REGION Network 79: TMP - ERROR - Tout Bajar Tope
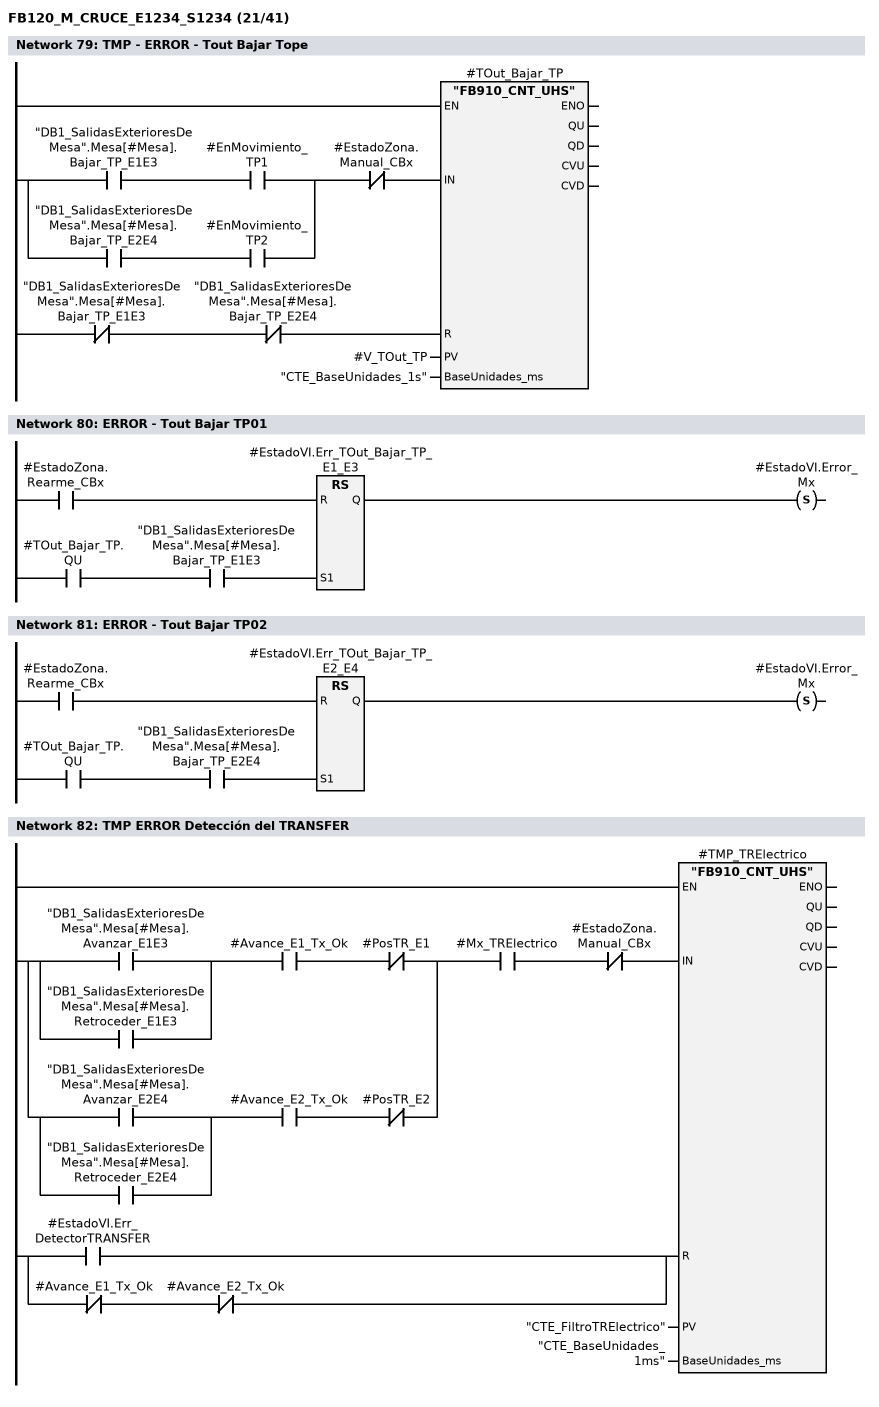
   RUNG wire#powerrail
      #TOut_Bajar_TP(IN := wire#w2, R := wire#w3, PV := #V_TOut_TP, BaseUnidades_ms := "CTE_BaseUnidades_1s", QU =>, QD =>, CVU =>, CVD =>)
   END_RUNG
   RUNG wire#powerrail
      Contact( "DB1_SalidasExterioresDeMesa".Mesa[#Mesa].Bajar_TP_E1E3 )
      Contact( #EnMovimiento_TP1 )
      wire#w1
      I_Contact( #EstadoZona.Manual_CBx )
   END_RUNG wire#w2
   RUNG wire#powerrail
      Contact( "DB1_SalidasExterioresDeMesa".Mesa[#Mesa].Bajar_TP_E2E4 )
      Contact( #EnMovimiento_TP2 )
   END_RUNG wire#w1
   RUNG wire#powerrail
      I_Contact( "DB1_SalidasExterioresDeMesa".Mesa[#Mesa].Bajar_TP_E1E3 )
      I_Contact( "DB1_SalidasExterioresDeMesa".Mesa[#Mesa].Bajar_TP_E2E4 )
   END_RUNG wire#w3
   // the same network as SCL:
   #TOut_Bajar_TP(IN := (("DB1_SalidasExterioresDeMesa".Mesa[#Mesa].Bajar_TP_E1E3 AND #EnMovimiento_TP1) OR ("DB1_SalidasExterioresDeMesa".Mesa[#Mesa].Bajar_TP_E2E4 AND #EnMovimiento_TP2)) AND NOT #EstadoZona.Manual_CBx,   // "FB910_CNT_UHS"
                  R := NOT "DB1_SalidasExterioresDeMesa".Mesa[#Mesa].Bajar_TP_E1E3 AND NOT "DB1_SalidasExterioresDeMesa".Mesa[#Mesa].Bajar_TP_E2E4,
                  PV := #V_TOut_TP,
                  BaseUnidades_ms := "CTE_BaseUnidades_1s");
END_REGION

REGION Network 80: ERROR - Tout Bajar TP01
   RUNG wire#powerrail
      Contact( #EstadoZona.Rearme_CBx )
      S_RS(operand := #EstadoVI.Err_TOut_Bajar_TP_E1_E3, s1 := wire#w1)
      S_Coil( #EstadoVI.Error_Mx )
   END_RUNG
   RUNG wire#powerrail
      Contact( #TOut_Bajar_TP.QU )
      Contact( "DB1_SalidasExterioresDeMesa".Mesa[#Mesa].Bajar_TP_E1E3 )
   END_RUNG wire#w1
   // the same network as SCL:
   IF #EstadoZona.Rearme_CBx THEN
       #EstadoVI.Err_TOut_Bajar_TP_E1_E3 := FALSE;   // RS flip-flop
   END_IF;
   IF #TOut_Bajar_TP.QU AND "DB1_SalidasExterioresDeMesa".Mesa[#Mesa].Bajar_TP_E1E3 THEN
       #EstadoVI.Err_TOut_Bajar_TP_E1_E3 := TRUE;
   END_IF;
   IF #EstadoVI.Err_TOut_Bajar_TP_E1_E3 THEN #EstadoVI.Error_Mx := TRUE; END_IF;
END_REGION

REGION Network 81: ERROR - Tout Bajar TP02
   RUNG wire#powerrail
      Contact( #EstadoZona.Rearme_CBx )
      S_RS(operand := #EstadoVI.Err_TOut_Bajar_TP_E2_E4, s1 := wire#w1)
      S_Coil( #EstadoVI.Error_Mx )
   END_RUNG
   RUNG wire#powerrail
      Contact( #TOut_Bajar_TP.QU )
      Contact( "DB1_SalidasExterioresDeMesa".Mesa[#Mesa].Bajar_TP_E2E4 )
   END_RUNG wire#w1
   // the same network as SCL:
   IF #EstadoZona.Rearme_CBx THEN
       #EstadoVI.Err_TOut_Bajar_TP_E2_E4 := FALSE;   // RS flip-flop
   END_IF;
   IF #TOut_Bajar_TP.QU AND "DB1_SalidasExterioresDeMesa".Mesa[#Mesa].Bajar_TP_E2E4 THEN
       #EstadoVI.Err_TOut_Bajar_TP_E2_E4 := TRUE;
   END_IF;
   IF #EstadoVI.Err_TOut_Bajar_TP_E2_E4 THEN #EstadoVI.Error_Mx := TRUE; END_IF;
END_REGION

REGION Network 82: TMP ERROR Detección del TRANSFER
   RUNG wire#powerrail
      #TMP_TRElectrico(IN := wire#w4, R := wire#w5, PV := "CTE_FiltroTRElectrico", BaseUnidades_ms := "CTE_BaseUnidades_1ms", QU =>, QD =>, CVU =>, CVD =>)
   END_RUNG
   RUNG wire#powerrail
      Contact( "DB1_SalidasExterioresDeMesa".Mesa[#Mesa].Avanzar_E1E3 )
      wire#w1
      Contact( #Avance_E1_Tx_Ok )
      I_Contact( #PosTR_E1 )
      wire#w2
      Contact( #Mx_TRElectrico )
      I_Contact( #EstadoZona.Manual_CBx )
   END_RUNG wire#w4
   RUNG wire#powerrail
      Contact( "DB1_SalidasExterioresDeMesa".Mesa[#Mesa].Retroceder_E1E3 )
   END_RUNG wire#w1
   RUNG wire#powerrail
      Contact( "DB1_SalidasExterioresDeMesa".Mesa[#Mesa].Avanzar_E2E4 )
      wire#w3
      Contact( #Avance_E2_Tx_Ok )
      I_Contact( #PosTR_E2 )
   END_RUNG wire#w2
   RUNG wire#powerrail
      Contact( "DB1_SalidasExterioresDeMesa".Mesa[#Mesa].Retroceder_E2E4 )
   END_RUNG wire#w3
   RUNG wire#powerrail
      Contact( #EstadoVI.Err_DetectorTRANSFER )
   END_RUNG wire#w5
   RUNG wire#powerrail
      I_Contact( #Avance_E1_Tx_Ok )
      I_Contact( #Avance_E2_Tx_Ok )
   END_RUNG wire#w5
   // the same network as SCL:
   #TMP_TRElectrico(IN := ((("DB1_SalidasExterioresDeMesa".Mesa[#Mesa].Avanzar_E1E3 OR "DB1_SalidasExterioresDeMesa".Mesa[#Mesa].Retroceder_E1E3) AND #Avance_E1_Tx_Ok AND NOT #PosTR_E1) OR (("DB1_SalidasExterioresDeMesa".Mesa[#Mesa].Avanzar_E2E4 OR "DB1_SalidasExterioresDeMesa".Mesa[#Mesa].Retroceder_E2E4) AND #Avance_E2_Tx_Ok AND NOT #PosTR_E2)) AND #Mx_TRElectrico AND NOT #EstadoZona.Manual_CBx,   // "FB910_CNT_UHS"
                    R := #EstadoVI.Err_DetectorTRANSFER OR (NOT #Avance_E1_Tx_Ok AND NOT #Avance_E2_Tx_Ok),
                    PV := "CTE_FiltroTRElectrico",
                    BaseUnidades_ms := "CTE_BaseUnidades_1ms");
END_REGION

REGION Network 83: ERROR - Detección del TRANSFER
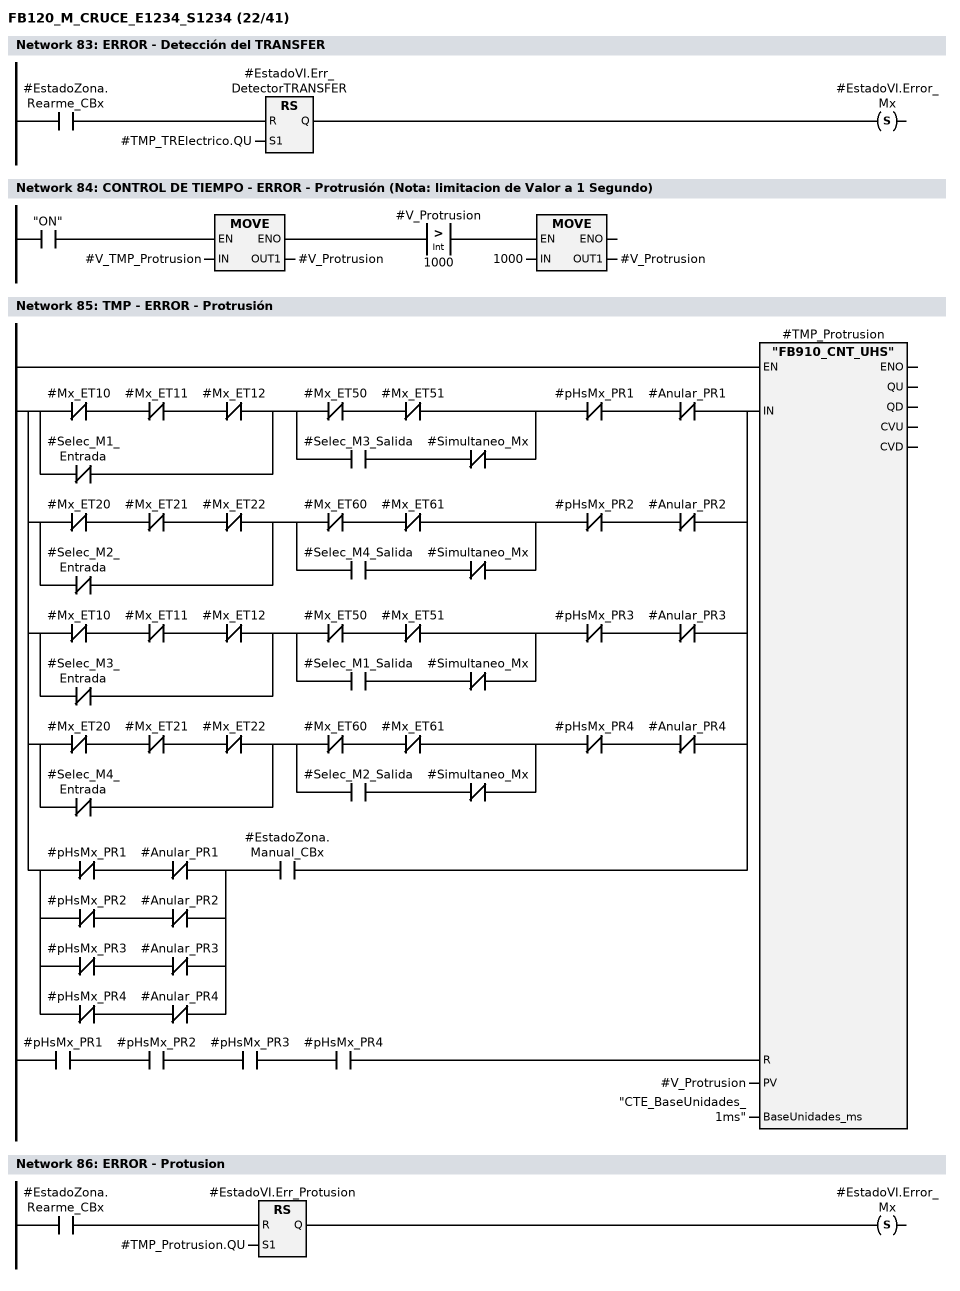
   RUNG wire#powerrail
      Contact( #EstadoZona.Rearme_CBx )
      S_RS(operand := #EstadoVI.Err_DetectorTRANSFER, s1 := #TMP_TRElectrico.QU)
      S_Coil( #EstadoVI.Error_Mx )
   END_RUNG
   // the same network as SCL:
   IF #EstadoZona.Rearme_CBx THEN
       #EstadoVI.Err_DetectorTRANSFER := FALSE;   // RS flip-flop
   END_IF;
   IF #TMP_TRElectrico.QU THEN #EstadoVI.Err_DetectorTRANSFER := TRUE; END_IF;
   IF #EstadoVI.Err_DetectorTRANSFER THEN #EstadoVI.Error_Mx := TRUE; END_IF;
END_REGION

REGION Network 84: CONTROL DE TIEMPO - ERROR - Protrusión (Nota: limitacion de Valor a 1 Segundo)
   RUNG wire#powerrail
      Contact( "ON" )
      Move(in := #V_TMP_Protrusion, out1 => #V_Protrusion)
      { S7_Templates := "SrcType := Int" } GT_Contact(in1 := #V_Protrusion, in2 := 1000)
      Move(in := 1000, out1 => #V_Protrusion)
   END_RUNG
   // the same network as SCL:
   IF "ON" THEN #V_Protrusion := #V_TMP_Protrusion; END_IF;
   IF "ON" AND (#V_Protrusion > 1000) THEN #V_Protrusion := 1000; END_IF;
END_REGION

REGION Network 85: TMP - ERROR - Protrusión
   RUNG wire#powerrail
      #TMP_Protrusion(IN := wire#w10, R := wire#w11, PV := #V_Protrusion, BaseUnidades_ms := "CTE_BaseUnidades_1ms", QU =>, QD =>, CVU =>, CVD =>)
   END_RUNG
   RUNG wire#powerrail
      I_Contact( #Mx_ET10 )
      I_Contact( #Mx_ET11 )
      I_Contact( #Mx_ET12 )
      wire#w1
      I_Contact( #Mx_ET50 )
      I_Contact( #Mx_ET51 )
      wire#w2
      I_Contact( #pHsMx_PR1 )
      I_Contact( #Anular_PR1 )
   END_RUNG wire#w10
   RUNG wire#powerrail
      I_Contact( #Selec_M1_Entrada )
   END_RUNG wire#w1
   RUNG wire#w1
      Contact( #Selec_M3_Salida )
      I_Contact( #Simultaneo_Mx )
   END_RUNG wire#w2
   RUNG wire#powerrail
      I_Contact( #Mx_ET20 )
      I_Contact( #Mx_ET21 )
      I_Contact( #Mx_ET22 )
      wire#w3
      I_Contact( #Mx_ET60 )
      I_Contact( #Mx_ET61 )
      wire#w4
      I_Contact( #pHsMx_PR2 )
      I_Contact( #Anular_PR2 )
   END_RUNG wire#w10
   RUNG wire#powerrail
      I_Contact( #Selec_M2_Entrada )
   END_RUNG wire#w3
   RUNG wire#w3
      Contact( #Selec_M4_Salida )
      I_Contact( #Simultaneo_Mx )
   END_RUNG wire#w4
   RUNG wire#powerrail
      I_Contact( #Mx_ET10 )
      I_Contact( #Mx_ET11 )
      I_Contact( #Mx_ET12 )
      wire#w5
      I_Contact( #Mx_ET50 )
      I_Contact( #Mx_ET51 )
      wire#w6
      I_Contact( #pHsMx_PR3 )
      I_Contact( #Anular_PR3 )
   END_RUNG wire#w10
   RUNG wire#powerrail
      I_Contact( #Selec_M3_Entrada )
   END_RUNG wire#w5
   RUNG wire#w5
      Contact( #Selec_M1_Salida )
      I_Contact( #Simultaneo_Mx )
   END_RUNG wire#w6
   RUNG wire#powerrail
      I_Contact( #Mx_ET20 )
      I_Contact( #Mx_ET21 )
      I_Contact( #Mx_ET22 )
      wire#w7
      I_Contact( #Mx_ET60 )
      I_Contact( #Mx_ET61 )
      wire#w8
      I_Contact( #pHsMx_PR4 )
      I_Contact( #Anular_PR4 )
   END_RUNG wire#w10
   RUNG wire#powerrail
      I_Contact( #Selec_M4_Entrada )
   END_RUNG wire#w7
   RUNG wire#w7
      Contact( #Selec_M2_Salida )
      I_Contact( #Simultaneo_Mx )
   END_RUNG wire#w8
   RUNG wire#powerrail
      I_Contact( #pHsMx_PR1 )
      I_Contact( #Anular_PR1 )
      wire#w9
      Contact( #EstadoZona.Manual_CBx )
   END_RUNG wire#w10
   RUNG wire#powerrail
      I_Contact( #pHsMx_PR2 )
      I_Contact( #Anular_PR2 )
   END_RUNG wire#w9
   RUNG wire#powerrail
      I_Contact( #pHsMx_PR3 )
      I_Contact( #Anular_PR3 )
   END_RUNG wire#w9
   RUNG wire#powerrail
      I_Contact( #pHsMx_PR4 )
      I_Contact( #Anular_PR4 )
   END_RUNG wire#w9
   RUNG wire#powerrail
      Contact( #pHsMx_PR1 )
      Contact( #pHsMx_PR2 )
      Contact( #pHsMx_PR3 )
      Contact( #pHsMx_PR4 )
   END_RUNG wire#w11
   // the same network as SCL:
   #TMP_Protrusion(IN := (((NOT #Mx_ET10 AND NOT #Mx_ET11 AND NOT #Mx_ET12) OR NOT #Selec_M1_Entrada) AND ((NOT #Mx_ET50 AND NOT #Mx_ET51) OR (#Selec_M3_Salida AND NOT #Simultaneo_Mx)) AND NOT #pHsMx_PR1 AND NOT #Anular_PR1) OR (((NOT #Mx_ET20 AND NOT #Mx_ET21 AND NOT #Mx_ET22) OR NOT #Selec_M2_Entrada) AND ((NOT #Mx_ET60 AND NOT #Mx_ET61) OR (#Selec_M4_Salida AND NOT #Simultaneo_Mx)) AND NOT #pHsMx_PR2 AND NOT #Anular_PR2) OR (((NOT #Mx_ET10 AND NOT #Mx_ET11 AND NOT #Mx_ET12) OR NOT #Selec_M3_Entrada) AND ((NOT #Mx_ET50 AND NOT #Mx_ET51) OR (#Selec_M1_Salida AND NOT #Simultaneo_Mx)) AND NOT #pHsMx_PR3 AND NOT #Anular_PR3) OR (((NOT #Mx_ET20 AND NOT #Mx_ET21 AND NOT #Mx_ET22) OR NOT #Selec_M4_Entrada) AND ((NOT #Mx_ET60 AND NOT #Mx_ET61) OR (#Selec_M2_Salida AND NOT #Simultaneo_Mx)) AND NOT #pHsMx_PR4 AND NOT #Anular_PR4) OR (((NOT #pHsMx_PR1 AND NOT #Anular_PR1) OR (NOT #pHsMx_PR2 AND NOT #Anular_PR2) OR (NOT #pHsMx_PR3 AND NOT #Anular_PR3) OR (NOT #pHsMx_PR4 AND NOT #Anular_PR4)) AND #EstadoZona.Manual_CBx),   // "FB910_CNT_UHS"
                   R := #pHsMx_PR1 AND #pHsMx_PR2 AND #pHsMx_PR3 AND #pHsMx_PR4,
                   PV := #V_Protrusion,
                   BaseUnidades_ms := "CTE_BaseUnidades_1ms");
END_REGION

REGION Network 86: ERROR - Protusion
   RUNG wire#powerrail
      Contact( #EstadoZona.Rearme_CBx )
      S_RS(operand := #EstadoVI.Err_Protusion, s1 := #TMP_Protrusion.QU)
      S_Coil( #EstadoVI.Error_Mx )
   END_RUNG
   // the same network as SCL:
   IF #EstadoZona.Rearme_CBx THEN
       #EstadoVI.Err_Protusion := FALSE;   // RS flip-flop
   END_IF;
   IF #TMP_Protrusion.QU THEN #EstadoVI.Err_Protusion := TRUE; END_IF;
   IF #EstadoVI.Err_Protusion THEN #EstadoVI.Error_Mx := TRUE; END_IF;
END_REGION

REGION Network 87: CONTADOR DE AUSENCIA DE LA "pHsSeg" DE CNTSeg - CNTApHs_CNTSeg_E1E3
   // Este contador asegura que la fotocélula con la que se empieza a contar el contador de seguridad ha dado ausencia. 
   // Por lo que con esto aseguramos que el contador de seguridad puede volver a comenzar a contar con la nueva paleta que se esta cargando.
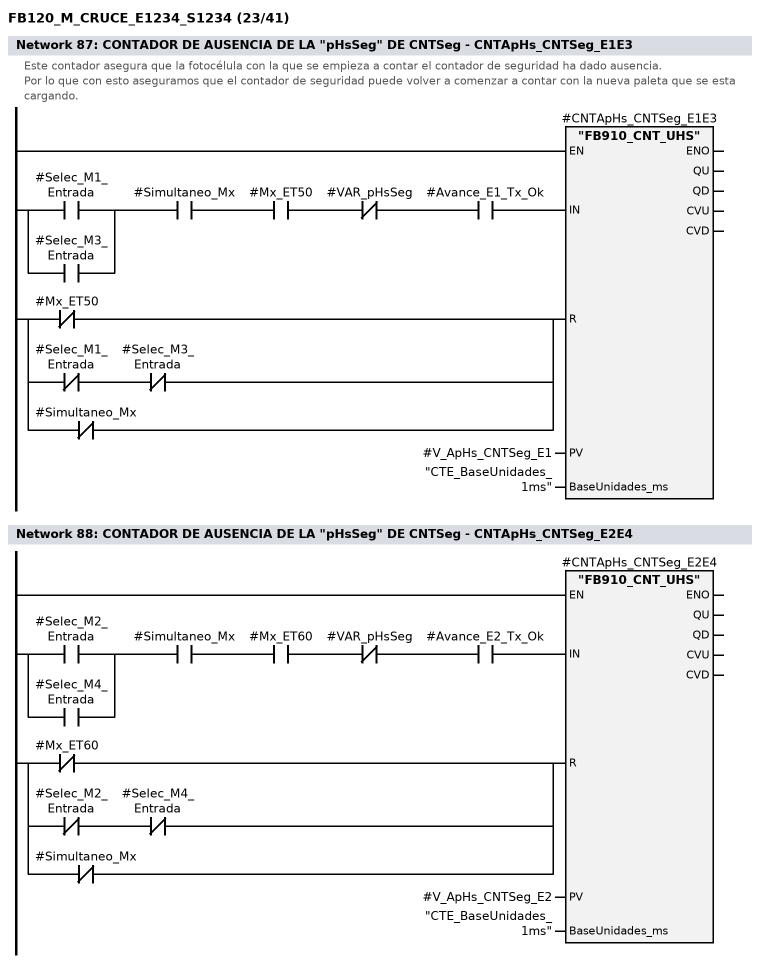
   RUNG wire#powerrail
      #CNTApHs_CNTSeg_E1E3(IN := wire#w2, R := wire#w3, PV := #V_ApHs_CNTSeg_E1, BaseUnidades_ms := "CTE_BaseUnidades_1ms", QU =>, QD =>, CVU =>, CVD =>)
   END_RUNG
   RUNG wire#powerrail
      Contact( #Selec_M1_Entrada )
      wire#w1
      Contact( #Simultaneo_Mx )
      Contact( #Mx_ET50 )
      I_Contact( #VAR_pHsSeg )
      Contact( #Avance_E1_Tx_Ok )
   END_RUNG wire#w2
   RUNG wire#powerrail
      Contact( #Selec_M3_Entrada )
   END_RUNG wire#w1
   RUNG wire#powerrail
      I_Contact( #Mx_ET50 )
   END_RUNG wire#w3
   RUNG wire#powerrail
      I_Contact( #Selec_M1_Entrada )
      I_Contact( #Selec_M3_Entrada )
   END_RUNG wire#w3
   RUNG wire#powerrail
      I_Contact( #Simultaneo_Mx )
   END_RUNG wire#w3
   // the same network as SCL:
   #CNTApHs_CNTSeg_E1E3(IN := (#Selec_M1_Entrada OR #Selec_M3_Entrada) AND #Simultaneo_Mx AND #Mx_ET50 AND NOT #VAR_pHsSeg AND #Avance_E1_Tx_Ok,   // "FB910_CNT_UHS"
                        R := NOT #Mx_ET50 OR (NOT #Selec_M1_Entrada AND NOT #Selec_M3_Entrada) OR NOT #Simultaneo_Mx,
                        PV := #V_ApHs_CNTSeg_E1,
                        BaseUnidades_ms := "CTE_BaseUnidades_1ms");
END_REGION

REGION Network 88: CONTADOR DE AUSENCIA DE LA "pHsSeg" DE CNTSeg - CNTApHs_CNTSeg_E2E4
   RUNG wire#powerrail
      #CNTApHs_CNTSeg_E2E4(IN := wire#w2, R := wire#w3, PV := #V_ApHs_CNTSeg_E2, BaseUnidades_ms := "CTE_BaseUnidades_1ms", QU =>, QD =>, CVU =>, CVD =>)
   END_RUNG
   RUNG wire#powerrail
      Contact( #Selec_M2_Entrada )
      wire#w1
      Contact( #Simultaneo_Mx )
      Contact( #Mx_ET60 )
      I_Contact( #VAR_pHsSeg )
      Contact( #Avance_E2_Tx_Ok )
   END_RUNG wire#w2
   RUNG wire#powerrail
      Contact( #Selec_M4_Entrada )
   END_RUNG wire#w1
   RUNG wire#powerrail
      I_Contact( #Mx_ET60 )
   END_RUNG wire#w3
   RUNG wire#powerrail
      I_Contact( #Selec_M2_Entrada )
      I_Contact( #Selec_M4_Entrada )
   END_RUNG wire#w3
   RUNG wire#powerrail
      I_Contact( #Simultaneo_Mx )
   END_RUNG wire#w3
   // the same network as SCL:
   #CNTApHs_CNTSeg_E2E4(IN := (#Selec_M2_Entrada OR #Selec_M4_Entrada) AND #Simultaneo_Mx AND #Mx_ET60 AND NOT #VAR_pHsSeg AND #Avance_E2_Tx_Ok,   // "FB910_CNT_UHS"
                        R := NOT #Mx_ET60 OR (NOT #Selec_M2_Entrada AND NOT #Selec_M4_Entrada) OR NOT #Simultaneo_Mx,
                        PV := #V_ApHs_CNTSeg_E2,
                        BaseUnidades_ms := "CTE_BaseUnidades_1ms");
END_REGION

REGION Network 89: CONTADOR DE SEGURIDAD DE PRESENCIA - CNTSeg_pHsMx_E1E3
   // VAR_pHsSeg ---> Inicio del CNT de Seguridad (Ha funcionar) ---- NOTA : Diferente con FB264
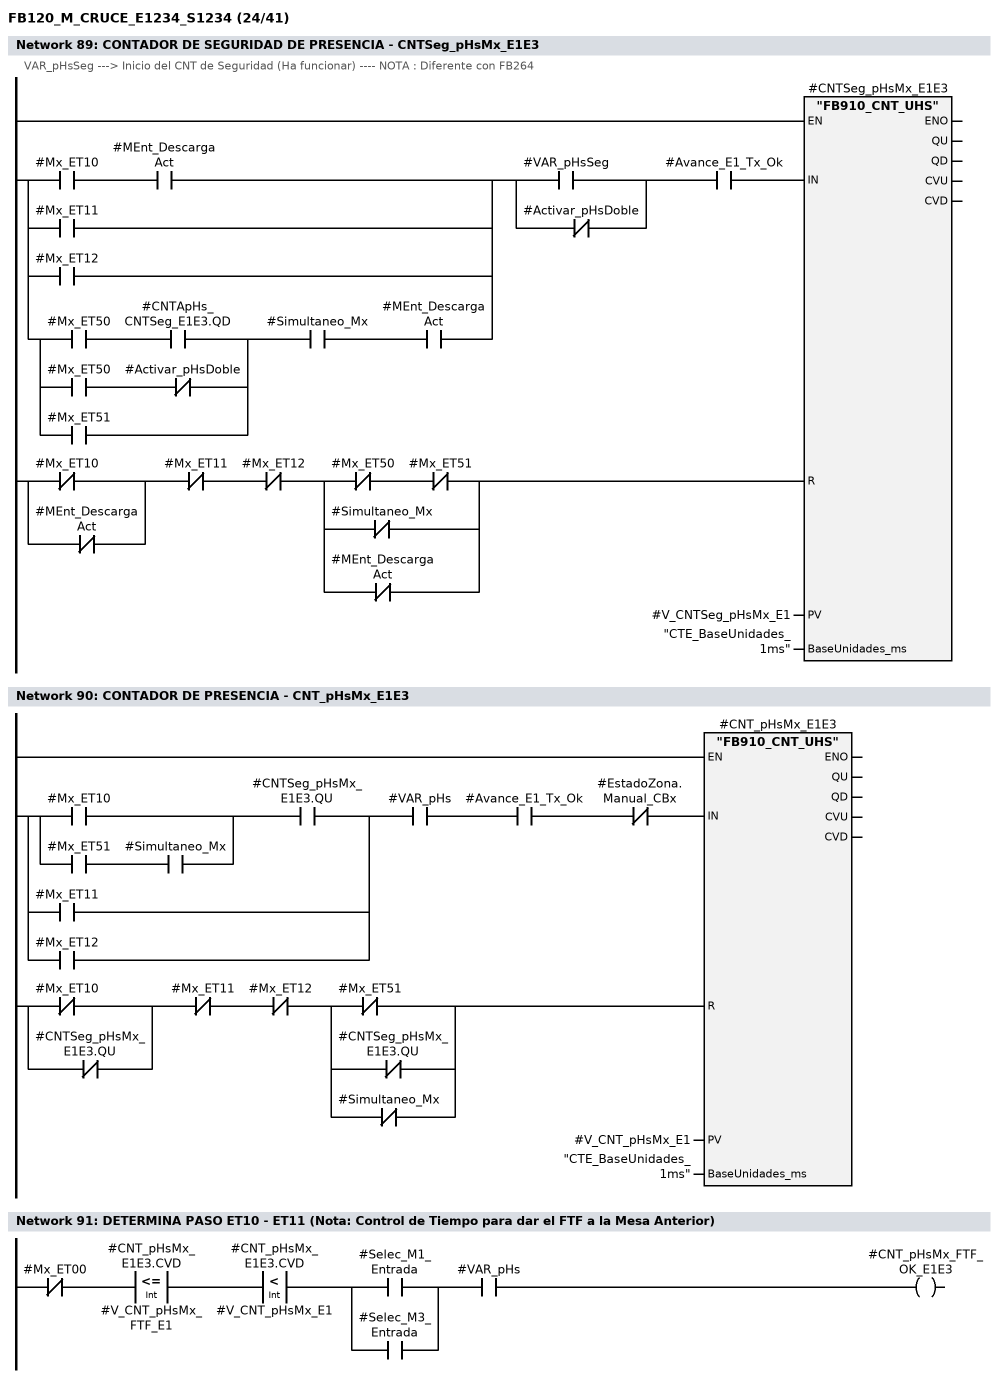
   RUNG wire#powerrail
      #CNTSeg_pHsMx_E1E3(IN := wire#w4, R := wire#w7, PV := #V_CNTSeg_pHsMx_E1, BaseUnidades_ms := "CTE_BaseUnidades_1ms", QU =>, QD =>, CVU =>, CVD =>)
   END_RUNG
   RUNG wire#powerrail
      Contact( #Mx_ET10 )
      Contact( #MEnt_DescargaAct )
      wire#w1
      Contact( #VAR_pHsSeg )
      wire#w3
      Contact( #Avance_E1_Tx_Ok )
   END_RUNG wire#w4
   RUNG wire#powerrail
      Contact( #Mx_ET11 )
   END_RUNG wire#w1
   RUNG wire#powerrail
      Contact( #Mx_ET12 )
   END_RUNG wire#w1
   RUNG wire#powerrail
      Contact( #Mx_ET50 )
      Contact( #CNTApHs_CNTSeg_E1E3.QD )
      wire#w2
      Contact( #Simultaneo_Mx )
      Contact( #MEnt_DescargaAct )
   END_RUNG wire#w1
   RUNG wire#powerrail
      Contact( #Mx_ET50 )
      I_Contact( #Activar_pHsDoble )
   END_RUNG wire#w2
   RUNG wire#powerrail
      Contact( #Mx_ET51 )
   END_RUNG wire#w2
   RUNG wire#w1
      I_Contact( #Activar_pHsDoble )
   END_RUNG wire#w3
   RUNG wire#powerrail
      I_Contact( #Mx_ET10 )
      wire#w5
      I_Contact( #Mx_ET11 )
      I_Contact( #Mx_ET12 )
      wire#w6
      I_Contact( #Mx_ET50 )
      I_Contact( #Mx_ET51 )
   END_RUNG wire#w7
   RUNG wire#powerrail
      I_Contact( #MEnt_DescargaAct )
   END_RUNG wire#w5
   RUNG wire#w6
      I_Contact( #Simultaneo_Mx )
   END_RUNG wire#w7
   RUNG wire#w6
      I_Contact( #MEnt_DescargaAct )
   END_RUNG wire#w7
   // the same network as SCL:
   #CNTSeg_pHsMx_E1E3(IN := ((#Mx_ET10 AND #MEnt_DescargaAct) OR #Mx_ET11 OR #Mx_ET12 OR (((#Mx_ET50 AND #CNTApHs_CNTSeg_E1E3.QD) OR (#Mx_ET50 AND NOT #Activar_pHsDoble) OR #Mx_ET51) AND #Simultaneo_Mx AND #MEnt_DescargaAct)) AND (#VAR_pHsSeg OR NOT #Activar_pHsDoble) AND #Avance_E1_Tx_Ok,   // "FB910_CNT_UHS"
                      R := (NOT #Mx_ET10 OR NOT #MEnt_DescargaAct) AND NOT #Mx_ET11 AND NOT #Mx_ET12 AND ((NOT #Mx_ET50 AND NOT #Mx_ET51) OR NOT #Simultaneo_Mx OR NOT #MEnt_DescargaAct),
                      PV := #V_CNTSeg_pHsMx_E1,
                      BaseUnidades_ms := "CTE_BaseUnidades_1ms");
END_REGION

REGION Network 90: CONTADOR DE PRESENCIA - CNT_pHsMx_E1E3
   RUNG wire#powerrail
      #CNT_pHsMx_E1E3(IN := wire#w3, R := wire#w6, PV := #V_CNT_pHsMx_E1, BaseUnidades_ms := "CTE_BaseUnidades_1ms", QU =>, QD =>, CVU =>, CVD =>)
   END_RUNG
   RUNG wire#powerrail
      Contact( #Mx_ET10 )
      wire#w1
      Contact( #CNTSeg_pHsMx_E1E3.QU )
      wire#w2
      Contact( #VAR_pHs )
      Contact( #Avance_E1_Tx_Ok )
      I_Contact( #EstadoZona.Manual_CBx )
   END_RUNG wire#w3
   RUNG wire#powerrail
      Contact( #Mx_ET51 )
      Contact( #Simultaneo_Mx )
   END_RUNG wire#w1
   RUNG wire#powerrail
      Contact( #Mx_ET11 )
   END_RUNG wire#w2
   RUNG wire#powerrail
      Contact( #Mx_ET12 )
   END_RUNG wire#w2
   RUNG wire#powerrail
      I_Contact( #Mx_ET10 )
      wire#w4
      I_Contact( #Mx_ET11 )
      I_Contact( #Mx_ET12 )
      wire#w5
      I_Contact( #Mx_ET51 )
   END_RUNG wire#w6
   RUNG wire#powerrail
      I_Contact( #CNTSeg_pHsMx_E1E3.QU )
   END_RUNG wire#w4
   RUNG wire#w5
      I_Contact( #CNTSeg_pHsMx_E1E3.QU )
   END_RUNG wire#w6
   RUNG wire#w5
      I_Contact( #Simultaneo_Mx )
   END_RUNG wire#w6
   // the same network as SCL:
   #CNT_pHsMx_E1E3(IN := (((#Mx_ET10 OR (#Mx_ET51 AND #Simultaneo_Mx)) AND #CNTSeg_pHsMx_E1E3.QU) OR #Mx_ET11 OR #Mx_ET12) AND #VAR_pHs AND #Avance_E1_Tx_Ok AND NOT #EstadoZona.Manual_CBx,   // "FB910_CNT_UHS"
                   R := (NOT #Mx_ET10 OR NOT #CNTSeg_pHsMx_E1E3.QU) AND NOT #Mx_ET11 AND NOT #Mx_ET12 AND (NOT #Mx_ET51 OR NOT #CNTSeg_pHsMx_E1E3.QU OR NOT #Simultaneo_Mx),
                   PV := #V_CNT_pHsMx_E1,
                   BaseUnidades_ms := "CTE_BaseUnidades_1ms");
END_REGION

REGION Network 91: DETERMINA PASO ET10 - ET11 (Nota: Control de Tiempo para dar el FTF a la Mesa Anterior)
   RUNG wire#powerrail
      I_Contact( #Mx_ET00 )
      { S7_Templates := "SrcType := Int" } LE_Contact(in1 := #CNT_pHsMx_E1E3.CVD, in2 := #V_CNT_pHsMx_FTF_E1)
      { S7_Templates := "SrcType := Int" } LT_Contact(in1 := #CNT_pHsMx_E1E3.CVD, in2 := #V_CNT_pHsMx_E1)
      wire#w1
      Contact( #Selec_M1_Entrada )
      wire#w2
      Contact( #VAR_pHs )
      Coil( #CNT_pHsMx_FTF_OK_E1E3 )
   END_RUNG
   RUNG wire#w1
      Contact( #Selec_M3_Entrada )
   END_RUNG wire#w2
   // the same network as SCL:
   #CNT_pHsMx_FTF_OK_E1E3 := NOT #Mx_ET00 AND (#CNT_pHsMx_E1E3.CVD <= #V_CNT_pHsMx_FTF_E1) AND (#CNT_pHsMx_E1E3.CVD < #V_CNT_pHsMx_E1) AND (#Selec_M1_Entrada OR #Selec_M3_Entrada) AND #VAR_pHs;
END_REGION

REGION Network 92: CONTADOR DE SEGURIDAD DE PRESENCIA - CNTSeg_pHsMx_E2E4
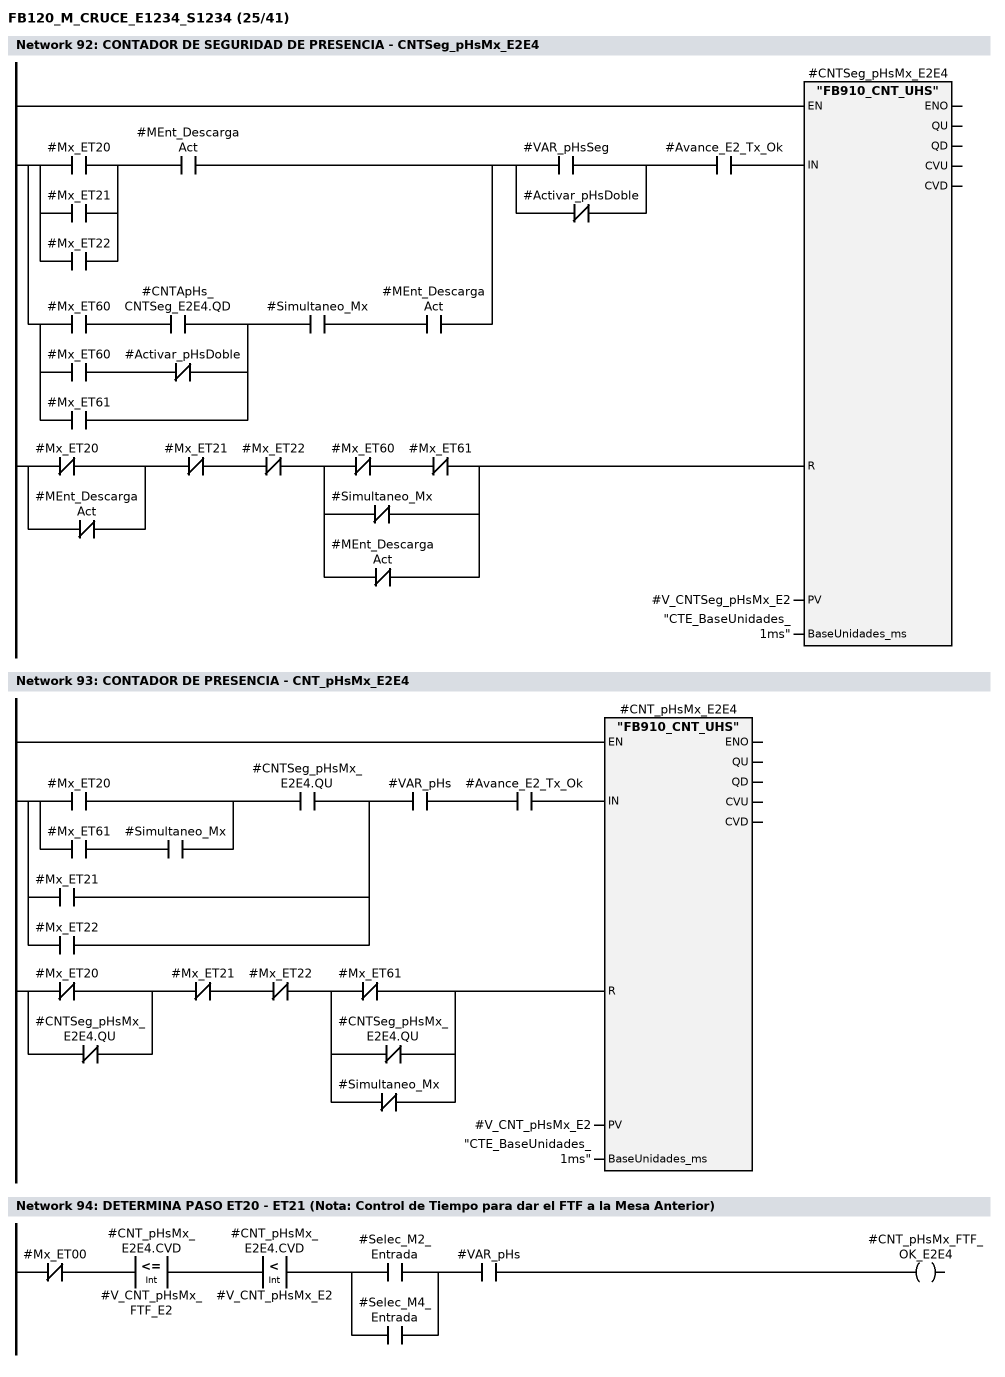
   RUNG wire#powerrail
      #CNTSeg_pHsMx_E2E4(IN := wire#w5, R := wire#w8, PV := #V_CNTSeg_pHsMx_E2, BaseUnidades_ms := "CTE_BaseUnidades_1ms", QU =>, QD =>, CVU =>, CVD =>)
   END_RUNG
   RUNG wire#powerrail
      Contact( #Mx_ET20 )
      wire#w1
      Contact( #MEnt_DescargaAct )
      wire#w2
      Contact( #VAR_pHsSeg )
      wire#w4
      Contact( #Avance_E2_Tx_Ok )
   END_RUNG wire#w5
   RUNG wire#powerrail
      Contact( #Mx_ET21 )
   END_RUNG wire#w1
   RUNG wire#powerrail
      Contact( #Mx_ET22 )
   END_RUNG wire#w1
   RUNG wire#powerrail
      Contact( #Mx_ET60 )
      Contact( #CNTApHs_CNTSeg_E2E4.QD )
      wire#w3
      Contact( #Simultaneo_Mx )
      Contact( #MEnt_DescargaAct )
   END_RUNG wire#w2
   RUNG wire#powerrail
      Contact( #Mx_ET60 )
      I_Contact( #Activar_pHsDoble )
   END_RUNG wire#w3
   RUNG wire#powerrail
      Contact( #Mx_ET61 )
   END_RUNG wire#w3
   RUNG wire#w2
      I_Contact( #Activar_pHsDoble )
   END_RUNG wire#w4
   RUNG wire#powerrail
      I_Contact( #Mx_ET20 )
      wire#w6
      I_Contact( #Mx_ET21 )
      I_Contact( #Mx_ET22 )
      wire#w7
      I_Contact( #Mx_ET60 )
      I_Contact( #Mx_ET61 )
   END_RUNG wire#w8
   RUNG wire#powerrail
      I_Contact( #MEnt_DescargaAct )
   END_RUNG wire#w6
   RUNG wire#w7
      I_Contact( #Simultaneo_Mx )
   END_RUNG wire#w8
   RUNG wire#w7
      I_Contact( #MEnt_DescargaAct )
   END_RUNG wire#w8
   // the same network as SCL:
   #CNTSeg_pHsMx_E2E4(IN := (((#Mx_ET20 OR #Mx_ET21 OR #Mx_ET22) AND #MEnt_DescargaAct) OR (((#Mx_ET60 AND #CNTApHs_CNTSeg_E2E4.QD) OR (#Mx_ET60 AND NOT #Activar_pHsDoble) OR #Mx_ET61) AND #Simultaneo_Mx AND #MEnt_DescargaAct)) AND (#VAR_pHsSeg OR NOT #Activar_pHsDoble) AND #Avance_E2_Tx_Ok,   // "FB910_CNT_UHS"
                      R := (NOT #Mx_ET20 OR NOT #MEnt_DescargaAct) AND NOT #Mx_ET21 AND NOT #Mx_ET22 AND ((NOT #Mx_ET60 AND NOT #Mx_ET61) OR NOT #Simultaneo_Mx OR NOT #MEnt_DescargaAct),
                      PV := #V_CNTSeg_pHsMx_E2,
                      BaseUnidades_ms := "CTE_BaseUnidades_1ms");
END_REGION

REGION Network 93: CONTADOR DE PRESENCIA - CNT_pHsMx_E2E4
   RUNG wire#powerrail
      #CNT_pHsMx_E2E4(IN := wire#w3, R := wire#w6, PV := #V_CNT_pHsMx_E2, BaseUnidades_ms := "CTE_BaseUnidades_1ms", QU =>, QD =>, CVU =>, CVD =>)
   END_RUNG
   RUNG wire#powerrail
      Contact( #Mx_ET20 )
      wire#w1
      Contact( #CNTSeg_pHsMx_E2E4.QU )
      wire#w2
      Contact( #VAR_pHs )
      Contact( #Avance_E2_Tx_Ok )
   END_RUNG wire#w3
   RUNG wire#powerrail
      Contact( #Mx_ET61 )
      Contact( #Simultaneo_Mx )
   END_RUNG wire#w1
   RUNG wire#powerrail
      Contact( #Mx_ET21 )
   END_RUNG wire#w2
   RUNG wire#powerrail
      Contact( #Mx_ET22 )
   END_RUNG wire#w2
   RUNG wire#powerrail
      I_Contact( #Mx_ET20 )
      wire#w4
      I_Contact( #Mx_ET21 )
      I_Contact( #Mx_ET22 )
      wire#w5
      I_Contact( #Mx_ET61 )
   END_RUNG wire#w6
   RUNG wire#powerrail
      I_Contact( #CNTSeg_pHsMx_E2E4.QU )
   END_RUNG wire#w4
   RUNG wire#w5
      I_Contact( #CNTSeg_pHsMx_E2E4.QU )
   END_RUNG wire#w6
   RUNG wire#w5
      I_Contact( #Simultaneo_Mx )
   END_RUNG wire#w6
   // the same network as SCL:
   #CNT_pHsMx_E2E4(IN := (((#Mx_ET20 OR (#Mx_ET61 AND #Simultaneo_Mx)) AND #CNTSeg_pHsMx_E2E4.QU) OR #Mx_ET21 OR #Mx_ET22) AND #VAR_pHs AND #Avance_E2_Tx_Ok,   // "FB910_CNT_UHS"
                   R := (NOT #Mx_ET20 OR NOT #CNTSeg_pHsMx_E2E4.QU) AND NOT #Mx_ET21 AND NOT #Mx_ET22 AND (NOT #Mx_ET61 OR NOT #CNTSeg_pHsMx_E2E4.QU OR NOT #Simultaneo_Mx),
                   PV := #V_CNT_pHsMx_E2,
                   BaseUnidades_ms := "CTE_BaseUnidades_1ms");
END_REGION

REGION Network 94: DETERMINA PASO ET20 - ET21 (Nota: Control de Tiempo para dar el FTF a la Mesa Anterior)
   RUNG wire#powerrail
      I_Contact( #Mx_ET00 )
      { S7_Templates := "SrcType := Int" } LE_Contact(in1 := #CNT_pHsMx_E2E4.CVD, in2 := #V_CNT_pHsMx_FTF_E2)
      { S7_Templates := "SrcType := Int" } LT_Contact(in1 := #CNT_pHsMx_E2E4.CVD, in2 := #V_CNT_pHsMx_E2)
      wire#w1
      Contact( #Selec_M2_Entrada )
      wire#w2
      Contact( #VAR_pHs )
      Coil( #CNT_pHsMx_FTF_OK_E2E4 )
   END_RUNG
   RUNG wire#w1
      Contact( #Selec_M4_Entrada )
   END_RUNG wire#w2
   // the same network as SCL:
   #CNT_pHsMx_FTF_OK_E2E4 := NOT #Mx_ET00 AND (#CNT_pHsMx_E2E4.CVD <= #V_CNT_pHsMx_FTF_E2) AND (#CNT_pHsMx_E2E4.CVD < #V_CNT_pHsMx_E2) AND (#Selec_M2_Entrada OR #Selec_M4_Entrada) AND #VAR_pHs;
END_REGION

REGION Network 95: CONTADOR SEGURIDAD DE AUSENCIA - CNTSeg_ApHsMx ??????? RESTAR VALOR DE POSICIONAMIENTO
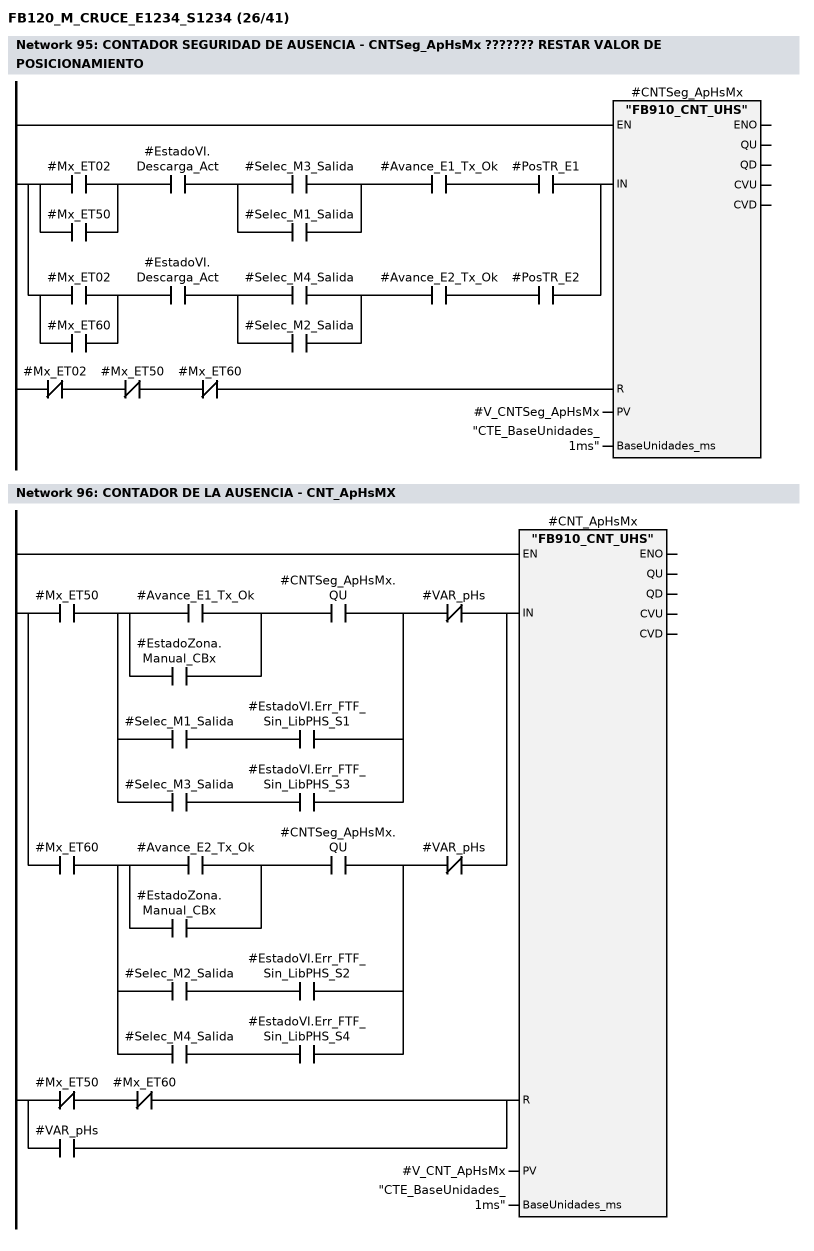
   RUNG wire#powerrail
      #CNTSeg_ApHsMx(IN := wire#w7, R := wire#w8, PV := #V_CNTSeg_ApHsMx, BaseUnidades_ms := "CTE_BaseUnidades_1ms", QU =>, QD =>, CVU =>, CVD =>)
   END_RUNG
   RUNG wire#powerrail
      Contact( #Mx_ET02 )
      wire#w1
      Contact( #EstadoVI.Descarga_Act )
      wire#w2
      Contact( #Selec_M3_Salida )
      wire#w3
      Contact( #Avance_E1_Tx_Ok )
      Contact( #PosTR_E1 )
   END_RUNG wire#w7
   RUNG wire#powerrail
      Contact( #Mx_ET50 )
   END_RUNG wire#w1
   RUNG wire#w2
      Contact( #Selec_M1_Salida )
   END_RUNG wire#w3
   RUNG wire#powerrail
      Contact( #Mx_ET02 )
      wire#w4
      Contact( #EstadoVI.Descarga_Act )
      wire#w5
      Contact( #Selec_M4_Salida )
      wire#w6
      Contact( #Avance_E2_Tx_Ok )
      Contact( #PosTR_E2 )
   END_RUNG wire#w7
   RUNG wire#powerrail
      Contact( #Mx_ET60 )
   END_RUNG wire#w4
   RUNG wire#w5
      Contact( #Selec_M2_Salida )
   END_RUNG wire#w6
   RUNG wire#powerrail
      I_Contact( #Mx_ET02 )
      I_Contact( #Mx_ET50 )
      I_Contact( #Mx_ET60 )
   END_RUNG wire#w8
   // the same network as SCL:
   #CNTSeg_ApHsMx(IN := ((#Mx_ET02 OR #Mx_ET50) AND #EstadoVI.Descarga_Act AND (#Selec_M3_Salida OR #Selec_M1_Salida) AND #Avance_E1_Tx_Ok AND #PosTR_E1) OR ((#Mx_ET02 OR #Mx_ET60) AND #EstadoVI.Descarga_Act AND (#Selec_M4_Salida OR #Selec_M2_Salida) AND #Avance_E2_Tx_Ok AND #PosTR_E2),   // "FB910_CNT_UHS"
                  R := NOT #Mx_ET02 AND NOT #Mx_ET50 AND NOT #Mx_ET60,
                  PV := #V_CNTSeg_ApHsMx,
                  BaseUnidades_ms := "CTE_BaseUnidades_1ms");
END_REGION

REGION Network 96: CONTADOR DE LA AUSENCIA - CNT_ApHsMX
   RUNG wire#powerrail
      #CNT_ApHsMx(IN := wire#w7, R := wire#w8, PV := #V_CNT_ApHsMx, BaseUnidades_ms := "CTE_BaseUnidades_1ms", QU =>, QD =>, CVU =>, CVD =>)
   END_RUNG
   RUNG wire#powerrail
      Contact( #Mx_ET50 )
      wire#w1
      Contact( #Avance_E1_Tx_Ok )
      wire#w2
      Contact( #CNTSeg_ApHsMx.QU )
      wire#w3
      I_Contact( #VAR_pHs )
   END_RUNG wire#w7
   RUNG wire#w1
      Contact( #EstadoZona.Manual_CBx )
   END_RUNG wire#w2
   RUNG wire#w1
      Contact( #Selec_M1_Salida )
      Contact( #EstadoVI.Err_FTF_Sin_LibPHS_S1 )
   END_RUNG wire#w3
   RUNG wire#w1
      Contact( #Selec_M3_Salida )
      Contact( #EstadoVI.Err_FTF_Sin_LibPHS_S3 )
   END_RUNG wire#w3
   RUNG wire#powerrail
      Contact( #Mx_ET60 )
      wire#w4
      Contact( #Avance_E2_Tx_Ok )
      wire#w5
      Contact( #CNTSeg_ApHsMx.QU )
      wire#w6
      I_Contact( #VAR_pHs )
   END_RUNG wire#w7
   RUNG wire#w4
      Contact( #EstadoZona.Manual_CBx )
   END_RUNG wire#w5
   RUNG wire#w4
      Contact( #Selec_M2_Salida )
      Contact( #EstadoVI.Err_FTF_Sin_LibPHS_S2 )
   END_RUNG wire#w6
   RUNG wire#w4
      Contact( #Selec_M4_Salida )
      Contact( #EstadoVI.Err_FTF_Sin_LibPHS_S4 )
   END_RUNG wire#w6
   RUNG wire#powerrail
      I_Contact( #Mx_ET50 )
      I_Contact( #Mx_ET60 )
   END_RUNG wire#w8
   RUNG wire#powerrail
      Contact( #VAR_pHs )
   END_RUNG wire#w8
   // the same network as SCL:
   #CNT_ApHsMx(IN := (#Mx_ET50 AND (((#Avance_E1_Tx_Ok OR #EstadoZona.Manual_CBx) AND #CNTSeg_ApHsMx.QU) OR (#Selec_M1_Salida AND #EstadoVI.Err_FTF_Sin_LibPHS_S1) OR (#Selec_M3_Salida AND #EstadoVI.Err_FTF_Sin_LibPHS_S3)) AND NOT #VAR_pHs) OR (#Mx_ET60 AND (((#Avance_E2_Tx_Ok OR #EstadoZona.Manual_CBx) AND #CNTSeg_ApHsMx.QU) OR (#Selec_M2_Salida AND #EstadoVI.Err_FTF_Sin_LibPHS_S2) OR (#Selec_M4_Salida AND #EstadoVI.Err_FTF_Sin_LibPHS_S4)) AND NOT #VAR_pHs),   // "FB910_CNT_UHS"
               R := (NOT #Mx_ET50 AND NOT #Mx_ET60) OR #VAR_pHs,
               PV := #V_CNT_ApHsMx,
               BaseUnidades_ms := "CTE_BaseUnidades_1ms");
END_REGION

REGION Network 97: TEMPORIZADOR DE BLOQUEO DE MESA
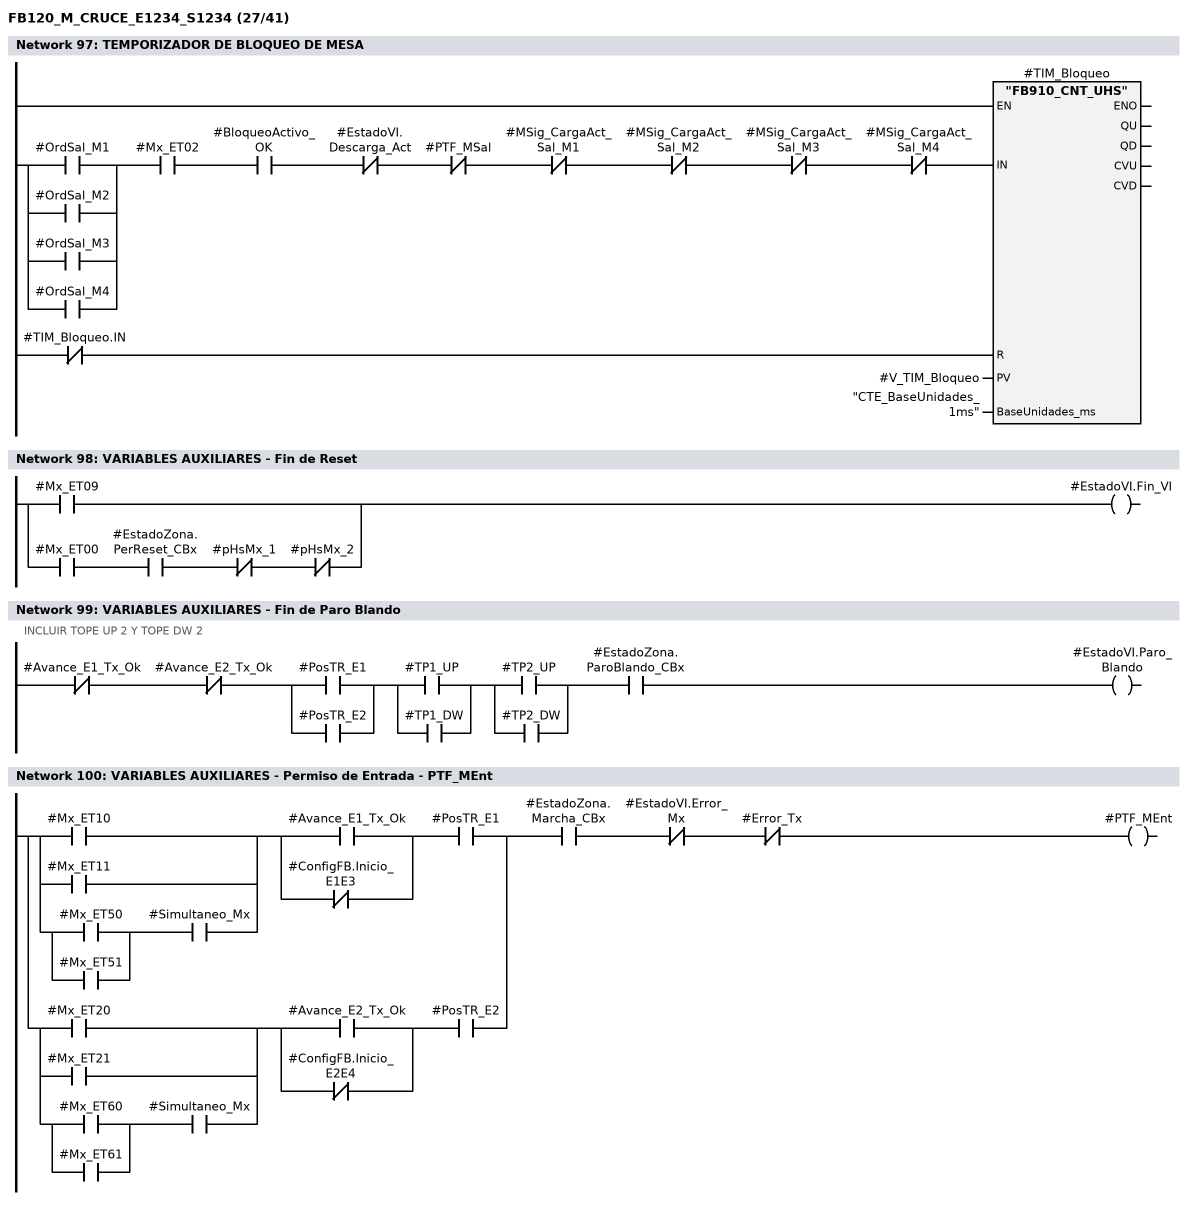
   RUNG wire#powerrail
      #TIM_Bloqueo(IN := wire#w2, R := wire#w3, PV := #V_TIM_Bloqueo, BaseUnidades_ms := "CTE_BaseUnidades_1ms", QU =>, QD =>, CVU =>, CVD =>)
   END_RUNG
   RUNG wire#powerrail
      Contact( #OrdSal_M1 )
      wire#w1
      Contact( #Mx_ET02 )
      Contact( #BloqueoActivo_OK )
      I_Contact( #EstadoVI.Descarga_Act )
      I_Contact( #PTF_MSal )
      I_Contact( #MSig_CargaAct_Sal_M1 )
      I_Contact( #MSig_CargaAct_Sal_M2 )
      I_Contact( #MSig_CargaAct_Sal_M3 )
      I_Contact( #MSig_CargaAct_Sal_M4 )
   END_RUNG wire#w2
   RUNG wire#powerrail
      Contact( #OrdSal_M2 )
   END_RUNG wire#w1
   RUNG wire#powerrail
      Contact( #OrdSal_M3 )
   END_RUNG wire#w1
   RUNG wire#powerrail
      Contact( #OrdSal_M4 )
   END_RUNG wire#w1
   RUNG wire#powerrail
      I_Contact( #TIM_Bloqueo.IN )
   END_RUNG wire#w3
   // the same network as SCL:
   #TIM_Bloqueo(IN := (#OrdSal_M1 OR #OrdSal_M2 OR #OrdSal_M3 OR #OrdSal_M4) AND #Mx_ET02 AND #BloqueoActivo_OK AND NOT #EstadoVI.Descarga_Act AND NOT #PTF_MSal AND NOT #MSig_CargaAct_Sal_M1 AND NOT #MSig_CargaAct_Sal_M2 AND NOT #MSig_CargaAct_Sal_M3 AND NOT #MSig_CargaAct_Sal_M4,   // "FB910_CNT_UHS"
                R := NOT #TIM_Bloqueo.IN,
                PV := #V_TIM_Bloqueo,
                BaseUnidades_ms := "CTE_BaseUnidades_1ms");
END_REGION

REGION Network 98: VARIABLES AUXILIARES - Fin de Reset
   RUNG wire#powerrail
      Contact( #Mx_ET09 )
      wire#w1
      Coil( #EstadoVI.Fin_VI )
   END_RUNG
   RUNG wire#powerrail
      Contact( #Mx_ET00 )
      Contact( #EstadoZona.PerReset_CBx )
      I_Contact( #pHsMx_1 )
      I_Contact( #pHsMx_2 )
   END_RUNG wire#w1
   // the same network as SCL:
   #EstadoVI.Fin_VI := #Mx_ET09 OR (#Mx_ET00 AND #EstadoZona.PerReset_CBx AND NOT #pHsMx_1 AND NOT #pHsMx_2);
END_REGION

REGION Network 99: VARIABLES AUXILIARES - Fin de Paro Blando
   // INCLUIR TOPE UP 2 Y TOPE DW 2
   RUNG wire#powerrail
      I_Contact( #Avance_E1_Tx_Ok )
      I_Contact( #Avance_E2_Tx_Ok )
      wire#w1
      Contact( #PosTR_E1 )
      wire#w2
      Contact( #TP1_UP )
      wire#w3
      Contact( #TP2_UP )
      wire#w4
      Contact( #EstadoZona.ParoBlando_CBx )
      Coil( #EstadoVI.Paro_Blando )
   END_RUNG
   RUNG wire#w1
      Contact( #PosTR_E2 )
   END_RUNG wire#w2
   RUNG wire#w2
      Contact( #TP1_DW )
   END_RUNG wire#w3
   RUNG wire#w3
      Contact( #TP2_DW )
   END_RUNG wire#w4
   // the same network as SCL:
   #EstadoVI.Paro_Blando := NOT #Avance_E1_Tx_Ok AND NOT #Avance_E2_Tx_Ok AND (#PosTR_E1 OR #PosTR_E2) AND (#TP1_UP OR #TP1_DW) AND (#TP2_UP OR #TP2_DW) AND #EstadoZona.ParoBlando_CBx;
END_REGION

REGION Network 100: VARIABLES AUXILIARES - Permiso de Entrada - PTF_MEnt
   RUNG wire#powerrail
      Contact( #Mx_ET10 )
      wire#w1
      Contact( #Avance_E1_Tx_Ok )
      wire#w3
      Contact( #PosTR_E1 )
      wire#w4
      Contact( #EstadoZona.Marcha_CBx )
      I_Contact( #EstadoVI.Error_Mx )
      I_Contact( #Error_Tx )
      Coil( #PTF_MEnt )
   END_RUNG
   RUNG wire#powerrail
      Contact( #Mx_ET11 )
   END_RUNG wire#w1
   RUNG wire#powerrail
      Contact( #Mx_ET50 )
      wire#w2
      Contact( #Simultaneo_Mx )
   END_RUNG wire#w1
   RUNG wire#powerrail
      Contact( #Mx_ET51 )
   END_RUNG wire#w2
   RUNG wire#w1
      I_Contact( #ConfigFB.Inicio_E1E3 )
   END_RUNG wire#w3
   RUNG wire#powerrail
      Contact( #Mx_ET20 )
      wire#w5
      Contact( #Avance_E2_Tx_Ok )
      wire#w7
      Contact( #PosTR_E2 )
   END_RUNG wire#w4
   RUNG wire#powerrail
      Contact( #Mx_ET21 )
   END_RUNG wire#w5
   RUNG wire#powerrail
      Contact( #Mx_ET60 )
      wire#w6
      Contact( #Simultaneo_Mx )
   END_RUNG wire#w5
   RUNG wire#powerrail
      Contact( #Mx_ET61 )
   END_RUNG wire#w6
   RUNG wire#w5
      I_Contact( #ConfigFB.Inicio_E2E4 )
   END_RUNG wire#w7
   // the same network as SCL:
   #PTF_MEnt := (((#Mx_ET10 OR #Mx_ET11 OR ((#Mx_ET50 OR #Mx_ET51) AND #Simultaneo_Mx)) AND (#Avance_E1_Tx_Ok OR NOT #ConfigFB.Inicio_E1E3) AND #PosTR_E1) OR ((#Mx_ET20 OR #Mx_ET21 OR ((#Mx_ET60 OR #Mx_ET61) AND #Simultaneo_Mx)) AND (#Avance_E2_Tx_Ok OR NOT #ConfigFB.Inicio_E2E4) AND #PosTR_E2)) AND #EstadoZona.Marcha_CBx AND NOT #EstadoVI.Error_Mx AND NOT #Error_Tx;
END_REGION

REGION Network 101: VARIABLES AUXILIARES - Aviso de Salida - AVTF_MSal
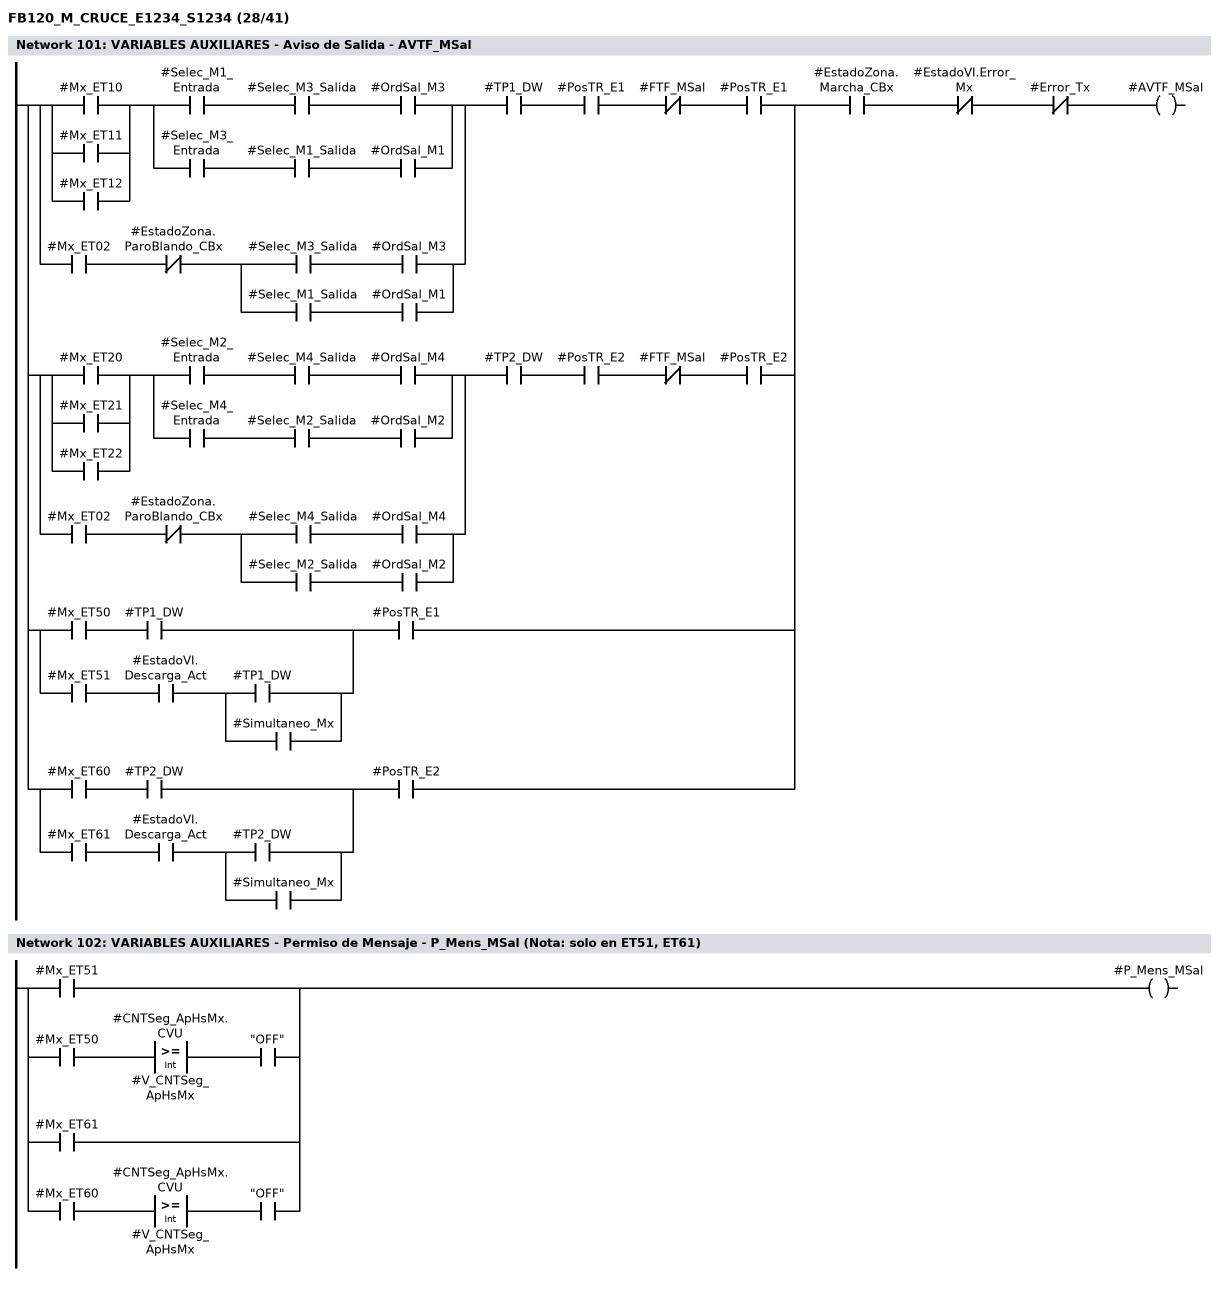
   RUNG wire#powerrail
      Contact( #Mx_ET10 )
      wire#w1
      Contact( #Selec_M1_Entrada )
      Contact( #Selec_M3_Salida )
      Contact( #OrdSal_M3 )
      wire#w2
      Contact( #TP1_DW )
      Contact( #PosTR_E1 )
      I_Contact( #FTF_MSal )
      Contact( #PosTR_E1 )
      wire#w4
      Contact( #EstadoZona.Marcha_CBx )
      I_Contact( #EstadoVI.Error_Mx )
      I_Contact( #Error_Tx )
      Coil( #AVTF_MSal )
   END_RUNG
   RUNG wire#powerrail
      Contact( #Mx_ET11 )
   END_RUNG wire#w1
   RUNG wire#powerrail
      Contact( #Mx_ET12 )
   END_RUNG wire#w1
   RUNG wire#w1
      Contact( #Selec_M3_Entrada )
      Contact( #Selec_M1_Salida )
      Contact( #OrdSal_M1 )
   END_RUNG wire#w2
   RUNG wire#powerrail
      Contact( #Mx_ET02 )
      I_Contact( #EstadoZona.ParoBlando_CBx )
      wire#w3
      Contact( #Selec_M3_Salida )
      Contact( #OrdSal_M3 )
   END_RUNG wire#w2
   RUNG wire#w3
      Contact( #Selec_M1_Salida )
      Contact( #OrdSal_M1 )
   END_RUNG wire#w2
   RUNG wire#powerrail
      Contact( #Mx_ET20 )
      wire#w5
      Contact( #Selec_M2_Entrada )
      Contact( #Selec_M4_Salida )
      Contact( #OrdSal_M4 )
      wire#w6
      Contact( #TP2_DW )
      Contact( #PosTR_E2 )
      I_Contact( #FTF_MSal )
      Contact( #PosTR_E2 )
   END_RUNG wire#w4
   RUNG wire#powerrail
      Contact( #Mx_ET21 )
   END_RUNG wire#w5
   RUNG wire#powerrail
      Contact( #Mx_ET22 )
   END_RUNG wire#w5
   RUNG wire#w5
      Contact( #Selec_M4_Entrada )
      Contact( #Selec_M2_Salida )
      Contact( #OrdSal_M2 )
   END_RUNG wire#w6
   RUNG wire#powerrail
      Contact( #Mx_ET02 )
      I_Contact( #EstadoZona.ParoBlando_CBx )
      wire#w7
      Contact( #Selec_M4_Salida )
      Contact( #OrdSal_M4 )
   END_RUNG wire#w6
   RUNG wire#w7
      Contact( #Selec_M2_Salida )
      Contact( #OrdSal_M2 )
   END_RUNG wire#w6
   RUNG wire#powerrail
      Contact( #Mx_ET50 )
      Contact( #TP1_DW )
      wire#w8
      Contact( #PosTR_E1 )
   END_RUNG wire#w4
   RUNG wire#powerrail
      Contact( #Mx_ET51 )
      Contact( #EstadoVI.Descarga_Act )
      wire#w9
      Contact( #TP1_DW )
   END_RUNG wire#w8
   RUNG wire#w9
      Contact( #Simultaneo_Mx )
   END_RUNG wire#w8
   RUNG wire#powerrail
      Contact( #Mx_ET60 )
      Contact( #TP2_DW )
      wire#w10
      Contact( #PosTR_E2 )
   END_RUNG wire#w4
   RUNG wire#powerrail
      Contact( #Mx_ET61 )
      Contact( #EstadoVI.Descarga_Act )
      wire#w11
      Contact( #TP2_DW )
   END_RUNG wire#w10
   RUNG wire#w11
      Contact( #Simultaneo_Mx )
   END_RUNG wire#w10
   // the same network as SCL:
   #AVTF_MSal := (((((#Mx_ET10 OR #Mx_ET11 OR #Mx_ET12) AND ((#Selec_M1_Entrada AND #Selec_M3_Salida AND #OrdSal_M3) OR (#Selec_M3_Entrada AND #Selec_M1_Salida AND #OrdSal_M1))) OR (#Mx_ET02 AND NOT #EstadoZona.ParoBlando_CBx AND ((#Selec_M3_Salida AND #OrdSal_M3) OR (#Selec_M1_Salida AND #OrdSal_M1)))) AND #TP1_DW AND #PosTR_E1 AND NOT #FTF_MSal AND #PosTR_E1) OR ((((#Mx_ET20 OR #Mx_ET21 OR #Mx_ET22) AND ((#Selec_M2_Entrada AND #Selec_M4_Salida AND #OrdSal_M4) OR (#Selec_M4_Entrada AND #Selec_M2_Salida AND #OrdSal_M2))) OR (#Mx_ET02 AND NOT #EstadoZona.ParoBlando_CBx AND ((#Selec_M4_Salida AND #OrdSal_M4) OR (#Selec_M2_Salida AND #OrdSal_M2)))) AND #TP2_DW AND #PosTR_E2 AND NOT #FTF_MSal AND #PosTR_E2) OR (((#Mx_ET50 AND #TP1_DW) OR (#Mx_ET51 AND #EstadoVI.Descarga_Act AND (#TP1_DW OR #Simultaneo_Mx))) AND #PosTR_E1) OR (((#Mx_ET60 AND #TP2_DW) OR (#Mx_ET61 AND #EstadoVI.Descarga_Act AND (#TP2_DW OR #Simultaneo_Mx))) AND #PosTR_E2)) AND #EstadoZona.Marcha_CBx AND NOT #EstadoVI.Error_Mx AND NOT #Error_Tx;
END_REGION

REGION Network 102: VARIABLES AUXILIARES - Permiso de Mensaje - P_Mens_MSal (Nota: solo en ET51, ET61)
   RUNG wire#powerrail
      Contact( #Mx_ET51 )
      wire#w1
      Coil( #P_Mens_MSal )
   END_RUNG
   RUNG wire#powerrail
      Contact( #Mx_ET50 )
      { S7_Templates := "SrcType := Int" } GE_Contact(in1 := #CNTSeg_ApHsMx.CVU, in2 := #V_CNTSeg_ApHsMx)
      Contact( "OFF" )
   END_RUNG wire#w1
   RUNG wire#powerrail
      Contact( #Mx_ET61 )
   END_RUNG wire#w1
   RUNG wire#powerrail
      Contact( #Mx_ET60 )
      { S7_Templates := "SrcType := Int" } GE_Contact(in1 := #CNTSeg_ApHsMx.CVU, in2 := #V_CNTSeg_ApHsMx)
      Contact( "OFF" )
   END_RUNG wire#w1
   // the same network as SCL:
   #P_Mens_MSal := #Mx_ET51 OR (#Mx_ET50 AND (#CNTSeg_ApHsMx.CVU >= #V_CNTSeg_ApHsMx) AND "OFF") OR #Mx_ET61 OR (#Mx_ET60 AND (#CNTSeg_ApHsMx.CVU >= #V_CNTSeg_ApHsMx) AND "OFF");
END_REGION

REGION Network 103: MULTIPLEXADO FINAL SEÑALES DE ENTRADA DE CARGA - PTF_MEnt
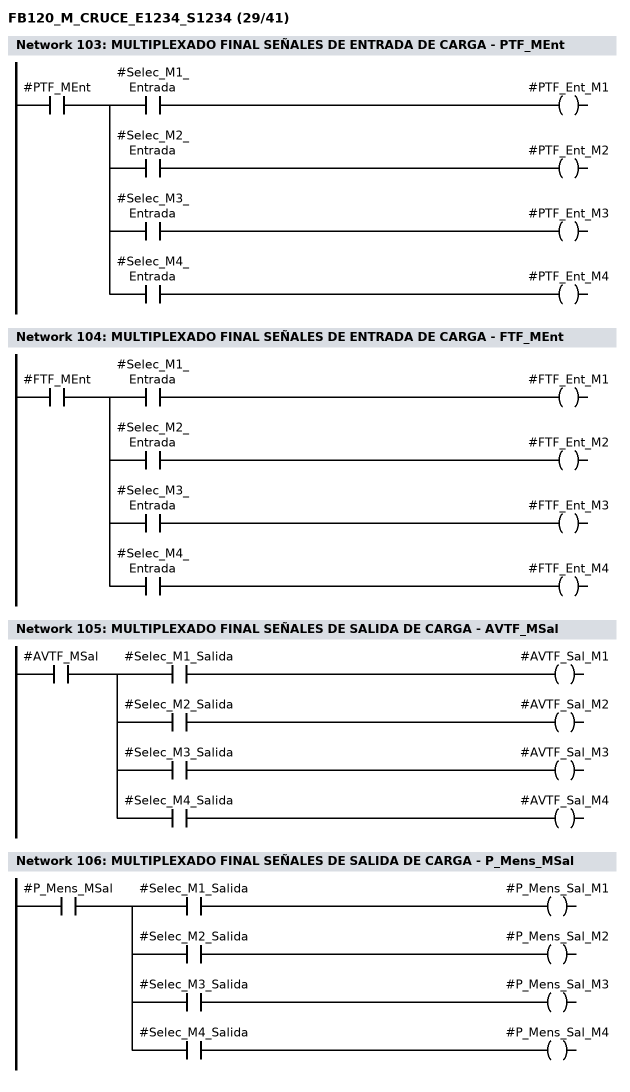
   RUNG wire#powerrail
      Contact( #PTF_MEnt )
      wire#w1
      Contact( #Selec_M1_Entrada )
      Coil( #PTF_Ent_M1 )
   END_RUNG
   RUNG wire#w1
      Contact( #Selec_M2_Entrada )
      Coil( #PTF_Ent_M2 )
   END_RUNG
   RUNG wire#w1
      Contact( #Selec_M3_Entrada )
      Coil( #PTF_Ent_M3 )
   END_RUNG
   RUNG wire#w1
      Contact( #Selec_M4_Entrada )
      Coil( #PTF_Ent_M4 )
   END_RUNG
   // the same network as SCL:
   #PTF_Ent_M1 := #PTF_MEnt AND #Selec_M1_Entrada;
   #PTF_Ent_M2 := #PTF_MEnt AND #Selec_M2_Entrada;
   #PTF_Ent_M3 := #PTF_MEnt AND #Selec_M3_Entrada;
   #PTF_Ent_M4 := #PTF_MEnt AND #Selec_M4_Entrada;
END_REGION

REGION Network 104: MULTIPLEXADO FINAL SEÑALES DE ENTRADA DE CARGA - FTF_MEnt
   RUNG wire#powerrail
      Contact( #FTF_MEnt )
      wire#w1
      Contact( #Selec_M1_Entrada )
      Coil( #FTF_Ent_M1 )
   END_RUNG
   RUNG wire#w1
      Contact( #Selec_M2_Entrada )
      Coil( #FTF_Ent_M2 )
   END_RUNG
   RUNG wire#w1
      Contact( #Selec_M3_Entrada )
      Coil( #FTF_Ent_M3 )
   END_RUNG
   RUNG wire#w1
      Contact( #Selec_M4_Entrada )
      Coil( #FTF_Ent_M4 )
   END_RUNG
   // the same network as SCL:
   #FTF_Ent_M1 := #FTF_MEnt AND #Selec_M1_Entrada;
   #FTF_Ent_M2 := #FTF_MEnt AND #Selec_M2_Entrada;
   #FTF_Ent_M3 := #FTF_MEnt AND #Selec_M3_Entrada;
   #FTF_Ent_M4 := #FTF_MEnt AND #Selec_M4_Entrada;
END_REGION

REGION Network 105: MULTIPLEXADO FINAL SEÑALES DE SALIDA DE CARGA - AVTF_MSal
   RUNG wire#powerrail
      Contact( #AVTF_MSal )
      wire#w1
      Contact( #Selec_M1_Salida )
      Coil( #AVTF_Sal_M1 )
   END_RUNG
   RUNG wire#w1
      Contact( #Selec_M2_Salida )
      Coil( #AVTF_Sal_M2 )
   END_RUNG
   RUNG wire#w1
      Contact( #Selec_M3_Salida )
      Coil( #AVTF_Sal_M3 )
   END_RUNG
   RUNG wire#w1
      Contact( #Selec_M4_Salida )
      Coil( #AVTF_Sal_M4 )
   END_RUNG
   // the same network as SCL:
   #AVTF_Sal_M1 := #AVTF_MSal AND #Selec_M1_Salida;
   #AVTF_Sal_M2 := #AVTF_MSal AND #Selec_M2_Salida;
   #AVTF_Sal_M3 := #AVTF_MSal AND #Selec_M3_Salida;
   #AVTF_Sal_M4 := #AVTF_MSal AND #Selec_M4_Salida;
END_REGION

REGION Network 106: MULTIPLEXADO FINAL SEÑALES DE SALIDA DE CARGA - P_Mens_MSal
   RUNG wire#powerrail
      Contact( #P_Mens_MSal )
      wire#w1
      Contact( #Selec_M1_Salida )
      Coil( #P_Mens_Sal_M1 )
   END_RUNG
   RUNG wire#w1
      Contact( #Selec_M2_Salida )
      Coil( #P_Mens_Sal_M2 )
   END_RUNG
   RUNG wire#w1
      Contact( #Selec_M3_Salida )
      Coil( #P_Mens_Sal_M3 )
   END_RUNG
   RUNG wire#w1
      Contact( #Selec_M4_Salida )
      Coil( #P_Mens_Sal_M4 )
   END_RUNG
   // the same network as SCL:
   #P_Mens_Sal_M1 := #P_Mens_MSal AND #Selec_M1_Salida;
   #P_Mens_Sal_M2 := #P_Mens_MSal AND #Selec_M2_Salida;
   #P_Mens_Sal_M3 := #P_Mens_MSal AND #Selec_M3_Salida;
   #P_Mens_Sal_M4 := #P_Mens_MSal AND #Selec_M4_Salida;
END_REGION

REGION Network 107: CONTADOR DE SIMULTANEO
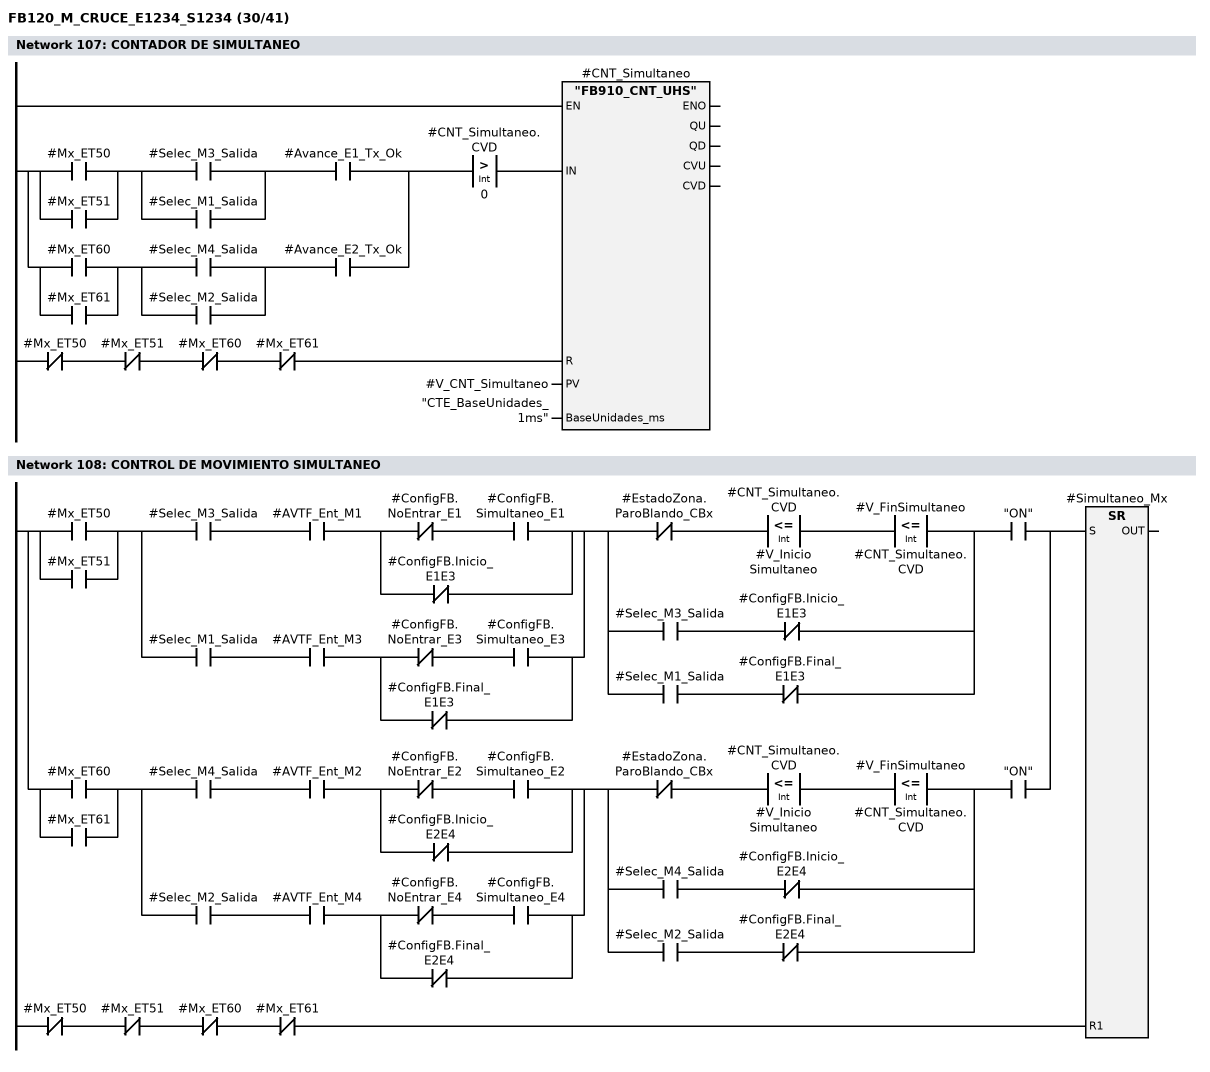
   RUNG wire#powerrail
      #CNT_Simultaneo(IN := wire#w6, R := wire#w7, PV := #V_CNT_Simultaneo, BaseUnidades_ms := "CTE_BaseUnidades_1ms", QU =>, QD =>, CVU =>, CVD =>)
   END_RUNG
   RUNG wire#powerrail
      Contact( #Mx_ET50 )
      wire#w1
      Contact( #Selec_M3_Salida )
      wire#w2
      Contact( #Avance_E1_Tx_Ok )
      wire#w3
      { S7_Templates := "SrcType := Int" } GT_Contact(in1 := #CNT_Simultaneo.CVD, in2 := 0)
   END_RUNG wire#w6
   RUNG wire#powerrail
      Contact( #Mx_ET51 )
   END_RUNG wire#w1
   RUNG wire#w1
      Contact( #Selec_M1_Salida )
   END_RUNG wire#w2
   RUNG wire#powerrail
      Contact( #Mx_ET60 )
      wire#w4
      Contact( #Selec_M4_Salida )
      wire#w5
      Contact( #Avance_E2_Tx_Ok )
   END_RUNG wire#w3
   RUNG wire#powerrail
      Contact( #Mx_ET61 )
   END_RUNG wire#w4
   RUNG wire#w4
      Contact( #Selec_M2_Salida )
   END_RUNG wire#w5
   RUNG wire#powerrail
      I_Contact( #Mx_ET50 )
      I_Contact( #Mx_ET51 )
      I_Contact( #Mx_ET60 )
      I_Contact( #Mx_ET61 )
   END_RUNG wire#w7
   // the same network as SCL:
   #CNT_Simultaneo(IN := (((#Mx_ET50 OR #Mx_ET51) AND (#Selec_M3_Salida OR #Selec_M1_Salida) AND #Avance_E1_Tx_Ok) OR ((#Mx_ET60 OR #Mx_ET61) AND (#Selec_M4_Salida OR #Selec_M2_Salida) AND #Avance_E2_Tx_Ok)) AND (#CNT_Simultaneo.CVD > 0),   // "FB910_CNT_UHS"
                   R := NOT #Mx_ET50 AND NOT #Mx_ET51 AND NOT #Mx_ET60 AND NOT #Mx_ET61,
                   PV := #V_CNT_Simultaneo,
                   BaseUnidades_ms := "CTE_BaseUnidades_1ms");
END_REGION

REGION Network 108: CONTROL DE MOVIMIENTO SIMULTANEO
   RUNG wire#powerrail
      Contact( #Mx_ET50 )
      wire#w1
      Contact( #Selec_M3_Salida )
      Contact( #AVTF_Ent_M1 )
      wire#w2
      I_Contact( #ConfigFB.NoEntrar_E1 )
      Contact( #ConfigFB.Simultaneo_E1 )
      wire#w3
      I_Contact( #EstadoZona.ParoBlando_CBx )
      { S7_Templates := "SrcType := Int" } LE_Contact(in1 := #CNT_Simultaneo.CVD, in2 := #V_InicioSimultaneo)
      { S7_Templates := "SrcType := Int" } LE_Contact(in1 := #V_FinSimultaneo, in2 := #CNT_Simultaneo.CVD)
      wire#w5
      Contact( "ON" )
      wire#w6
      S_SR(operand := #Simultaneo_Mx, r1 := wire#w12)
   END_RUNG
   RUNG wire#powerrail
      Contact( #Mx_ET51 )
   END_RUNG wire#w1
   RUNG wire#w2
      I_Contact( #ConfigFB.Inicio_E1E3 )
   END_RUNG wire#w3
   RUNG wire#w1
      Contact( #Selec_M1_Salida )
      Contact( #AVTF_Ent_M3 )
      wire#w4
      I_Contact( #ConfigFB.NoEntrar_E3 )
      Contact( #ConfigFB.Simultaneo_E3 )
   END_RUNG wire#w3
   RUNG wire#w4
      I_Contact( #ConfigFB.Final_E1E3 )
   END_RUNG wire#w3
   RUNG wire#w3
      Contact( #Selec_M3_Salida )
      I_Contact( #ConfigFB.Inicio_E1E3 )
   END_RUNG wire#w5
   RUNG wire#w3
      Contact( #Selec_M1_Salida )
      I_Contact( #ConfigFB.Final_E1E3 )
   END_RUNG wire#w5
   RUNG wire#powerrail
      Contact( #Mx_ET60 )
      wire#w7
      Contact( #Selec_M4_Salida )
      Contact( #AVTF_Ent_M2 )
      wire#w8
      I_Contact( #ConfigFB.NoEntrar_E2 )
      Contact( #ConfigFB.Simultaneo_E2 )
      wire#w9
      I_Contact( #EstadoZona.ParoBlando_CBx )
      { S7_Templates := "SrcType := Int" } LE_Contact(in1 := #CNT_Simultaneo.CVD, in2 := #V_InicioSimultaneo)
      { S7_Templates := "SrcType := Int" } LE_Contact(in1 := #V_FinSimultaneo, in2 := #CNT_Simultaneo.CVD)
      wire#w11
      Contact( "ON" )
   END_RUNG wire#w6
   RUNG wire#powerrail
      Contact( #Mx_ET61 )
   END_RUNG wire#w7
   RUNG wire#w8
      I_Contact( #ConfigFB.Inicio_E2E4 )
   END_RUNG wire#w9
   RUNG wire#w7
      Contact( #Selec_M2_Salida )
      Contact( #AVTF_Ent_M4 )
      wire#w10
      I_Contact( #ConfigFB.NoEntrar_E4 )
      Contact( #ConfigFB.Simultaneo_E4 )
   END_RUNG wire#w9
   RUNG wire#w10
      I_Contact( #ConfigFB.Final_E2E4 )
   END_RUNG wire#w9
   RUNG wire#w9
      Contact( #Selec_M4_Salida )
      I_Contact( #ConfigFB.Inicio_E2E4 )
   END_RUNG wire#w11
   RUNG wire#w9
      Contact( #Selec_M2_Salida )
      I_Contact( #ConfigFB.Final_E2E4 )
   END_RUNG wire#w11
   RUNG wire#powerrail
      I_Contact( #Mx_ET50 )
      I_Contact( #Mx_ET51 )
      I_Contact( #Mx_ET60 )
      I_Contact( #Mx_ET61 )
   END_RUNG wire#w12
   // the same network as SCL:
   IF ((#Mx_ET50 OR #Mx_ET51) AND ((#Selec_M3_Salida AND #AVTF_Ent_M1 AND ((NOT #ConfigFB.NoEntrar_E1 AND #ConfigFB.Simultaneo_E1) OR NOT #ConfigFB.Inicio_E1E3)) OR (#Selec_M1_Salida AND #AVTF_Ent_M3 AND ((NOT #ConfigFB.NoEntrar_E3 AND #ConfigFB.Simultaneo_E3) OR NOT #ConfigFB.Final_E1E3))) AND ((NOT #EstadoZona.ParoBlando_CBx AND (#CNT_Simultaneo.CVD <= #V_InicioSimultaneo) AND (#V_FinSimultaneo <= #CNT_Simultaneo.CVD)) OR (#Selec_M3_Salida AND NOT #ConfigFB.Inicio_E1E3) OR (#Selec_M1_Salida AND NOT #ConfigFB.Final_E1E3)) AND "ON") OR ((#Mx_ET60 OR #Mx_ET61) AND ((#Selec_M4_Salida AND #AVTF_Ent_M2 AND ((NOT #ConfigFB.NoEntrar_E2 AND #ConfigFB.Simultaneo_E2) OR NOT #ConfigFB.Inicio_E2E4)) OR (#Selec_M2_Salida AND #AVTF_Ent_M4 AND ((NOT #ConfigFB.NoEntrar_E4 AND #ConfigFB.Simultaneo_E4) OR NOT #ConfigFB.Final_E2E4))) AND ((NOT #EstadoZona.ParoBlando_CBx AND (#CNT_Simultaneo.CVD <= #V_InicioSimultaneo) AND (#V_FinSimultaneo <= #CNT_Simultaneo.CVD)) OR (#Selec_M4_Salida AND NOT #ConfigFB.Inicio_E2E4) OR (#Selec_M2_Salida AND NOT #ConfigFB.Final_E2E4)) AND "ON") THEN
       #Simultaneo_Mx := TRUE;   // SR flip-flop
   END_IF;
   IF NOT #Mx_ET50 AND NOT #Mx_ET51 AND NOT #Mx_ET60 AND NOT #Mx_ET61 THEN #Simultaneo_Mx := FALSE; END_IF;
END_REGION

REGION Network 109: MENSAJES - PRESENCIA
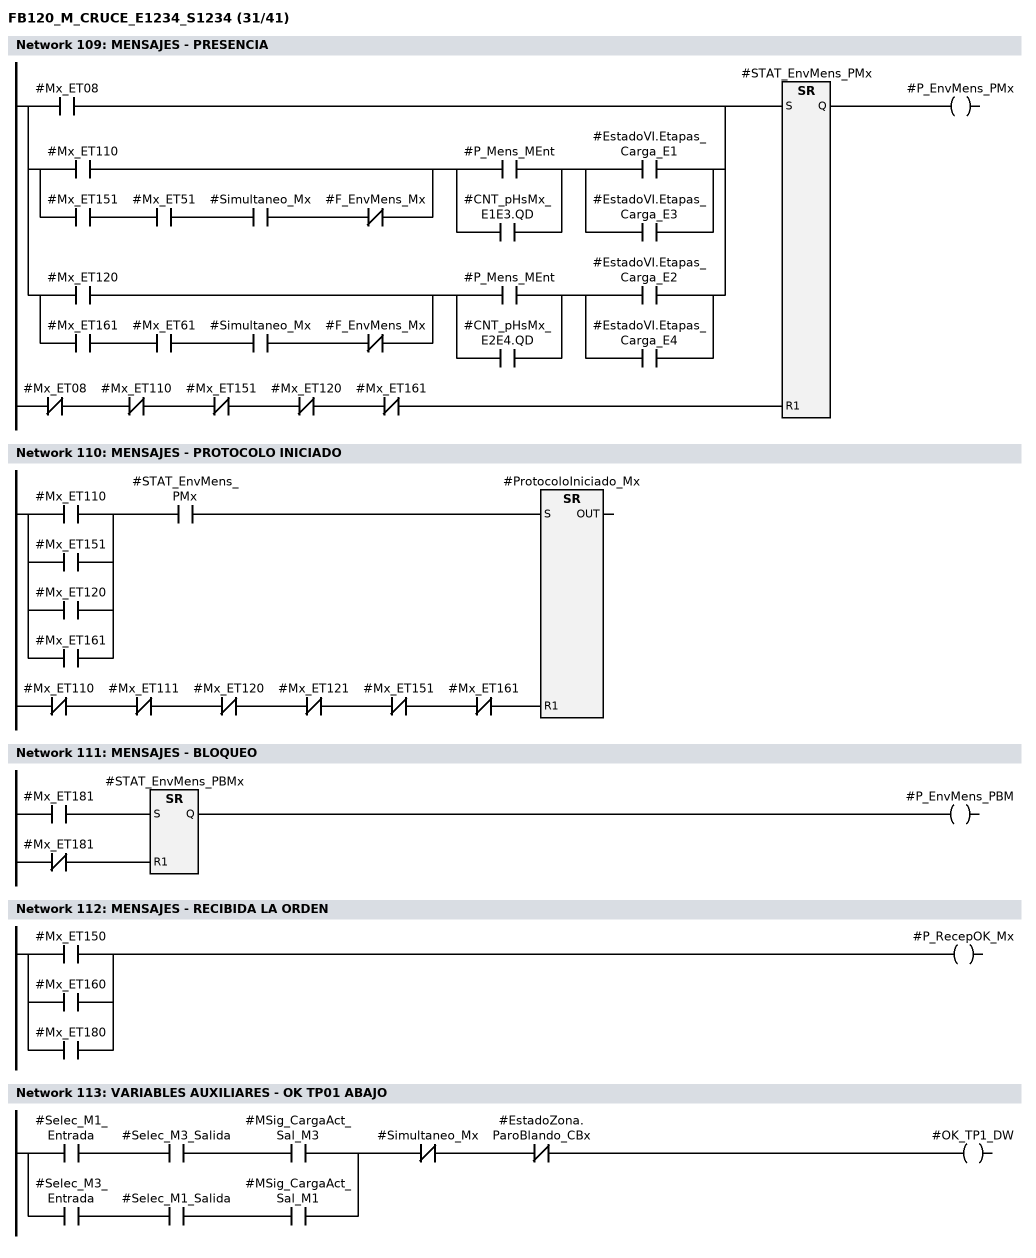
   RUNG wire#powerrail
      Contact( #Mx_ET08 )
      wire#w1
      S_SR(operand := #STAT_EnvMens_PMx, r1 := wire#w6)
      Coil( #P_EnvMens_PMx )
   END_RUNG
   RUNG wire#powerrail
      Contact( #Mx_ET110 )
      wire#w2
      Contact( #P_Mens_MEnt )
      wire#w3
      Contact( #EstadoVI.Etapas_Carga_E1 )
   END_RUNG wire#w1
   RUNG wire#powerrail
      Contact( #Mx_ET151 )
      Contact( #Mx_ET51 )
      Contact( #Simultaneo_Mx )
      I_Contact( #F_EnvMens_Mx )
   END_RUNG wire#w2
   RUNG wire#w2
      Contact( #CNT_pHsMx_E1E3.QD )
   END_RUNG wire#w3
   RUNG wire#w3
      Contact( #EstadoVI.Etapas_Carga_E3 )
   END_RUNG wire#w1
   RUNG wire#powerrail
      Contact( #Mx_ET120 )
      wire#w4
      Contact( #P_Mens_MEnt )
      wire#w5
      Contact( #EstadoVI.Etapas_Carga_E2 )
   END_RUNG wire#w1
   RUNG wire#powerrail
      Contact( #Mx_ET161 )
      Contact( #Mx_ET61 )
      Contact( #Simultaneo_Mx )
      I_Contact( #F_EnvMens_Mx )
   END_RUNG wire#w4
   RUNG wire#w4
      Contact( #CNT_pHsMx_E2E4.QD )
   END_RUNG wire#w5
   RUNG wire#w5
      Contact( #EstadoVI.Etapas_Carga_E4 )
   END_RUNG wire#w1
   RUNG wire#powerrail
      I_Contact( #Mx_ET08 )
      I_Contact( #Mx_ET110 )
      I_Contact( #Mx_ET151 )
      I_Contact( #Mx_ET120 )
      I_Contact( #Mx_ET161 )
   END_RUNG wire#w6
   // the same network as SCL:
   IF #Mx_ET08 OR ((#Mx_ET110 OR (#Mx_ET151 AND #Mx_ET51 AND #Simultaneo_Mx AND NOT #F_EnvMens_Mx)) AND (#P_Mens_MEnt OR #CNT_pHsMx_E1E3.QD) AND (#EstadoVI.Etapas_Carga_E1 OR #EstadoVI.Etapas_Carga_E3)) OR ((#Mx_ET120 OR (#Mx_ET161 AND #Mx_ET61 AND #Simultaneo_Mx AND NOT #F_EnvMens_Mx)) AND (#P_Mens_MEnt OR #CNT_pHsMx_E2E4.QD) AND (#EstadoVI.Etapas_Carga_E2 OR #EstadoVI.Etapas_Carga_E4)) THEN
       #STAT_EnvMens_PMx := TRUE;   // SR flip-flop
   END_IF;
   IF NOT #Mx_ET08 AND NOT #Mx_ET110 AND NOT #Mx_ET151 AND NOT #Mx_ET120 AND NOT #Mx_ET161 THEN
       #STAT_EnvMens_PMx := FALSE;
   END_IF;
   #P_EnvMens_PMx := #STAT_EnvMens_PMx;
END_REGION

REGION Network 110: MENSAJES - PROTOCOLO INICIADO
   RUNG wire#powerrail
      Contact( #Mx_ET110 )
      wire#w1
      Contact( #STAT_EnvMens_PMx )
      S_SR(operand := #ProtocoloIniciado_Mx, r1 := wire#w2)
   END_RUNG
   RUNG wire#powerrail
      Contact( #Mx_ET151 )
   END_RUNG wire#w1
   RUNG wire#powerrail
      Contact( #Mx_ET120 )
   END_RUNG wire#w1
   RUNG wire#powerrail
      Contact( #Mx_ET161 )
   END_RUNG wire#w1
   RUNG wire#powerrail
      I_Contact( #Mx_ET110 )
      I_Contact( #Mx_ET111 )
      I_Contact( #Mx_ET120 )
      I_Contact( #Mx_ET121 )
      I_Contact( #Mx_ET151 )
      I_Contact( #Mx_ET161 )
   END_RUNG wire#w2
   // the same network as SCL:
   IF (#Mx_ET110 OR #Mx_ET151 OR #Mx_ET120 OR #Mx_ET161) AND #STAT_EnvMens_PMx THEN
       #ProtocoloIniciado_Mx := TRUE;   // SR flip-flop
   END_IF;
   IF NOT #Mx_ET110 AND NOT #Mx_ET111 AND NOT #Mx_ET120 AND NOT #Mx_ET121 AND NOT #Mx_ET151 AND NOT #Mx_ET161 THEN
       #ProtocoloIniciado_Mx := FALSE;
   END_IF;
END_REGION

REGION Network 111: MENSAJES - BLOQUEO
   RUNG wire#powerrail
      Contact( #Mx_ET181 )
      S_SR(operand := #STAT_EnvMens_PBMx, r1 := wire#w1)
      Coil( #P_EnvMens_PBM )
   END_RUNG
   RUNG wire#powerrail
      I_Contact( #Mx_ET181 )
   END_RUNG wire#w1
   // the same network as SCL:
   IF #Mx_ET181 THEN
       #STAT_EnvMens_PBMx := TRUE;   // SR flip-flop
   END_IF;
   IF NOT #Mx_ET181 THEN #STAT_EnvMens_PBMx := FALSE; END_IF;
   #P_EnvMens_PBM := #STAT_EnvMens_PBMx;
END_REGION

REGION Network 112: MENSAJES - RECIBIDA LA ORDEN
   RUNG wire#powerrail
      Contact( #Mx_ET150 )
      wire#w1
      Coil( #P_RecepOK_Mx )
   END_RUNG
   RUNG wire#powerrail
      Contact( #Mx_ET160 )
   END_RUNG wire#w1
   RUNG wire#powerrail
      Contact( #Mx_ET180 )
   END_RUNG wire#w1
   // the same network as SCL:
   #P_RecepOK_Mx := #Mx_ET150 OR #Mx_ET160 OR #Mx_ET180;
END_REGION

REGION Network 113: VARIABLES AUXILIARES - OK TP01 ABAJO
   RUNG wire#powerrail
      Contact( #Selec_M1_Entrada )
      Contact( #Selec_M3_Salida )
      Contact( #MSig_CargaAct_Sal_M3 )
      wire#w1
      I_Contact( #Simultaneo_Mx )
      I_Contact( #EstadoZona.ParoBlando_CBx )
      Coil( #OK_TP1_DW )
   END_RUNG
   RUNG wire#powerrail
      Contact( #Selec_M3_Entrada )
      Contact( #Selec_M1_Salida )
      Contact( #MSig_CargaAct_Sal_M1 )
   END_RUNG wire#w1
   // the same network as SCL:
   #OK_TP1_DW := ((#Selec_M1_Entrada AND #Selec_M3_Salida AND #MSig_CargaAct_Sal_M3) OR (#Selec_M3_Entrada AND #Selec_M1_Salida AND #MSig_CargaAct_Sal_M1)) AND NOT #Simultaneo_Mx AND NOT #EstadoZona.ParoBlando_CBx;
END_REGION

REGION Network 114: VARIABLES AUXILIARES - OK TP02 ABAJO
   // MODIFICACION: NUEVO TOPE
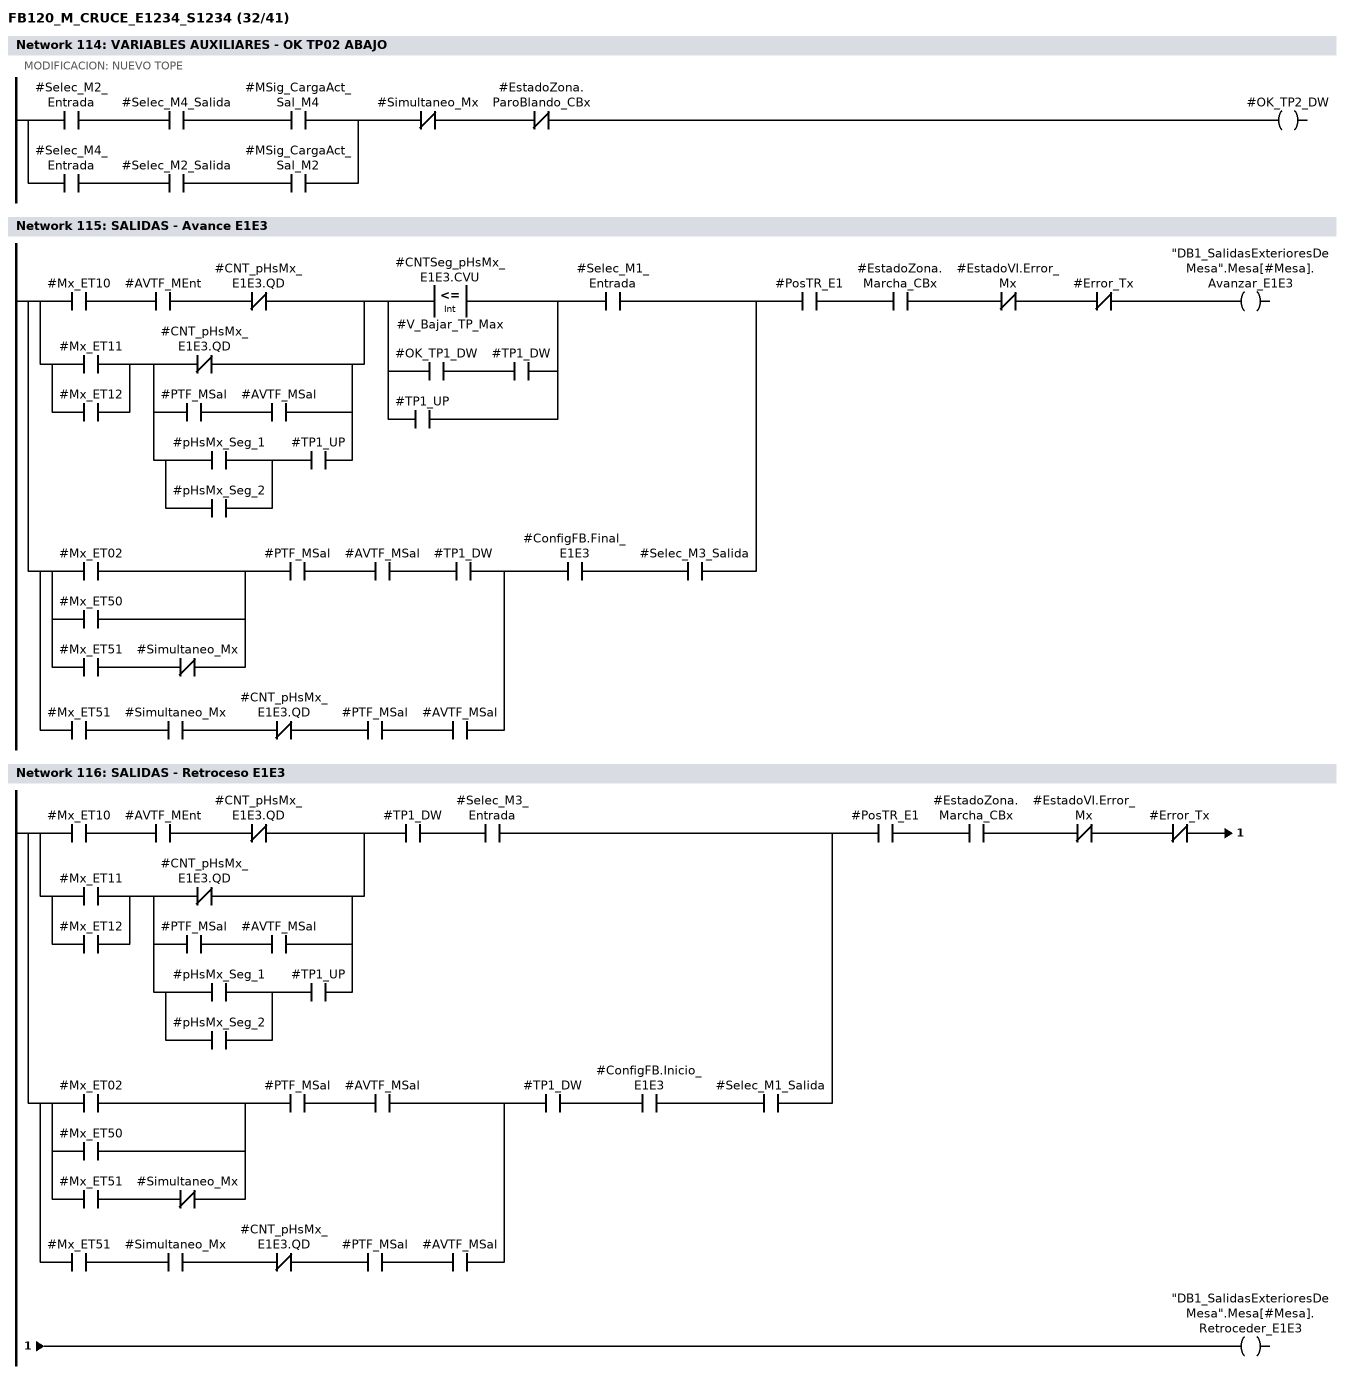
   RUNG wire#powerrail
      Contact( #Selec_M2_Entrada )
      Contact( #Selec_M4_Salida )
      Contact( #MSig_CargaAct_Sal_M4 )
      wire#w1
      I_Contact( #Simultaneo_Mx )
      I_Contact( #EstadoZona.ParoBlando_CBx )
      Coil( #OK_TP2_DW )
   END_RUNG
   RUNG wire#powerrail
      Contact( #Selec_M4_Entrada )
      Contact( #Selec_M2_Salida )
      Contact( #MSig_CargaAct_Sal_M2 )
   END_RUNG wire#w1
   // the same network as SCL:
   #OK_TP2_DW := ((#Selec_M2_Entrada AND #Selec_M4_Salida AND #MSig_CargaAct_Sal_M4) OR (#Selec_M4_Entrada AND #Selec_M2_Salida AND #MSig_CargaAct_Sal_M2)) AND NOT #Simultaneo_Mx AND NOT #EstadoZona.ParoBlando_CBx;
END_REGION

REGION Network 115: SALIDAS - Avance E1E3
   RUNG wire#powerrail
      Contact( #Mx_ET10 )
      Contact( #AVTF_MEnt )
      I_Contact( #CNT_pHsMx_E1E3.QD )
      wire#w1
      { S7_Templates := "SrcType := Int" } LE_Contact(in1 := #CNTSeg_pHsMx_E1E3.CVU, in2 := #V_Bajar_TP_Max)
      wire#w4
      Contact( #Selec_M1_Entrada )
      wire#w5
      Contact( #PosTR_E1 )
      Contact( #EstadoZona.Marcha_CBx )
      I_Contact( #EstadoVI.Error_Mx )
      I_Contact( #Error_Tx )
      Coil( "DB1_SalidasExterioresDeMesa".Mesa[#Mesa].Avanzar_E1E3 )
   END_RUNG
   RUNG wire#powerrail
      Contact( #Mx_ET11 )
      wire#w2
      I_Contact( #CNT_pHsMx_E1E3.QD )
   END_RUNG wire#w1
   RUNG wire#powerrail
      Contact( #Mx_ET12 )
   END_RUNG wire#w2
   RUNG wire#w2
      Contact( #PTF_MSal )
      Contact( #AVTF_MSal )
   END_RUNG wire#w1
   RUNG wire#w2
      Contact( #pHsMx_Seg_1 )
      wire#w3
      Contact( #TP1_UP )
   END_RUNG wire#w1
   RUNG wire#w2
      Contact( #pHsMx_Seg_2 )
   END_RUNG wire#w3
   RUNG wire#w1
      Contact( #OK_TP1_DW )
      Contact( #TP1_DW )
   END_RUNG wire#w4
   RUNG wire#w1
      Contact( #TP1_UP )
   END_RUNG wire#w4
   RUNG wire#powerrail
      Contact( #Mx_ET02 )
      wire#w6
      Contact( #PTF_MSal )
      Contact( #AVTF_MSal )
      Contact( #TP1_DW )
      wire#w7
      Contact( #ConfigFB.Final_E1E3 )
      Contact( #Selec_M3_Salida )
   END_RUNG wire#w5
   RUNG wire#powerrail
      Contact( #Mx_ET50 )
   END_RUNG wire#w6
   RUNG wire#powerrail
      Contact( #Mx_ET51 )
      I_Contact( #Simultaneo_Mx )
   END_RUNG wire#w6
   RUNG wire#powerrail
      Contact( #Mx_ET51 )
      Contact( #Simultaneo_Mx )
      I_Contact( #CNT_pHsMx_E1E3.QD )
      Contact( #PTF_MSal )
      Contact( #AVTF_MSal )
   END_RUNG wire#w7
   // the same network as SCL:
   "DB1_SalidasExterioresDeMesa".Mesa[#Mesa].Avanzar_E1E3 := ((((#Mx_ET10 AND #AVTF_MEnt AND NOT #CNT_pHsMx_E1E3.QD) OR ((#Mx_ET11 OR #Mx_ET12) AND (NOT #CNT_pHsMx_E1E3.QD OR (#PTF_MSal AND #AVTF_MSal) OR ((#pHsMx_Seg_1 OR #pHsMx_Seg_2) AND #TP1_UP)))) AND ((#CNTSeg_pHsMx_E1E3.CVU <= #V_Bajar_TP_Max) OR (#OK_TP1_DW AND #TP1_DW) OR #TP1_UP) AND #Selec_M1_Entrada) OR ((((#Mx_ET02 OR #Mx_ET50 OR (#Mx_ET51 AND NOT #Simultaneo_Mx)) AND #PTF_MSal AND #AVTF_MSal AND #TP1_DW) OR (#Mx_ET51 AND #Simultaneo_Mx AND NOT #CNT_pHsMx_E1E3.QD AND #PTF_MSal AND #AVTF_MSal)) AND #ConfigFB.Final_E1E3 AND #Selec_M3_Salida)) AND #PosTR_E1 AND #EstadoZona.Marcha_CBx AND NOT #EstadoVI.Error_Mx AND NOT #Error_Tx;
END_REGION

REGION Network 116: SALIDAS - Retroceso E1E3
   RUNG wire#powerrail
      Contact( #Mx_ET10 )
      Contact( #AVTF_MEnt )
      I_Contact( #CNT_pHsMx_E1E3.QD )
      wire#w1
      Contact( #TP1_DW )
      Contact( #Selec_M3_Entrada )
      wire#w4
      Contact( #PosTR_E1 )
      Contact( #EstadoZona.Marcha_CBx )
      I_Contact( #EstadoVI.Error_Mx )
      I_Contact( #Error_Tx )
      Coil( "DB1_SalidasExterioresDeMesa".Mesa[#Mesa].Retroceder_E1E3 )
   END_RUNG
   RUNG wire#powerrail
      Contact( #Mx_ET11 )
      wire#w2
      I_Contact( #CNT_pHsMx_E1E3.QD )
   END_RUNG wire#w1
   RUNG wire#powerrail
      Contact( #Mx_ET12 )
   END_RUNG wire#w2
   RUNG wire#w2
      Contact( #PTF_MSal )
      Contact( #AVTF_MSal )
   END_RUNG wire#w1
   RUNG wire#w2
      Contact( #pHsMx_Seg_1 )
      wire#w3
      Contact( #TP1_UP )
   END_RUNG wire#w1
   RUNG wire#w2
      Contact( #pHsMx_Seg_2 )
   END_RUNG wire#w3
   RUNG wire#powerrail
      Contact( #Mx_ET02 )
      wire#w5
      Contact( #PTF_MSal )
      Contact( #AVTF_MSal )
      wire#w6
      Contact( #TP1_DW )
      Contact( #ConfigFB.Inicio_E1E3 )
      Contact( #Selec_M1_Salida )
   END_RUNG wire#w4
   RUNG wire#powerrail
      Contact( #Mx_ET50 )
   END_RUNG wire#w5
   RUNG wire#powerrail
      Contact( #Mx_ET51 )
      I_Contact( #Simultaneo_Mx )
   END_RUNG wire#w5
   RUNG wire#powerrail
      Contact( #Mx_ET51 )
      Contact( #Simultaneo_Mx )
      I_Contact( #CNT_pHsMx_E1E3.QD )
      Contact( #PTF_MSal )
      Contact( #AVTF_MSal )
   END_RUNG wire#w6
   // the same network as SCL:
   "DB1_SalidasExterioresDeMesa".Mesa[#Mesa].Retroceder_E1E3 := ((((#Mx_ET10 AND #AVTF_MEnt AND NOT #CNT_pHsMx_E1E3.QD) OR ((#Mx_ET11 OR #Mx_ET12) AND (NOT #CNT_pHsMx_E1E3.QD OR (#PTF_MSal AND #AVTF_MSal) OR ((#pHsMx_Seg_1 OR #pHsMx_Seg_2) AND #TP1_UP)))) AND #TP1_DW AND #Selec_M3_Entrada) OR ((((#Mx_ET02 OR #Mx_ET50 OR (#Mx_ET51 AND NOT #Simultaneo_Mx)) AND #PTF_MSal AND #AVTF_MSal) OR (#Mx_ET51 AND #Simultaneo_Mx AND NOT #CNT_pHsMx_E1E3.QD AND #PTF_MSal AND #AVTF_MSal)) AND #TP1_DW AND #ConfigFB.Inicio_E1E3 AND #Selec_M1_Salida)) AND #PosTR_E1 AND #EstadoZona.Marcha_CBx AND NOT #EstadoVI.Error_Mx AND NOT #Error_Tx;
END_REGION

REGION Network 117: SALIDAS - Parar E1E3
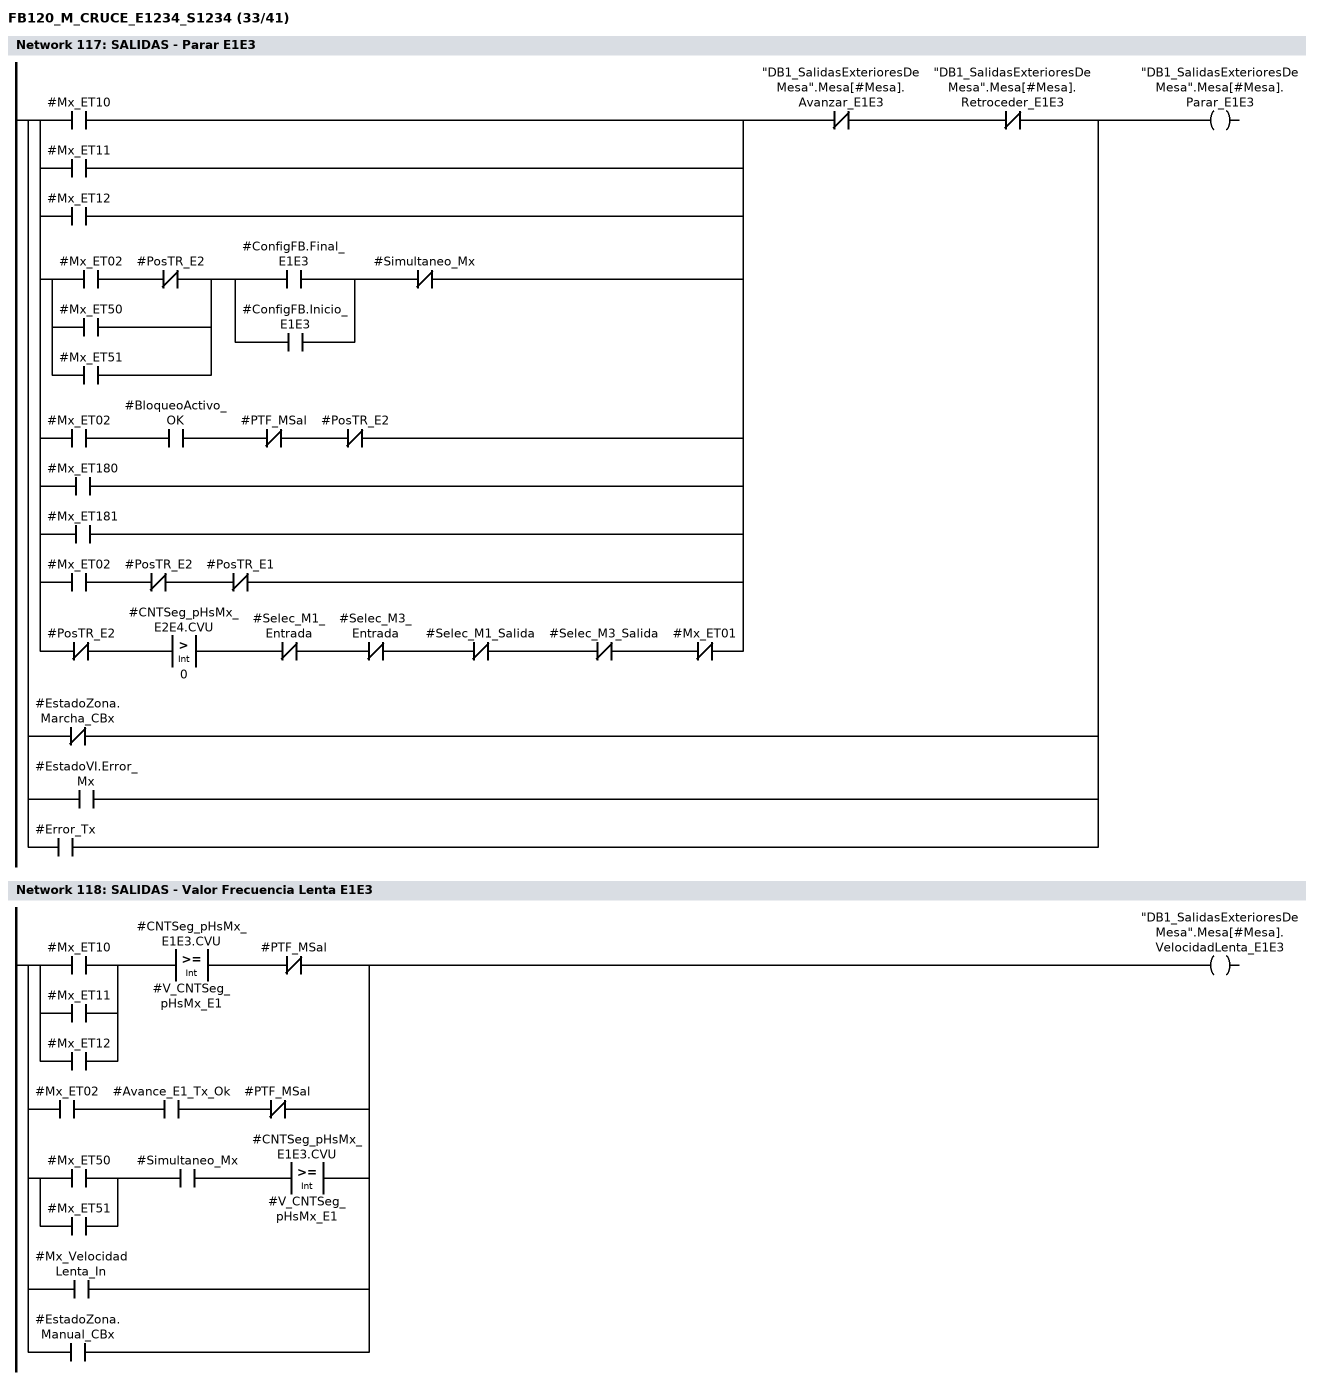
   RUNG wire#powerrail
      Contact( #Mx_ET10 )
      wire#w1
      I_Contact( "DB1_SalidasExterioresDeMesa".Mesa[#Mesa].Avanzar_E1E3 )
      I_Contact( "DB1_SalidasExterioresDeMesa".Mesa[#Mesa].Retroceder_E1E3 )
      wire#w4
      Coil( "DB1_SalidasExterioresDeMesa".Mesa[#Mesa].Parar_E1E3 )
   END_RUNG
   RUNG wire#powerrail
      Contact( #Mx_ET11 )
   END_RUNG wire#w1
   RUNG wire#powerrail
      Contact( #Mx_ET12 )
   END_RUNG wire#w1
   RUNG wire#powerrail
      Contact( #Mx_ET02 )
      I_Contact( #PosTR_E2 )
      wire#w2
      Contact( #ConfigFB.Final_E1E3 )
      wire#w3
      I_Contact( #Simultaneo_Mx )
   END_RUNG wire#w1
   RUNG wire#powerrail
      Contact( #Mx_ET50 )
   END_RUNG wire#w2
   RUNG wire#powerrail
      Contact( #Mx_ET51 )
   END_RUNG wire#w2
   RUNG wire#w2
      Contact( #ConfigFB.Inicio_E1E3 )
   END_RUNG wire#w3
   RUNG wire#powerrail
      Contact( #Mx_ET02 )
      Contact( #BloqueoActivo_OK )
      I_Contact( #PTF_MSal )
      I_Contact( #PosTR_E2 )
   END_RUNG wire#w1
   RUNG wire#powerrail
      Contact( #Mx_ET180 )
   END_RUNG wire#w1
   RUNG wire#powerrail
      Contact( #Mx_ET181 )
   END_RUNG wire#w1
   RUNG wire#powerrail
      Contact( #Mx_ET02 )
      I_Contact( #PosTR_E2 )
      I_Contact( #PosTR_E1 )
   END_RUNG wire#w1
   RUNG wire#powerrail
      I_Contact( #PosTR_E2 )
      { S7_Templates := "SrcType := Int" } GT_Contact(in1 := #CNTSeg_pHsMx_E2E4.CVU, in2 := 0)
      I_Contact( #Selec_M1_Entrada )
      I_Contact( #Selec_M3_Entrada )
      I_Contact( #Selec_M1_Salida )
      I_Contact( #Selec_M3_Salida )
      I_Contact( #Mx_ET01 )
   END_RUNG wire#w1
   RUNG wire#powerrail
      I_Contact( #EstadoZona.Marcha_CBx )
   END_RUNG wire#w4
   RUNG wire#powerrail
      Contact( #EstadoVI.Error_Mx )
   END_RUNG wire#w4
   RUNG wire#powerrail
      Contact( #Error_Tx )
   END_RUNG wire#w4
   // the same network as SCL:
   "DB1_SalidasExterioresDeMesa".Mesa[#Mesa].Parar_E1E3 := ((#Mx_ET10 OR #Mx_ET11 OR #Mx_ET12 OR (((#Mx_ET02 AND NOT #PosTR_E2) OR #Mx_ET50 OR #Mx_ET51) AND (#ConfigFB.Final_E1E3 OR #ConfigFB.Inicio_E1E3) AND NOT #Simultaneo_Mx) OR (#Mx_ET02 AND #BloqueoActivo_OK AND NOT #PTF_MSal AND NOT #PosTR_E2) OR #Mx_ET180 OR #Mx_ET181 OR (#Mx_ET02 AND NOT #PosTR_E2 AND NOT #PosTR_E1) OR (NOT #PosTR_E2 AND (#CNTSeg_pHsMx_E2E4.CVU > 0) AND NOT #Selec_M1_Entrada AND NOT #Selec_M3_Entrada AND NOT #Selec_M1_Salida AND NOT #Selec_M3_Salida AND NOT #Mx_ET01)) AND NOT "DB1_SalidasExterioresDeMesa".Mesa[#Mesa].Avanzar_E1E3 AND NOT "DB1_SalidasExterioresDeMesa".Mesa[#Mesa].Retroceder_E1E3) OR NOT #EstadoZona.Marcha_CBx OR #EstadoVI.Error_Mx OR #Error_Tx;
END_REGION

REGION Network 118: SALIDAS - Valor Frecuencia Lenta E1E3
   RUNG wire#powerrail
      Contact( #Mx_ET10 )
      wire#w1
      { S7_Templates := "SrcType := Int" } GE_Contact(in1 := #CNTSeg_pHsMx_E1E3.CVU, in2 := #V_CNTSeg_pHsMx_E1)
      I_Contact( #PTF_MSal )
      wire#w2
      Coil( "DB1_SalidasExterioresDeMesa".Mesa[#Mesa].VelocidadLenta_E1E3 )
   END_RUNG
   RUNG wire#powerrail
      Contact( #Mx_ET11 )
   END_RUNG wire#w1
   RUNG wire#powerrail
      Contact( #Mx_ET12 )
   END_RUNG wire#w1
   RUNG wire#powerrail
      Contact( #Mx_ET02 )
      Contact( #Avance_E1_Tx_Ok )
      I_Contact( #PTF_MSal )
   END_RUNG wire#w2
   RUNG wire#powerrail
      Contact( #Mx_ET50 )
      wire#w3
      Contact( #Simultaneo_Mx )
      { S7_Templates := "SrcType := Int" } GE_Contact(in1 := #CNTSeg_pHsMx_E1E3.CVU, in2 := #V_CNTSeg_pHsMx_E1)
   END_RUNG wire#w2
   RUNG wire#powerrail
      Contact( #Mx_ET51 )
   END_RUNG wire#w3
   RUNG wire#powerrail
      Contact( #Mx_VelocidadLenta_In )
   END_RUNG wire#w2
   RUNG wire#powerrail
      Contact( #EstadoZona.Manual_CBx )
   END_RUNG wire#w2
   // the same network as SCL:
   "DB1_SalidasExterioresDeMesa".Mesa[#Mesa].VelocidadLenta_E1E3 := ((#Mx_ET10 OR #Mx_ET11 OR #Mx_ET12) AND (#CNTSeg_pHsMx_E1E3.CVU >= #V_CNTSeg_pHsMx_E1) AND NOT #PTF_MSal) OR (#Mx_ET02 AND #Avance_E1_Tx_Ok AND NOT #PTF_MSal) OR ((#Mx_ET50 OR #Mx_ET51) AND #Simultaneo_Mx AND (#CNTSeg_pHsMx_E1E3.CVU >= #V_CNTSeg_pHsMx_E1)) OR #Mx_VelocidadLenta_In OR #EstadoZona.Manual_CBx;
END_REGION

REGION Network 119: SALIDAS - Avance E2E4
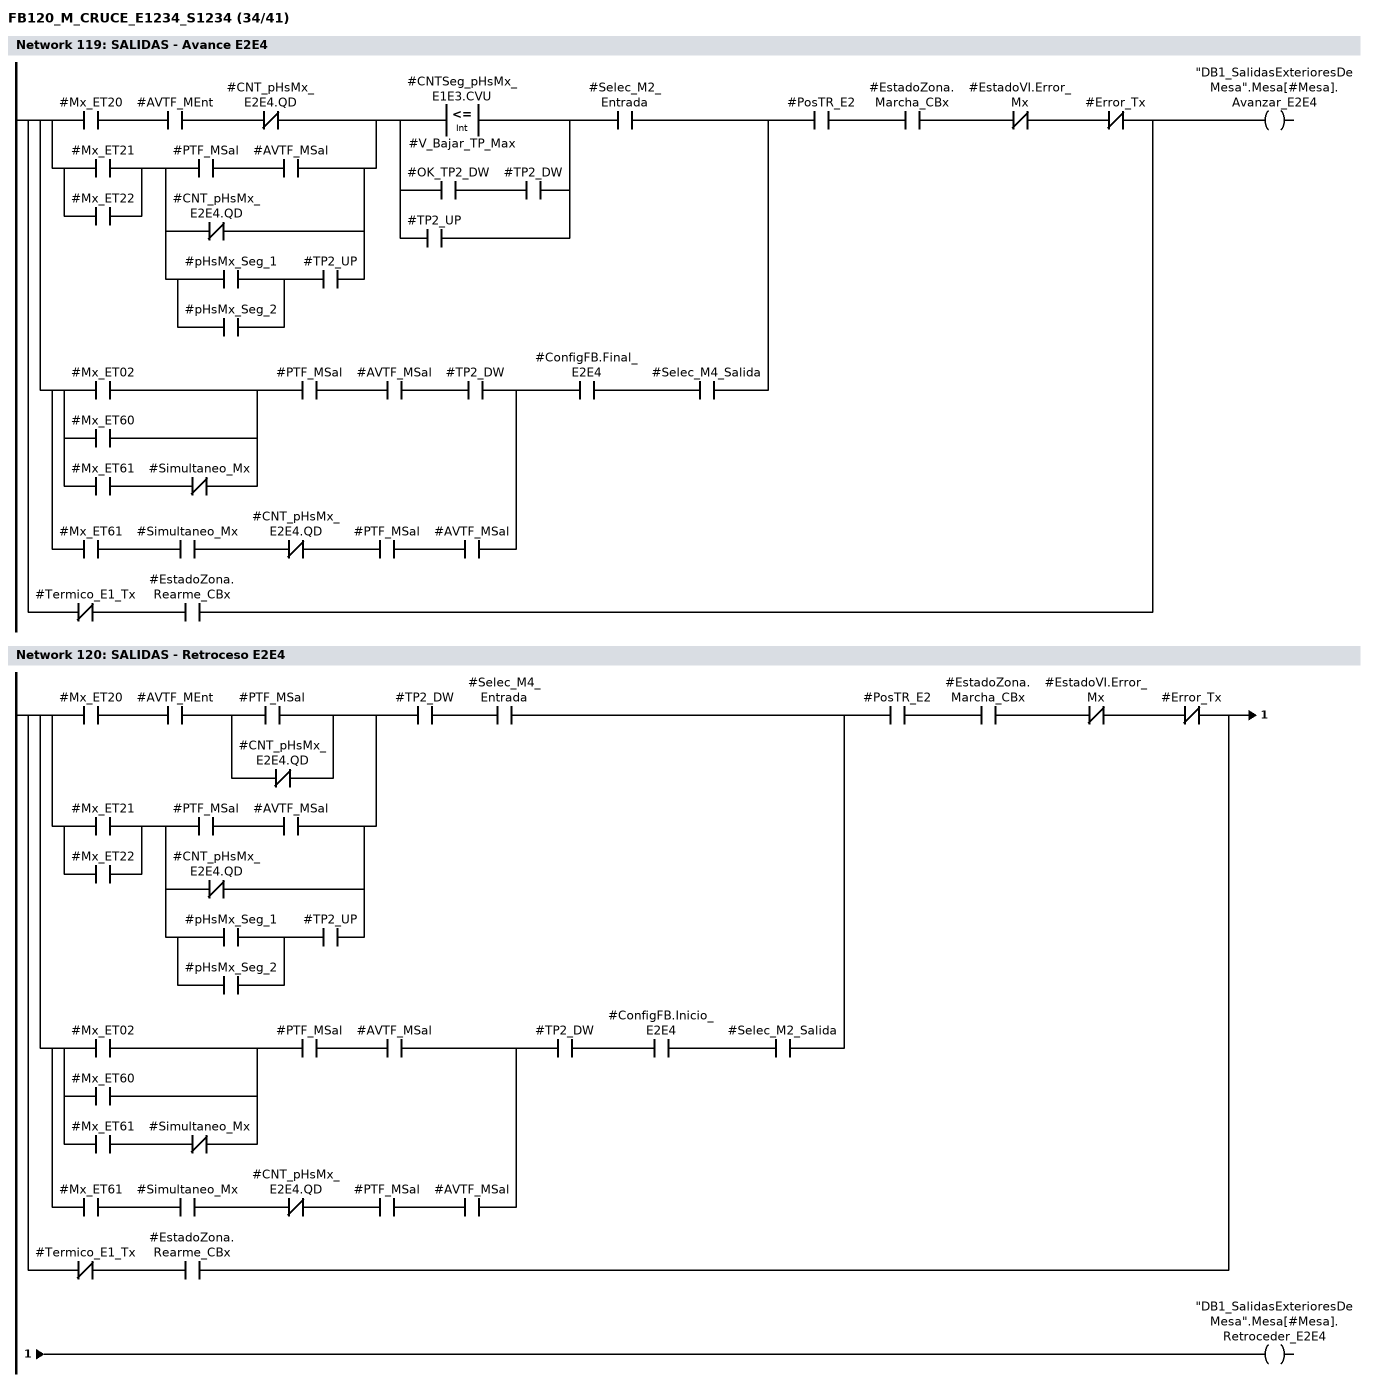
   RUNG wire#powerrail
      Contact( #Mx_ET20 )
      Contact( #AVTF_MEnt )
      I_Contact( #CNT_pHsMx_E2E4.QD )
      wire#w1
      { S7_Templates := "SrcType := Int" } LE_Contact(in1 := #CNTSeg_pHsMx_E1E3.CVU, in2 := #V_Bajar_TP_Max)
      wire#w4
      Contact( #Selec_M2_Entrada )
      wire#w5
      Contact( #PosTR_E2 )
      Contact( #EstadoZona.Marcha_CBx )
      I_Contact( #EstadoVI.Error_Mx )
      I_Contact( #Error_Tx )
      wire#w8
      Coil( "DB1_SalidasExterioresDeMesa".Mesa[#Mesa].Avanzar_E2E4 )
   END_RUNG
   RUNG wire#powerrail
      Contact( #Mx_ET21 )
      wire#w2
      Contact( #PTF_MSal )
      Contact( #AVTF_MSal )
   END_RUNG wire#w1
   RUNG wire#powerrail
      Contact( #Mx_ET22 )
   END_RUNG wire#w2
   RUNG wire#w2
      I_Contact( #CNT_pHsMx_E2E4.QD )
   END_RUNG wire#w1
   RUNG wire#w2
      Contact( #pHsMx_Seg_1 )
      wire#w3
      Contact( #TP2_UP )
   END_RUNG wire#w1
   RUNG wire#w2
      Contact( #pHsMx_Seg_2 )
   END_RUNG wire#w3
   RUNG wire#w1
      Contact( #OK_TP2_DW )
      Contact( #TP2_DW )
   END_RUNG wire#w4
   RUNG wire#w1
      Contact( #TP2_UP )
   END_RUNG wire#w4
   RUNG wire#powerrail
      Contact( #Mx_ET02 )
      wire#w6
      Contact( #PTF_MSal )
      Contact( #AVTF_MSal )
      Contact( #TP2_DW )
      wire#w7
      Contact( #ConfigFB.Final_E2E4 )
      Contact( #Selec_M4_Salida )
   END_RUNG wire#w5
   RUNG wire#powerrail
      Contact( #Mx_ET60 )
   END_RUNG wire#w6
   RUNG wire#powerrail
      Contact( #Mx_ET61 )
      I_Contact( #Simultaneo_Mx )
   END_RUNG wire#w6
   RUNG wire#powerrail
      Contact( #Mx_ET61 )
      Contact( #Simultaneo_Mx )
      I_Contact( #CNT_pHsMx_E2E4.QD )
      Contact( #PTF_MSal )
      Contact( #AVTF_MSal )
   END_RUNG wire#w7
   RUNG wire#powerrail
      I_Contact( #Termico_E1_Tx )
      Contact( #EstadoZona.Rearme_CBx )
   END_RUNG wire#w8
   // the same network as SCL:
   "DB1_SalidasExterioresDeMesa".Mesa[#Mesa].Avanzar_E2E4 := (((((#Mx_ET20 AND #AVTF_MEnt AND NOT #CNT_pHsMx_E2E4.QD) OR ((#Mx_ET21 OR #Mx_ET22) AND ((#PTF_MSal AND #AVTF_MSal) OR NOT #CNT_pHsMx_E2E4.QD OR ((#pHsMx_Seg_1 OR #pHsMx_Seg_2) AND #TP2_UP)))) AND ((#CNTSeg_pHsMx_E1E3.CVU <= #V_Bajar_TP_Max) OR (#OK_TP2_DW AND #TP2_DW) OR #TP2_UP) AND #Selec_M2_Entrada) OR ((((#Mx_ET02 OR #Mx_ET60 OR (#Mx_ET61 AND NOT #Simultaneo_Mx)) AND #PTF_MSal AND #AVTF_MSal AND #TP2_DW) OR (#Mx_ET61 AND #Simultaneo_Mx AND NOT #CNT_pHsMx_E2E4.QD AND #PTF_MSal AND #AVTF_MSal)) AND #ConfigFB.Final_E2E4 AND #Selec_M4_Salida)) AND #PosTR_E2 AND #EstadoZona.Marcha_CBx AND NOT #EstadoVI.Error_Mx AND NOT #Error_Tx) OR (NOT #Termico_E1_Tx AND #EstadoZona.Rearme_CBx);
END_REGION

REGION Network 120: SALIDAS - Retroceso E2E4
   RUNG wire#powerrail
      Contact( #Mx_ET20 )
      Contact( #AVTF_MEnt )
      wire#w1
      Contact( #PTF_MSal )
      wire#w2
      Contact( #TP2_DW )
      Contact( #Selec_M4_Entrada )
      wire#w5
      Contact( #PosTR_E2 )
      Contact( #EstadoZona.Marcha_CBx )
      I_Contact( #EstadoVI.Error_Mx )
      I_Contact( #Error_Tx )
      wire#w8
      Coil( "DB1_SalidasExterioresDeMesa".Mesa[#Mesa].Retroceder_E2E4 )
   END_RUNG
   RUNG wire#w1
      I_Contact( #CNT_pHsMx_E2E4.QD )
   END_RUNG wire#w2
   RUNG wire#powerrail
      Contact( #Mx_ET21 )
      wire#w3
      Contact( #PTF_MSal )
      Contact( #AVTF_MSal )
   END_RUNG wire#w2
   RUNG wire#powerrail
      Contact( #Mx_ET22 )
   END_RUNG wire#w3
   RUNG wire#w3
      I_Contact( #CNT_pHsMx_E2E4.QD )
   END_RUNG wire#w2
   RUNG wire#w3
      Contact( #pHsMx_Seg_1 )
      wire#w4
      Contact( #TP2_UP )
   END_RUNG wire#w2
   RUNG wire#w3
      Contact( #pHsMx_Seg_2 )
   END_RUNG wire#w4
   RUNG wire#powerrail
      Contact( #Mx_ET02 )
      wire#w6
      Contact( #PTF_MSal )
      Contact( #AVTF_MSal )
      wire#w7
      Contact( #TP2_DW )
      Contact( #ConfigFB.Inicio_E2E4 )
      Contact( #Selec_M2_Salida )
   END_RUNG wire#w5
   RUNG wire#powerrail
      Contact( #Mx_ET60 )
   END_RUNG wire#w6
   RUNG wire#powerrail
      Contact( #Mx_ET61 )
      I_Contact( #Simultaneo_Mx )
   END_RUNG wire#w6
   RUNG wire#powerrail
      Contact( #Mx_ET61 )
      Contact( #Simultaneo_Mx )
      I_Contact( #CNT_pHsMx_E2E4.QD )
      Contact( #PTF_MSal )
      Contact( #AVTF_MSal )
   END_RUNG wire#w7
   RUNG wire#powerrail
      I_Contact( #Termico_E1_Tx )
      Contact( #EstadoZona.Rearme_CBx )
   END_RUNG wire#w8
   // the same network as SCL:
   "DB1_SalidasExterioresDeMesa".Mesa[#Mesa].Retroceder_E2E4 := (((((#Mx_ET20 AND #AVTF_MEnt AND (#PTF_MSal OR NOT #CNT_pHsMx_E2E4.QD)) OR ((#Mx_ET21 OR #Mx_ET22) AND ((#PTF_MSal AND #AVTF_MSal) OR NOT #CNT_pHsMx_E2E4.QD OR ((#pHsMx_Seg_1 OR #pHsMx_Seg_2) AND #TP2_UP)))) AND #TP2_DW AND #Selec_M4_Entrada) OR ((((#Mx_ET02 OR #Mx_ET60 OR (#Mx_ET61 AND NOT #Simultaneo_Mx)) AND #PTF_MSal AND #AVTF_MSal) OR (#Mx_ET61 AND #Simultaneo_Mx AND NOT #CNT_pHsMx_E2E4.QD AND #PTF_MSal AND #AVTF_MSal)) AND #TP2_DW AND #ConfigFB.Inicio_E2E4 AND #Selec_M2_Salida)) AND #PosTR_E2 AND #EstadoZona.Marcha_CBx AND NOT #EstadoVI.Error_Mx AND NOT #Error_Tx) OR (NOT #Termico_E1_Tx AND #EstadoZona.Rearme_CBx);
END_REGION

REGION Network 121: SALIDAS - Parar E2E4
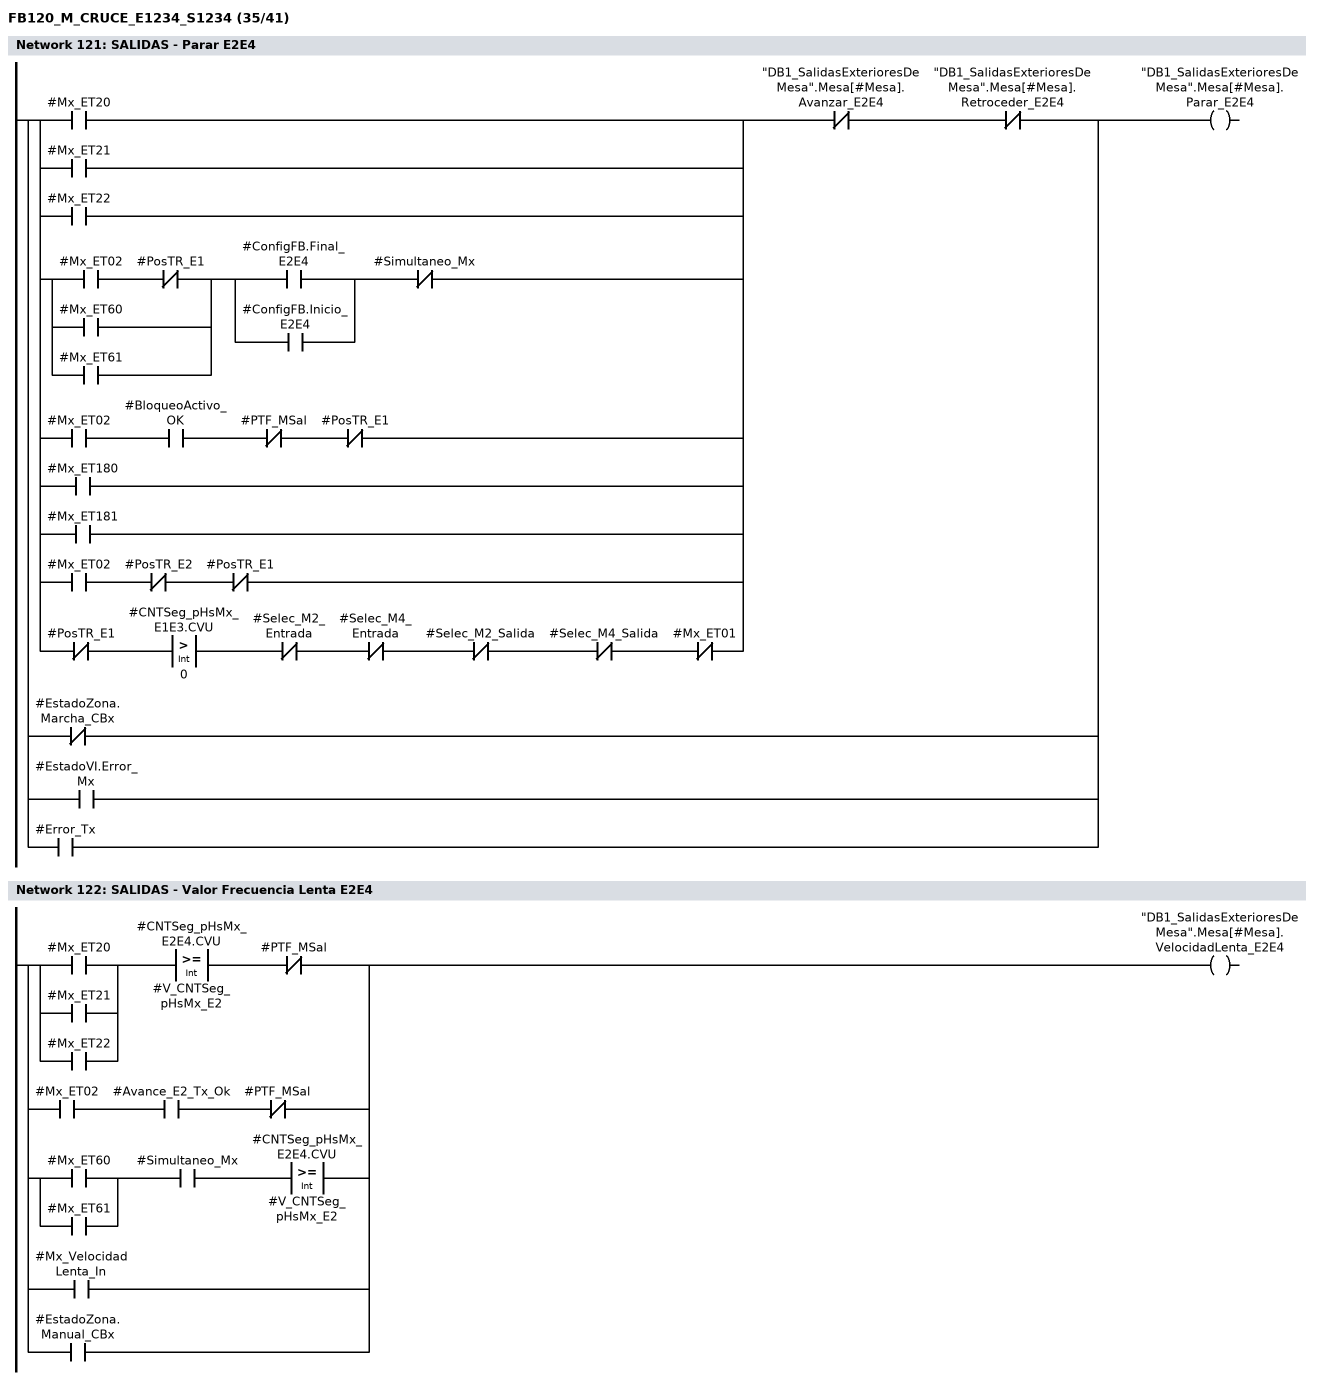
   RUNG wire#powerrail
      Contact( #Mx_ET20 )
      wire#w1
      I_Contact( "DB1_SalidasExterioresDeMesa".Mesa[#Mesa].Avanzar_E2E4 )
      I_Contact( "DB1_SalidasExterioresDeMesa".Mesa[#Mesa].Retroceder_E2E4 )
      wire#w4
      Coil( "DB1_SalidasExterioresDeMesa".Mesa[#Mesa].Parar_E2E4 )
   END_RUNG
   RUNG wire#powerrail
      Contact( #Mx_ET21 )
   END_RUNG wire#w1
   RUNG wire#powerrail
      Contact( #Mx_ET22 )
   END_RUNG wire#w1
   RUNG wire#powerrail
      Contact( #Mx_ET02 )
      I_Contact( #PosTR_E1 )
      wire#w2
      Contact( #ConfigFB.Final_E2E4 )
      wire#w3
      I_Contact( #Simultaneo_Mx )
   END_RUNG wire#w1
   RUNG wire#powerrail
      Contact( #Mx_ET60 )
   END_RUNG wire#w2
   RUNG wire#powerrail
      Contact( #Mx_ET61 )
   END_RUNG wire#w2
   RUNG wire#w2
      Contact( #ConfigFB.Inicio_E2E4 )
   END_RUNG wire#w3
   RUNG wire#powerrail
      Contact( #Mx_ET02 )
      Contact( #BloqueoActivo_OK )
      I_Contact( #PTF_MSal )
      I_Contact( #PosTR_E1 )
   END_RUNG wire#w1
   RUNG wire#powerrail
      Contact( #Mx_ET180 )
   END_RUNG wire#w1
   RUNG wire#powerrail
      Contact( #Mx_ET181 )
   END_RUNG wire#w1
   RUNG wire#powerrail
      Contact( #Mx_ET02 )
      I_Contact( #PosTR_E2 )
      I_Contact( #PosTR_E1 )
   END_RUNG wire#w1
   RUNG wire#powerrail
      I_Contact( #PosTR_E1 )
      { S7_Templates := "SrcType := Int" } GT_Contact(in1 := #CNTSeg_pHsMx_E1E3.CVU, in2 := 0)
      I_Contact( #Selec_M2_Entrada )
      I_Contact( #Selec_M4_Entrada )
      I_Contact( #Selec_M2_Salida )
      I_Contact( #Selec_M4_Salida )
      I_Contact( #Mx_ET01 )
   END_RUNG wire#w1
   RUNG wire#powerrail
      I_Contact( #EstadoZona.Marcha_CBx )
   END_RUNG wire#w4
   RUNG wire#powerrail
      Contact( #EstadoVI.Error_Mx )
   END_RUNG wire#w4
   RUNG wire#powerrail
      Contact( #Error_Tx )
   END_RUNG wire#w4
   // the same network as SCL:
   "DB1_SalidasExterioresDeMesa".Mesa[#Mesa].Parar_E2E4 := ((#Mx_ET20 OR #Mx_ET21 OR #Mx_ET22 OR (((#Mx_ET02 AND NOT #PosTR_E1) OR #Mx_ET60 OR #Mx_ET61) AND (#ConfigFB.Final_E2E4 OR #ConfigFB.Inicio_E2E4) AND NOT #Simultaneo_Mx) OR (#Mx_ET02 AND #BloqueoActivo_OK AND NOT #PTF_MSal AND NOT #PosTR_E1) OR #Mx_ET180 OR #Mx_ET181 OR (#Mx_ET02 AND NOT #PosTR_E2 AND NOT #PosTR_E1) OR (NOT #PosTR_E1 AND (#CNTSeg_pHsMx_E1E3.CVU > 0) AND NOT #Selec_M2_Entrada AND NOT #Selec_M4_Entrada AND NOT #Selec_M2_Salida AND NOT #Selec_M4_Salida AND NOT #Mx_ET01)) AND NOT "DB1_SalidasExterioresDeMesa".Mesa[#Mesa].Avanzar_E2E4 AND NOT "DB1_SalidasExterioresDeMesa".Mesa[#Mesa].Retroceder_E2E4) OR NOT #EstadoZona.Marcha_CBx OR #EstadoVI.Error_Mx OR #Error_Tx;
END_REGION

REGION Network 122: SALIDAS - Valor Frecuencia Lenta E2E4
   RUNG wire#powerrail
      Contact( #Mx_ET20 )
      wire#w1
      { S7_Templates := "SrcType := Int" } GE_Contact(in1 := #CNTSeg_pHsMx_E2E4.CVU, in2 := #V_CNTSeg_pHsMx_E2)
      I_Contact( #PTF_MSal )
      wire#w2
      Coil( "DB1_SalidasExterioresDeMesa".Mesa[#Mesa].VelocidadLenta_E2E4 )
   END_RUNG
   RUNG wire#powerrail
      Contact( #Mx_ET21 )
   END_RUNG wire#w1
   RUNG wire#powerrail
      Contact( #Mx_ET22 )
   END_RUNG wire#w1
   RUNG wire#powerrail
      Contact( #Mx_ET02 )
      Contact( #Avance_E2_Tx_Ok )
      I_Contact( #PTF_MSal )
   END_RUNG wire#w2
   RUNG wire#powerrail
      Contact( #Mx_ET60 )
      wire#w3
      Contact( #Simultaneo_Mx )
      { S7_Templates := "SrcType := Int" } GE_Contact(in1 := #CNTSeg_pHsMx_E2E4.CVU, in2 := #V_CNTSeg_pHsMx_E2)
   END_RUNG wire#w2
   RUNG wire#powerrail
      Contact( #Mx_ET61 )
   END_RUNG wire#w3
   RUNG wire#powerrail
      Contact( #Mx_VelocidadLenta_In )
   END_RUNG wire#w2
   RUNG wire#powerrail
      Contact( #EstadoZona.Manual_CBx )
   END_RUNG wire#w2
   // the same network as SCL:
   "DB1_SalidasExterioresDeMesa".Mesa[#Mesa].VelocidadLenta_E2E4 := ((#Mx_ET20 OR #Mx_ET21 OR #Mx_ET22) AND (#CNTSeg_pHsMx_E2E4.CVU >= #V_CNTSeg_pHsMx_E2) AND NOT #PTF_MSal) OR (#Mx_ET02 AND #Avance_E2_Tx_Ok AND NOT #PTF_MSal) OR ((#Mx_ET60 OR #Mx_ET61) AND #Simultaneo_Mx AND (#CNTSeg_pHsMx_E2E4.CVU >= #V_CNTSeg_pHsMx_E2)) OR #Mx_VelocidadLenta_In OR #EstadoZona.Manual_CBx;
END_REGION

REGION Network 123: SALIDAS - Ir a posicion E1E3
   // DANI: 2021/06/28. BAJAR EL TOPE DE CADENAS SI HAY S2 O S4 EN ETAPA2 Y TR POS RODILLOS
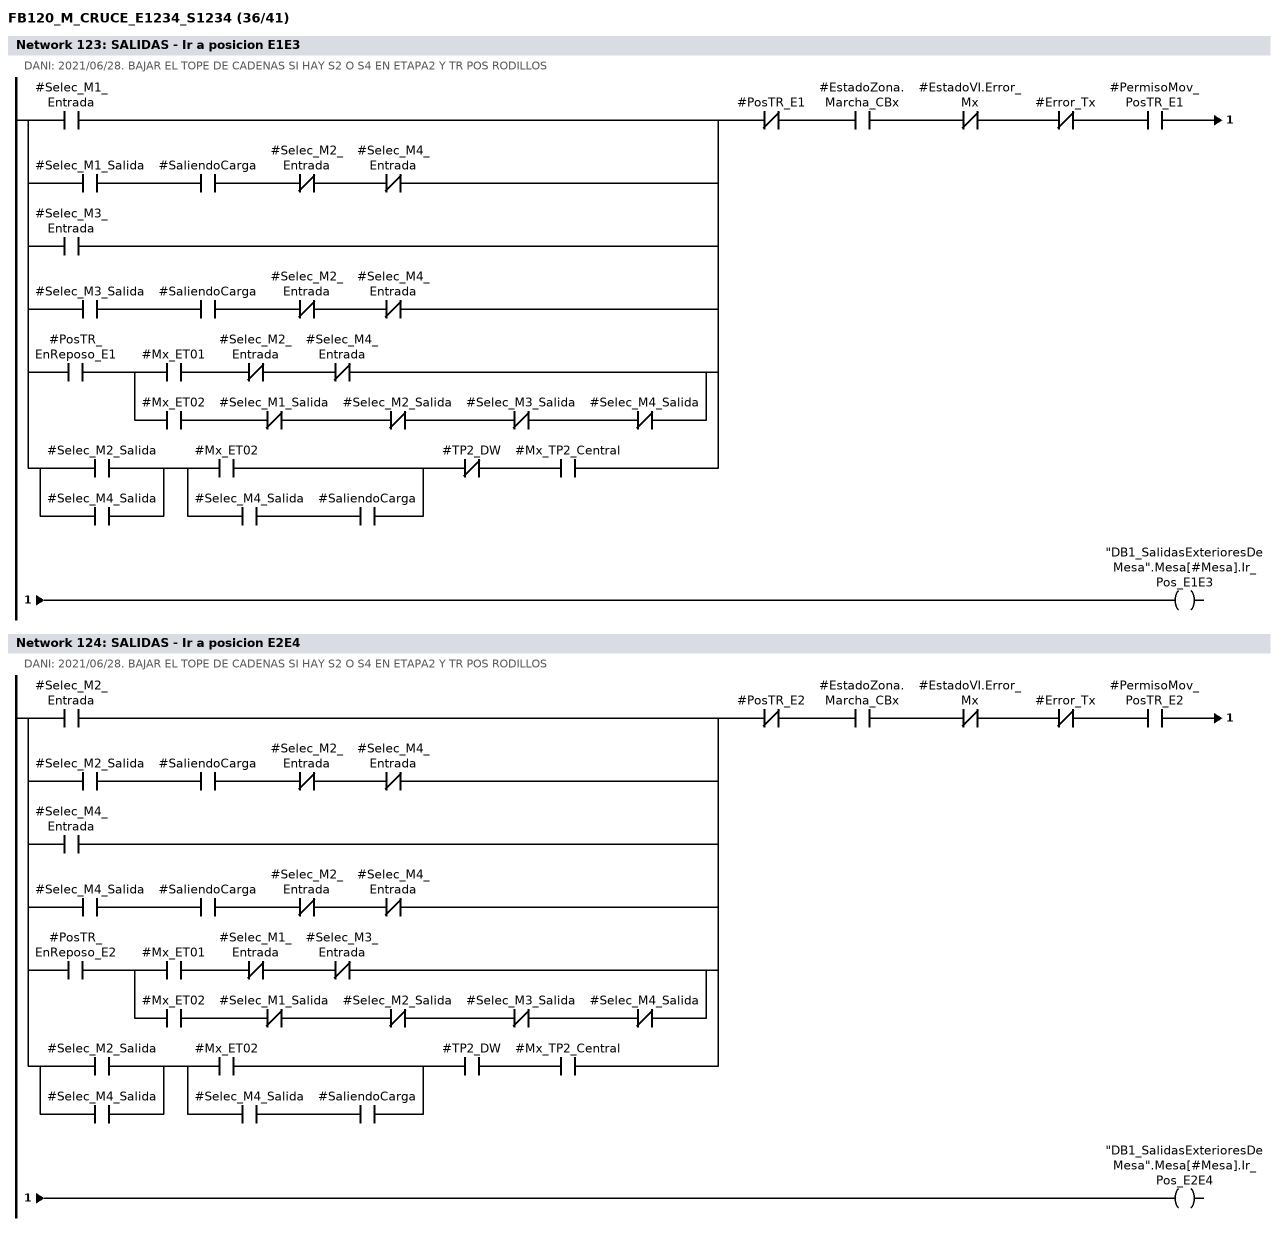
   RUNG wire#powerrail
      Contact( #Selec_M1_Entrada )
      wire#w1
      I_Contact( #PosTR_E1 )
      Contact( #EstadoZona.Marcha_CBx )
      I_Contact( #EstadoVI.Error_Mx )
      I_Contact( #Error_Tx )
      Contact( #PermisoMov_PosTR_E1 )
      Coil( "DB1_SalidasExterioresDeMesa".Mesa[#Mesa].Ir_Pos_E1E3 )
   END_RUNG
   RUNG wire#powerrail
      Contact( #Selec_M1_Salida )
      Contact( #SaliendoCarga )
      I_Contact( #Selec_M2_Entrada )
      I_Contact( #Selec_M4_Entrada )
   END_RUNG wire#w1
   RUNG wire#powerrail
      Contact( #Selec_M3_Entrada )
   END_RUNG wire#w1
   RUNG wire#powerrail
      Contact( #Selec_M3_Salida )
      Contact( #SaliendoCarga )
      I_Contact( #Selec_M2_Entrada )
      I_Contact( #Selec_M4_Entrada )
   END_RUNG wire#w1
   RUNG wire#powerrail
      Contact( #PosTR_EnReposo_E1 )
      wire#w2
      Contact( #Mx_ET01 )
      I_Contact( #Selec_M2_Entrada )
      I_Contact( #Selec_M4_Entrada )
   END_RUNG wire#w1
   RUNG wire#w2
      Contact( #Mx_ET02 )
      I_Contact( #Selec_M1_Salida )
      I_Contact( #Selec_M2_Salida )
      I_Contact( #Selec_M3_Salida )
      I_Contact( #Selec_M4_Salida )
   END_RUNG wire#w1
   RUNG wire#powerrail
      Contact( #Selec_M2_Salida )
      wire#w3
      Contact( #Mx_ET02 )
      wire#w4
      I_Contact( #TP2_DW )
      Contact( #Mx_TP2_Central )
   END_RUNG wire#w1
   RUNG wire#powerrail
      Contact( #Selec_M4_Salida )
   END_RUNG wire#w3
   RUNG wire#w3
      Contact( #Selec_M4_Salida )
      Contact( #SaliendoCarga )
   END_RUNG wire#w4
   // the same network as SCL:
   "DB1_SalidasExterioresDeMesa".Mesa[#Mesa].Ir_Pos_E1E3 := (#Selec_M1_Entrada OR (#Selec_M1_Salida AND #SaliendoCarga AND NOT #Selec_M2_Entrada AND NOT #Selec_M4_Entrada) OR #Selec_M3_Entrada OR (#Selec_M3_Salida AND #SaliendoCarga AND NOT #Selec_M2_Entrada AND NOT #Selec_M4_Entrada) OR (#PosTR_EnReposo_E1 AND ((#Mx_ET01 AND NOT #Selec_M2_Entrada AND NOT #Selec_M4_Entrada) OR (#Mx_ET02 AND NOT #Selec_M1_Salida AND NOT #Selec_M2_Salida AND NOT #Selec_M3_Salida AND NOT #Selec_M4_Salida))) OR ((#Selec_M2_Salida OR #Selec_M4_Salida) AND (#Mx_ET02 OR (#Selec_M4_Salida AND #SaliendoCarga)) AND NOT #TP2_DW AND #Mx_TP2_Central)) AND NOT #PosTR_E1 AND #EstadoZona.Marcha_CBx AND NOT #EstadoVI.Error_Mx AND NOT #Error_Tx AND #PermisoMov_PosTR_E1;
END_REGION

REGION Network 124: SALIDAS - Ir a posicion E2E4
   // DANI: 2021/06/28. BAJAR EL TOPE DE CADENAS SI HAY S2 O S4 EN ETAPA2 Y TR POS RODILLOS
   RUNG wire#powerrail
      Contact( #Selec_M2_Entrada )
      wire#w1
      I_Contact( #PosTR_E2 )
      Contact( #EstadoZona.Marcha_CBx )
      I_Contact( #EstadoVI.Error_Mx )
      I_Contact( #Error_Tx )
      Contact( #PermisoMov_PosTR_E2 )
      Coil( "DB1_SalidasExterioresDeMesa".Mesa[#Mesa].Ir_Pos_E2E4 )
   END_RUNG
   RUNG wire#powerrail
      Contact( #Selec_M2_Salida )
      Contact( #SaliendoCarga )
      I_Contact( #Selec_M2_Entrada )
      I_Contact( #Selec_M4_Entrada )
   END_RUNG wire#w1
   RUNG wire#powerrail
      Contact( #Selec_M4_Entrada )
   END_RUNG wire#w1
   RUNG wire#powerrail
      Contact( #Selec_M4_Salida )
      Contact( #SaliendoCarga )
      I_Contact( #Selec_M2_Entrada )
      I_Contact( #Selec_M4_Entrada )
   END_RUNG wire#w1
   RUNG wire#powerrail
      Contact( #PosTR_EnReposo_E2 )
      wire#w2
      Contact( #Mx_ET01 )
      I_Contact( #Selec_M1_Entrada )
      I_Contact( #Selec_M3_Entrada )
   END_RUNG wire#w1
   RUNG wire#w2
      Contact( #Mx_ET02 )
      I_Contact( #Selec_M1_Salida )
      I_Contact( #Selec_M2_Salida )
      I_Contact( #Selec_M3_Salida )
      I_Contact( #Selec_M4_Salida )
   END_RUNG wire#w1
   RUNG wire#powerrail
      Contact( #Selec_M2_Salida )
      wire#w3
      Contact( #Mx_ET02 )
      wire#w4
      Contact( #TP2_DW )
      Contact( #Mx_TP2_Central )
   END_RUNG wire#w1
   RUNG wire#powerrail
      Contact( #Selec_M4_Salida )
   END_RUNG wire#w3
   RUNG wire#w3
      Contact( #Selec_M4_Salida )
      Contact( #SaliendoCarga )
   END_RUNG wire#w4
   // the same network as SCL:
   "DB1_SalidasExterioresDeMesa".Mesa[#Mesa].Ir_Pos_E2E4 := (#Selec_M2_Entrada OR (#Selec_M2_Salida AND #SaliendoCarga AND NOT #Selec_M2_Entrada AND NOT #Selec_M4_Entrada) OR #Selec_M4_Entrada OR (#Selec_M4_Salida AND #SaliendoCarga AND NOT #Selec_M2_Entrada AND NOT #Selec_M4_Entrada) OR (#PosTR_EnReposo_E2 AND ((#Mx_ET01 AND NOT #Selec_M1_Entrada AND NOT #Selec_M3_Entrada) OR (#Mx_ET02 AND NOT #Selec_M1_Salida AND NOT #Selec_M2_Salida AND NOT #Selec_M3_Salida AND NOT #Selec_M4_Salida))) OR ((#Selec_M2_Salida OR #Selec_M4_Salida) AND (#Mx_ET02 OR (#Selec_M4_Salida AND #SaliendoCarga)) AND #TP2_DW AND #Mx_TP2_Central)) AND NOT #PosTR_E2 AND #EstadoZona.Marcha_CBx AND NOT #EstadoVI.Error_Mx AND NOT #Error_Tx AND #PermisoMov_PosTR_E2;
END_REGION

REGION Network 125: SALIDAS - Bajar TP1
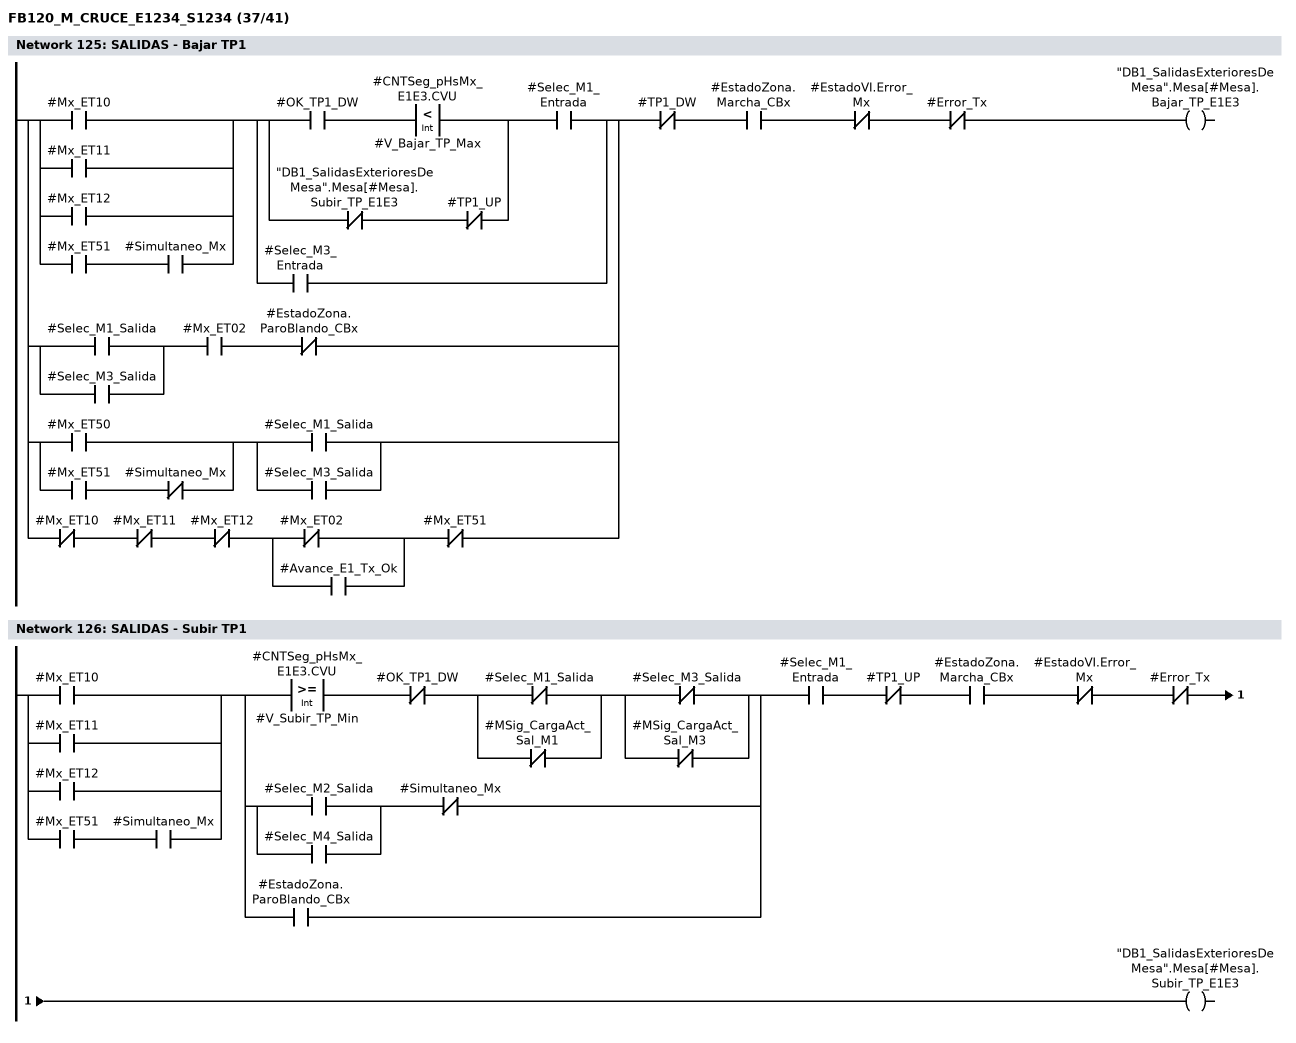
   RUNG wire#powerrail
      Contact( #Mx_ET10 )
      wire#w1
      Contact( #OK_TP1_DW )
      { S7_Templates := "SrcType := Int" } LT_Contact(in1 := #CNTSeg_pHsMx_E1E3.CVU, in2 := #V_Bajar_TP_Max)
      wire#w2
      Contact( #Selec_M1_Entrada )
      wire#w3
      I_Contact( #TP1_DW )
      Contact( #EstadoZona.Marcha_CBx )
      I_Contact( #EstadoVI.Error_Mx )
      I_Contact( #Error_Tx )
      Coil( "DB1_SalidasExterioresDeMesa".Mesa[#Mesa].Bajar_TP_E1E3 )
   END_RUNG
   RUNG wire#powerrail
      Contact( #Mx_ET11 )
   END_RUNG wire#w1
   RUNG wire#powerrail
      Contact( #Mx_ET12 )
   END_RUNG wire#w1
   RUNG wire#powerrail
      Contact( #Mx_ET51 )
      Contact( #Simultaneo_Mx )
   END_RUNG wire#w1
   RUNG wire#w1
      I_Contact( "DB1_SalidasExterioresDeMesa".Mesa[#Mesa].Subir_TP_E1E3 )
      I_Contact( #TP1_UP )
   END_RUNG wire#w2
   RUNG wire#w1
      Contact( #Selec_M3_Entrada )
   END_RUNG wire#w3
   RUNG wire#powerrail
      Contact( #Selec_M1_Salida )
      wire#w4
      Contact( #Mx_ET02 )
      I_Contact( #EstadoZona.ParoBlando_CBx )
   END_RUNG wire#w3
   RUNG wire#powerrail
      Contact( #Selec_M3_Salida )
   END_RUNG wire#w4
   RUNG wire#powerrail
      Contact( #Mx_ET50 )
      wire#w5
      Contact( #Selec_M1_Salida )
   END_RUNG wire#w3
   RUNG wire#powerrail
      Contact( #Mx_ET51 )
      I_Contact( #Simultaneo_Mx )
   END_RUNG wire#w5
   RUNG wire#w5
      Contact( #Selec_M3_Salida )
   END_RUNG wire#w3
   RUNG wire#powerrail
      I_Contact( #Mx_ET10 )
      I_Contact( #Mx_ET11 )
      I_Contact( #Mx_ET12 )
      wire#w6
      I_Contact( #Mx_ET02 )
      wire#w7
      I_Contact( #Mx_ET51 )
   END_RUNG wire#w3
   RUNG wire#w6
      Contact( #Avance_E1_Tx_Ok )
   END_RUNG wire#w7
   // the same network as SCL:
   "DB1_SalidasExterioresDeMesa".Mesa[#Mesa].Bajar_TP_E1E3 := (((#Mx_ET10 OR #Mx_ET11 OR #Mx_ET12 OR (#Mx_ET51 AND #Simultaneo_Mx)) AND ((((#OK_TP1_DW AND (#CNTSeg_pHsMx_E1E3.CVU < #V_Bajar_TP_Max)) OR (NOT "DB1_SalidasExterioresDeMesa".Mesa[#Mesa].Subir_TP_E1E3 AND NOT #TP1_UP)) AND #Selec_M1_Entrada) OR #Selec_M3_Entrada)) OR ((#Selec_M1_Salida OR #Selec_M3_Salida) AND #Mx_ET02 AND NOT #EstadoZona.ParoBlando_CBx) OR ((#Mx_ET50 OR (#Mx_ET51 AND NOT #Simultaneo_Mx)) AND (#Selec_M1_Salida OR #Selec_M3_Salida)) OR (NOT #Mx_ET10 AND NOT #Mx_ET11 AND NOT #Mx_ET12 AND (NOT #Mx_ET02 OR #Avance_E1_Tx_Ok) AND NOT #Mx_ET51)) AND NOT #TP1_DW AND #EstadoZona.Marcha_CBx AND NOT #EstadoVI.Error_Mx AND NOT #Error_Tx;
END_REGION

REGION Network 126: SALIDAS - Subir TP1
   RUNG wire#powerrail
      Contact( #Mx_ET10 )
      wire#w1
      { S7_Templates := "SrcType := Int" } GE_Contact(in1 := #CNTSeg_pHsMx_E1E3.CVU, in2 := #V_Subir_TP_Min)
      I_Contact( #OK_TP1_DW )
      wire#w2
      I_Contact( #Selec_M1_Salida )
      wire#w3
      I_Contact( #Selec_M3_Salida )
      wire#w4
      Contact( #Selec_M1_Entrada )
      I_Contact( #TP1_UP )
      Contact( #EstadoZona.Marcha_CBx )
      I_Contact( #EstadoVI.Error_Mx )
      I_Contact( #Error_Tx )
      Coil( "DB1_SalidasExterioresDeMesa".Mesa[#Mesa].Subir_TP_E1E3 )
   END_RUNG
   RUNG wire#powerrail
      Contact( #Mx_ET11 )
   END_RUNG wire#w1
   RUNG wire#powerrail
      Contact( #Mx_ET12 )
   END_RUNG wire#w1
   RUNG wire#powerrail
      Contact( #Mx_ET51 )
      Contact( #Simultaneo_Mx )
   END_RUNG wire#w1
   RUNG wire#w2
      I_Contact( #MSig_CargaAct_Sal_M1 )
   END_RUNG wire#w3
   RUNG wire#w3
      I_Contact( #MSig_CargaAct_Sal_M3 )
   END_RUNG wire#w4
   RUNG wire#w1
      Contact( #Selec_M2_Salida )
      wire#w5
      I_Contact( #Simultaneo_Mx )
   END_RUNG wire#w4
   RUNG wire#w1
      Contact( #Selec_M4_Salida )
   END_RUNG wire#w5
   RUNG wire#w1
      Contact( #EstadoZona.ParoBlando_CBx )
   END_RUNG wire#w4
   // the same network as SCL:
   "DB1_SalidasExterioresDeMesa".Mesa[#Mesa].Subir_TP_E1E3 := (#Mx_ET10 OR #Mx_ET11 OR #Mx_ET12 OR (#Mx_ET51 AND #Simultaneo_Mx)) AND (((#CNTSeg_pHsMx_E1E3.CVU >= #V_Subir_TP_Min) AND NOT #OK_TP1_DW AND (NOT #Selec_M1_Salida OR NOT #MSig_CargaAct_Sal_M1) AND (NOT #Selec_M3_Salida OR NOT #MSig_CargaAct_Sal_M3)) OR ((#Selec_M2_Salida OR #Selec_M4_Salida) AND NOT #Simultaneo_Mx) OR #EstadoZona.ParoBlando_CBx) AND #Selec_M1_Entrada AND NOT #TP1_UP AND #EstadoZona.Marcha_CBx AND NOT #EstadoVI.Error_Mx AND NOT #Error_Tx;
END_REGION

REGION Network 127: SALIDAS - Bajar TP2
   // DANI: 2021/06/28. BAJAR EL TOPE DE CADENAS SI HAY S2 O S4 EN ETAPA2 Y TR POS RODILLOS
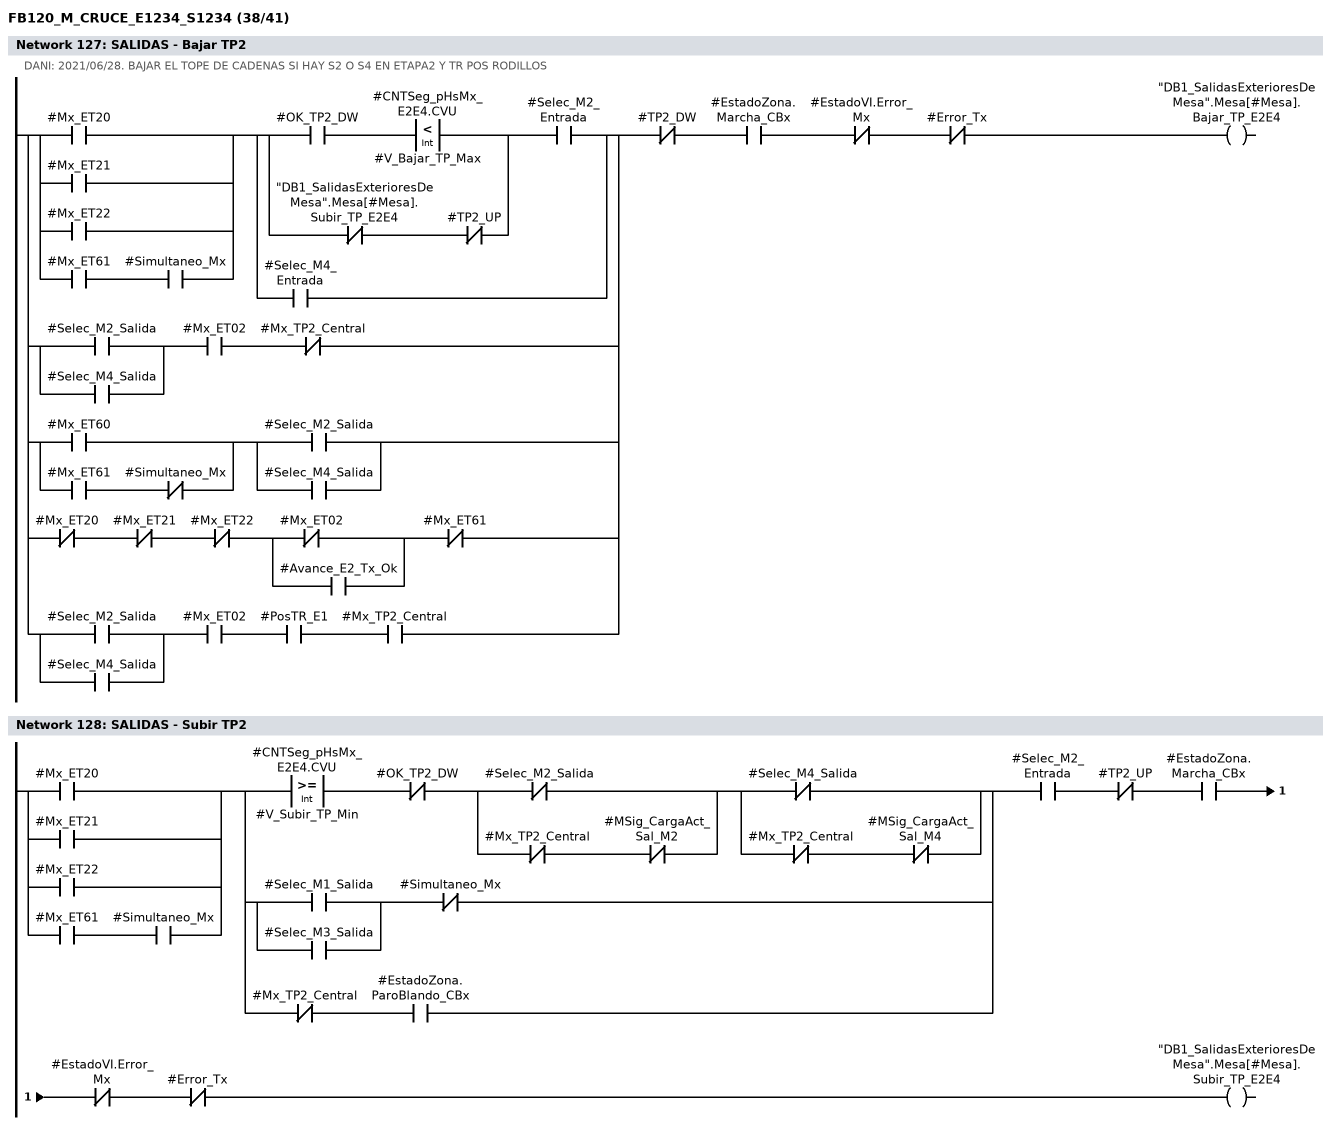
   RUNG wire#powerrail
      Contact( #Mx_ET20 )
      wire#w1
      Contact( #OK_TP2_DW )
      { S7_Templates := "SrcType := Int" } LT_Contact(in1 := #CNTSeg_pHsMx_E2E4.CVU, in2 := #V_Bajar_TP_Max)
      wire#w2
      Contact( #Selec_M2_Entrada )
      wire#w3
      I_Contact( #TP2_DW )
      Contact( #EstadoZona.Marcha_CBx )
      I_Contact( #EstadoVI.Error_Mx )
      I_Contact( #Error_Tx )
      Coil( "DB1_SalidasExterioresDeMesa".Mesa[#Mesa].Bajar_TP_E2E4 )
   END_RUNG
   RUNG wire#powerrail
      Contact( #Mx_ET21 )
   END_RUNG wire#w1
   RUNG wire#powerrail
      Contact( #Mx_ET22 )
   END_RUNG wire#w1
   RUNG wire#powerrail
      Contact( #Mx_ET61 )
      Contact( #Simultaneo_Mx )
   END_RUNG wire#w1
   RUNG wire#w1
      I_Contact( "DB1_SalidasExterioresDeMesa".Mesa[#Mesa].Subir_TP_E2E4 )
      I_Contact( #TP2_UP )
   END_RUNG wire#w2
   RUNG wire#w1
      Contact( #Selec_M4_Entrada )
   END_RUNG wire#w3
   RUNG wire#powerrail
      Contact( #Selec_M2_Salida )
      wire#w4
      Contact( #Mx_ET02 )
      I_Contact( #Mx_TP2_Central )
   END_RUNG wire#w3
   RUNG wire#powerrail
      Contact( #Selec_M4_Salida )
   END_RUNG wire#w4
   RUNG wire#powerrail
      Contact( #Mx_ET60 )
      wire#w5
      Contact( #Selec_M2_Salida )
   END_RUNG wire#w3
   RUNG wire#powerrail
      Contact( #Mx_ET61 )
      I_Contact( #Simultaneo_Mx )
   END_RUNG wire#w5
   RUNG wire#w5
      Contact( #Selec_M4_Salida )
   END_RUNG wire#w3
   RUNG wire#powerrail
      I_Contact( #Mx_ET20 )
      I_Contact( #Mx_ET21 )
      I_Contact( #Mx_ET22 )
      wire#w6
      I_Contact( #Mx_ET02 )
      wire#w7
      I_Contact( #Mx_ET61 )
   END_RUNG wire#w3
   RUNG wire#w6
      Contact( #Avance_E2_Tx_Ok )
   END_RUNG wire#w7
   RUNG wire#powerrail
      Contact( #Selec_M2_Salida )
      wire#w8
      Contact( #Mx_ET02 )
      Contact( #PosTR_E1 )
      Contact( #Mx_TP2_Central )
   END_RUNG wire#w3
   RUNG wire#powerrail
      Contact( #Selec_M4_Salida )
   END_RUNG wire#w8
   // the same network as SCL:
   "DB1_SalidasExterioresDeMesa".Mesa[#Mesa].Bajar_TP_E2E4 := (((#Mx_ET20 OR #Mx_ET21 OR #Mx_ET22 OR (#Mx_ET61 AND #Simultaneo_Mx)) AND ((((#OK_TP2_DW AND (#CNTSeg_pHsMx_E2E4.CVU < #V_Bajar_TP_Max)) OR (NOT "DB1_SalidasExterioresDeMesa".Mesa[#Mesa].Subir_TP_E2E4 AND NOT #TP2_UP)) AND #Selec_M2_Entrada) OR #Selec_M4_Entrada)) OR ((#Selec_M2_Salida OR #Selec_M4_Salida) AND #Mx_ET02 AND NOT #Mx_TP2_Central) OR ((#Mx_ET60 OR (#Mx_ET61 AND NOT #Simultaneo_Mx)) AND (#Selec_M2_Salida OR #Selec_M4_Salida)) OR (NOT #Mx_ET20 AND NOT #Mx_ET21 AND NOT #Mx_ET22 AND (NOT #Mx_ET02 OR #Avance_E2_Tx_Ok) AND NOT #Mx_ET61) OR ((#Selec_M2_Salida OR #Selec_M4_Salida) AND #Mx_ET02 AND #PosTR_E1 AND #Mx_TP2_Central)) AND NOT #TP2_DW AND #EstadoZona.Marcha_CBx AND NOT #EstadoVI.Error_Mx AND NOT #Error_Tx;
END_REGION

REGION Network 128: SALIDAS - Subir TP2
   RUNG wire#powerrail
      Contact( #Mx_ET20 )
      wire#w1
      { S7_Templates := "SrcType := Int" } GE_Contact(in1 := #CNTSeg_pHsMx_E2E4.CVU, in2 := #V_Subir_TP_Min)
      I_Contact( #OK_TP2_DW )
      wire#w2
      I_Contact( #Selec_M2_Salida )
      wire#w3
      I_Contact( #Selec_M4_Salida )
      wire#w4
      Contact( #Selec_M2_Entrada )
      I_Contact( #TP2_UP )
      Contact( #EstadoZona.Marcha_CBx )
      I_Contact( #EstadoVI.Error_Mx )
      I_Contact( #Error_Tx )
      Coil( "DB1_SalidasExterioresDeMesa".Mesa[#Mesa].Subir_TP_E2E4 )
   END_RUNG
   RUNG wire#powerrail
      Contact( #Mx_ET21 )
   END_RUNG wire#w1
   RUNG wire#powerrail
      Contact( #Mx_ET22 )
   END_RUNG wire#w1
   RUNG wire#powerrail
      Contact( #Mx_ET61 )
      Contact( #Simultaneo_Mx )
   END_RUNG wire#w1
   RUNG wire#w2
      I_Contact( #Mx_TP2_Central )
      I_Contact( #MSig_CargaAct_Sal_M2 )
   END_RUNG wire#w3
   RUNG wire#w3
      I_Contact( #Mx_TP2_Central )
      I_Contact( #MSig_CargaAct_Sal_M4 )
   END_RUNG wire#w4
   RUNG wire#w1
      Contact( #Selec_M1_Salida )
      wire#w5
      I_Contact( #Simultaneo_Mx )
   END_RUNG wire#w4
   RUNG wire#w1
      Contact( #Selec_M3_Salida )
   END_RUNG wire#w5
   RUNG wire#w1
      I_Contact( #Mx_TP2_Central )
      Contact( #EstadoZona.ParoBlando_CBx )
   END_RUNG wire#w4
   // the same network as SCL:
   "DB1_SalidasExterioresDeMesa".Mesa[#Mesa].Subir_TP_E2E4 := (#Mx_ET20 OR #Mx_ET21 OR #Mx_ET22 OR (#Mx_ET61 AND #Simultaneo_Mx)) AND (((#CNTSeg_pHsMx_E2E4.CVU >= #V_Subir_TP_Min) AND NOT #OK_TP2_DW AND (NOT #Selec_M2_Salida OR (NOT #Mx_TP2_Central AND NOT #MSig_CargaAct_Sal_M2)) AND (NOT #Selec_M4_Salida OR (NOT #Mx_TP2_Central AND NOT #MSig_CargaAct_Sal_M4))) OR ((#Selec_M1_Salida OR #Selec_M3_Salida) AND NOT #Simultaneo_Mx) OR (NOT #Mx_TP2_Central AND #EstadoZona.ParoBlando_CBx)) AND #Selec_M2_Entrada AND NOT #TP2_UP AND #EstadoZona.Marcha_CBx AND NOT #EstadoVI.Error_Mx AND NOT #Error_Tx;
END_REGION

REGION Network 129: ESTADOS DE LA MESA
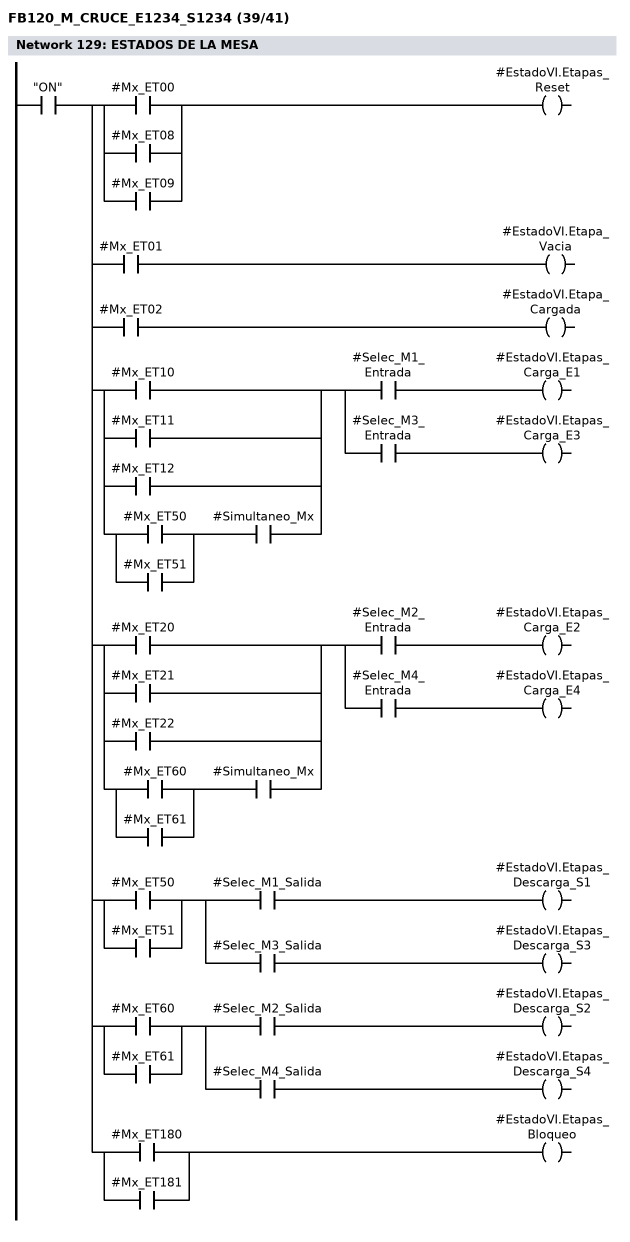
   RUNG wire#powerrail
      Contact( "ON" )
      wire#w1
      Contact( #Mx_ET00 )
      wire#w2
      Coil( #EstadoVI.Etapas_Reset )
   END_RUNG
   RUNG wire#w1
      Contact( #Mx_ET08 )
   END_RUNG wire#w2
   RUNG wire#w1
      Contact( #Mx_ET09 )
   END_RUNG wire#w2
   RUNG wire#w1
      Contact( #Mx_ET01 )
      Coil( #EstadoVI.Etapa_Vacia )
   END_RUNG
   RUNG wire#w1
      Contact( #Mx_ET02 )
      Coil( #EstadoVI.Etapa_Cargada )
   END_RUNG
   RUNG wire#w1
      Contact( #Mx_ET10 )
      wire#w3
      Contact( #Selec_M1_Entrada )
      Coil( #EstadoVI.Etapas_Carga_E1 )
   END_RUNG
   RUNG wire#w1
      Contact( #Mx_ET11 )
   END_RUNG wire#w3
   RUNG wire#w1
      Contact( #Mx_ET12 )
   END_RUNG wire#w3
   RUNG wire#w1
      Contact( #Mx_ET50 )
      wire#w4
      Contact( #Simultaneo_Mx )
   END_RUNG wire#w3
   RUNG wire#w1
      Contact( #Mx_ET51 )
   END_RUNG wire#w4
   RUNG wire#w3
      Contact( #Selec_M3_Entrada )
      Coil( #EstadoVI.Etapas_Carga_E3 )
   END_RUNG
   RUNG wire#w1
      Contact( #Mx_ET20 )
      wire#w5
      Contact( #Selec_M2_Entrada )
      Coil( #EstadoVI.Etapas_Carga_E2 )
   END_RUNG
   RUNG wire#w1
      Contact( #Mx_ET21 )
   END_RUNG wire#w5
   RUNG wire#w1
      Contact( #Mx_ET22 )
   END_RUNG wire#w5
   RUNG wire#w1
      Contact( #Mx_ET60 )
      wire#w6
      Contact( #Simultaneo_Mx )
   END_RUNG wire#w5
   RUNG wire#w1
      Contact( #Mx_ET61 )
   END_RUNG wire#w6
   RUNG wire#w5
      Contact( #Selec_M4_Entrada )
      Coil( #EstadoVI.Etapas_Carga_E4 )
   END_RUNG
   RUNG wire#w1
      Contact( #Mx_ET50 )
      wire#w7
      Contact( #Selec_M1_Salida )
      Coil( #EstadoVI.Etapas_Descarga_S1 )
   END_RUNG
   RUNG wire#w1
      Contact( #Mx_ET51 )
   END_RUNG wire#w7
   RUNG wire#w7
      Contact( #Selec_M3_Salida )
      Coil( #EstadoVI.Etapas_Descarga_S3 )
   END_RUNG
   RUNG wire#w1
      Contact( #Mx_ET60 )
      wire#w8
      Contact( #Selec_M2_Salida )
      Coil( #EstadoVI.Etapas_Descarga_S2 )
   END_RUNG
   RUNG wire#w1
      Contact( #Mx_ET61 )
   END_RUNG wire#w8
   RUNG wire#w8
      Contact( #Selec_M4_Salida )
      Coil( #EstadoVI.Etapas_Descarga_S4 )
   END_RUNG
   RUNG wire#w1
      Contact( #Mx_ET180 )
      wire#w9
      Coil( #EstadoVI.Etapas_Bloqueo )
   END_RUNG
   RUNG wire#w1
      Contact( #Mx_ET181 )
   END_RUNG wire#w9
   // the same network as SCL:
   #EstadoVI.Etapas_Reset := "ON" AND (#Mx_ET00 OR #Mx_ET08 OR #Mx_ET09);
   #EstadoVI.Etapa_Vacia := "ON" AND #Mx_ET01;
   #EstadoVI.Etapa_Cargada := "ON" AND #Mx_ET02;
   #_w1 := "ON" AND (#Mx_ET10 OR #Mx_ET11 OR #Mx_ET12 OR ((#Mx_ET50 OR #Mx_ET51) AND #Simultaneo_Mx));
   #EstadoVI.Etapas_Carga_E1 := #_w1 AND #Selec_M1_Entrada;
   #EstadoVI.Etapas_Carga_E3 := #_w1 AND #Selec_M3_Entrada;
   #_w2 := "ON" AND (#Mx_ET20 OR #Mx_ET21 OR #Mx_ET22 OR ((#Mx_ET60 OR #Mx_ET61) AND #Simultaneo_Mx));
   #EstadoVI.Etapas_Carga_E2 := #_w2 AND #Selec_M2_Entrada;
   #EstadoVI.Etapas_Carga_E4 := #_w2 AND #Selec_M4_Entrada;
   #_w3 := "ON" AND (#Mx_ET50 OR #Mx_ET51);
   #EstadoVI.Etapas_Descarga_S1 := #_w3 AND #Selec_M1_Salida;
   #EstadoVI.Etapas_Descarga_S3 := #_w3 AND #Selec_M3_Salida;
   #_w4 := "ON" AND (#Mx_ET60 OR #Mx_ET61);
   #EstadoVI.Etapas_Descarga_S2 := #_w4 AND #Selec_M2_Salida;
   #EstadoVI.Etapas_Descarga_S4 := #_w4 AND #Selec_M4_Salida;
   #EstadoVI.Etapas_Bloqueo := "ON" AND (#Mx_ET180 OR #Mx_ET181);
END_REGION

REGION Network 130: ESTADO ENTRADAS DE LA MESA
   // MODIF: TRANSFER UP, TRANSFER_DW, TOPE_UP_2, TOPE_DW_2
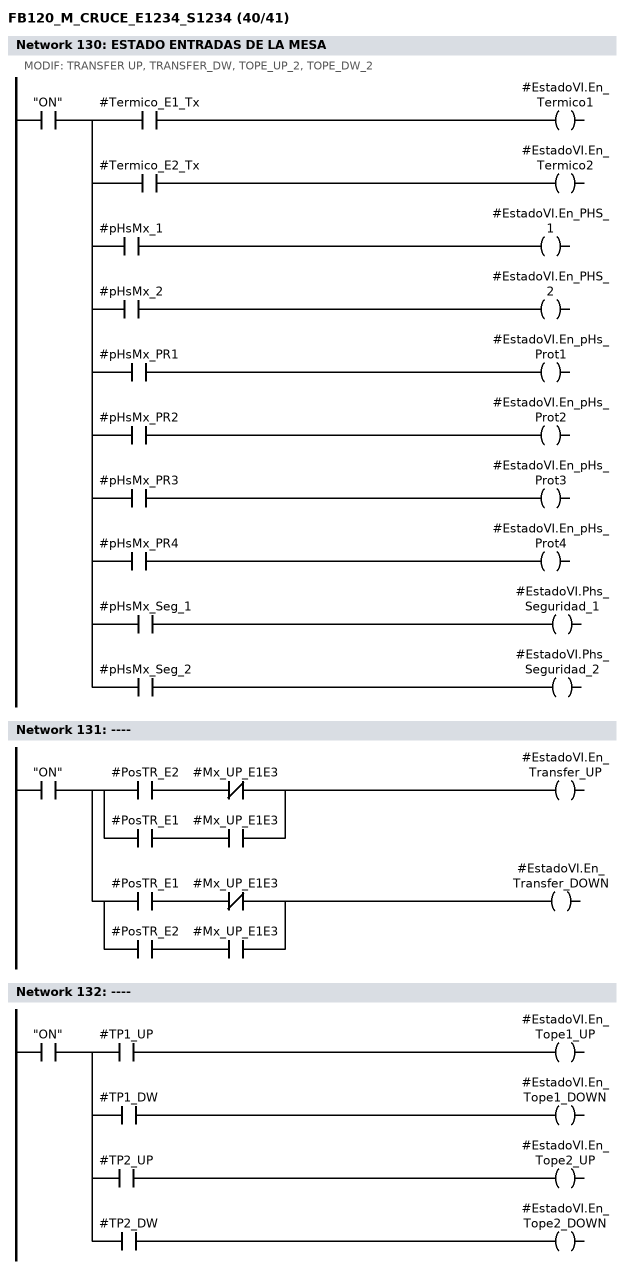
   RUNG wire#powerrail
      Contact( "ON" )
      wire#w1
      Contact( #Termico_E1_Tx )
      Coil( #EstadoVI.En_Termico1 )
   END_RUNG
   RUNG wire#w1
      Contact( #Termico_E2_Tx )
      Coil( #EstadoVI.En_Termico2 )
   END_RUNG
   RUNG wire#w1
      Contact( #pHsMx_1 )
      Coil( #EstadoVI.En_PHS_1 )
   END_RUNG
   RUNG wire#w1
      Contact( #pHsMx_2 )
      Coil( #EstadoVI.En_PHS_2 )
   END_RUNG
   RUNG wire#w1
      Contact( #pHsMx_PR1 )
      Coil( #EstadoVI.En_pHs_Prot1 )
   END_RUNG
   RUNG wire#w1
      Contact( #pHsMx_PR2 )
      Coil( #EstadoVI.En_pHs_Prot2 )
   END_RUNG
   RUNG wire#w1
      Contact( #pHsMx_PR3 )
      Coil( #EstadoVI.En_pHs_Prot3 )
   END_RUNG
   RUNG wire#w1
      Contact( #pHsMx_PR4 )
      Coil( #EstadoVI.En_pHs_Prot4 )
   END_RUNG
   RUNG wire#w1
      Contact( #pHsMx_Seg_1 )
      Coil( #EstadoVI.Phs_Seguridad_1 )
   END_RUNG
   RUNG wire#w1
      Contact( #pHsMx_Seg_2 )
      Coil( #EstadoVI.Phs_Seguridad_2 )
   END_RUNG
   // the same network as SCL:
   #EstadoVI.En_Termico1 := "ON" AND #Termico_E1_Tx;
   #EstadoVI.En_Termico2 := "ON" AND #Termico_E2_Tx;
   #EstadoVI.En_PHS_1 := "ON" AND #pHsMx_1;
   #EstadoVI.En_PHS_2 := "ON" AND #pHsMx_2;
   #EstadoVI.En_pHs_Prot1 := "ON" AND #pHsMx_PR1;
   #EstadoVI.En_pHs_Prot2 := "ON" AND #pHsMx_PR2;
   #EstadoVI.En_pHs_Prot3 := "ON" AND #pHsMx_PR3;
   #EstadoVI.En_pHs_Prot4 := "ON" AND #pHsMx_PR4;
   #EstadoVI.Phs_Seguridad_1 := "ON" AND #pHsMx_Seg_1;
   #EstadoVI.Phs_Seguridad_2 := "ON" AND #pHsMx_Seg_2;
END_REGION

REGION Network 131: ----
   RUNG wire#powerrail
      Contact( "ON" )
      wire#w1
      Contact( #PosTR_E2 )
      I_Contact( #Mx_UP_E1E3 )
      wire#w2
      Coil( #EstadoVI.En_Transfer_UP )
   END_RUNG
   RUNG wire#w1
      Contact( #PosTR_E1 )
      Contact( #Mx_UP_E1E3 )
   END_RUNG wire#w2
   RUNG wire#w1
      Contact( #PosTR_E1 )
      I_Contact( #Mx_UP_E1E3 )
      wire#w3
      Coil( #EstadoVI.En_Transfer_DOWN )
   END_RUNG
   RUNG wire#w1
      Contact( #PosTR_E2 )
      Contact( #Mx_UP_E1E3 )
   END_RUNG wire#w3
   // the same network as SCL:
   #EstadoVI.En_Transfer_UP := "ON" AND ((#PosTR_E2 AND NOT #Mx_UP_E1E3) OR (#PosTR_E1 AND #Mx_UP_E1E3));
   #EstadoVI.En_Transfer_DOWN := "ON" AND ((#PosTR_E1 AND NOT #Mx_UP_E1E3) OR (#PosTR_E2 AND #Mx_UP_E1E3));
END_REGION

REGION Network 132: ----
   RUNG wire#powerrail
      Contact( "ON" )
      wire#w1
      Contact( #TP1_UP )
      Coil( #EstadoVI.En_Tope1_UP )
   END_RUNG
   RUNG wire#w1
      Contact( #TP1_DW )
      Coil( #EstadoVI.En_Tope1_DOWN )
   END_RUNG
   RUNG wire#w1
      Contact( #TP2_UP )
      Coil( #EstadoVI.En_Tope2_UP )
   END_RUNG
   RUNG wire#w1
      Contact( #TP2_DW )
      Coil( #EstadoVI.En_Tope2_DOWN )
   END_RUNG
   // the same network as SCL:
   #EstadoVI.En_Tope1_UP := "ON" AND #TP1_UP;
   #EstadoVI.En_Tope1_DOWN := "ON" AND #TP1_DW;
   #EstadoVI.En_Tope2_UP := "ON" AND #TP2_UP;
   #EstadoVI.En_Tope2_DOWN := "ON" AND #TP2_DW;
END_REGION

REGION Network 133: SALIDAS DE LA MESA
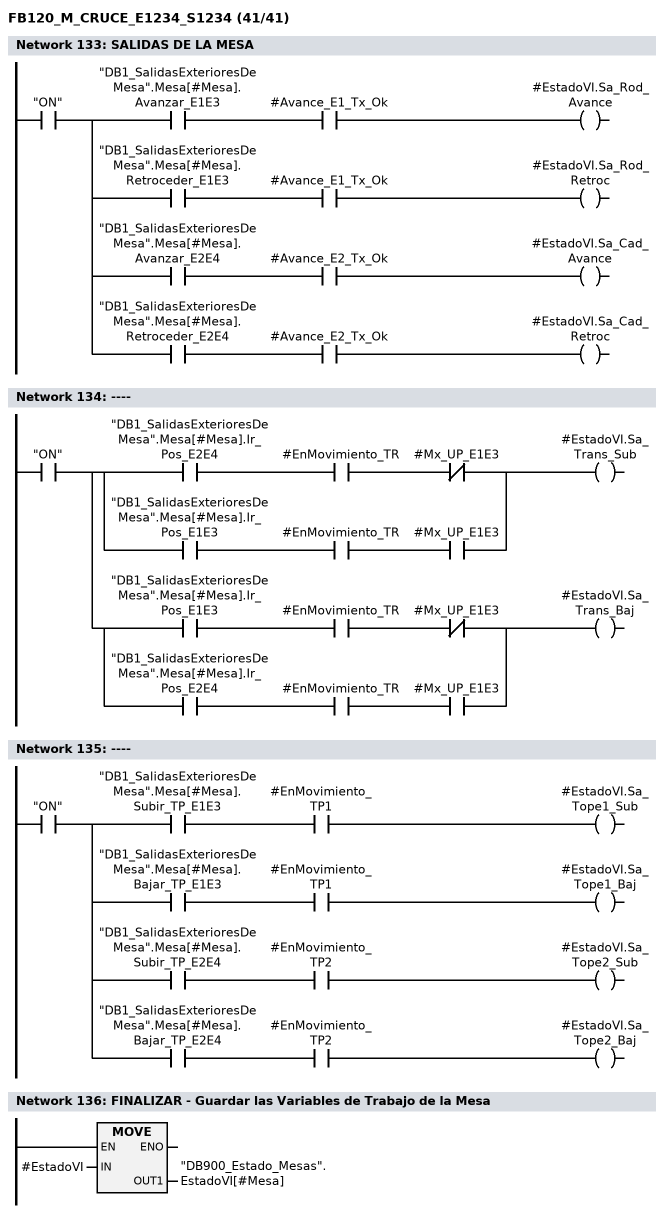
   RUNG wire#powerrail
      Contact( "ON" )
      wire#w1
      Contact( "DB1_SalidasExterioresDeMesa".Mesa[#Mesa].Avanzar_E1E3 )
      Contact( #Avance_E1_Tx_Ok )
      Coil( #EstadoVI.Sa_Rod_Avance )
   END_RUNG
   RUNG wire#w1
      Contact( "DB1_SalidasExterioresDeMesa".Mesa[#Mesa].Retroceder_E1E3 )
      Contact( #Avance_E1_Tx_Ok )
      Coil( #EstadoVI.Sa_Rod_Retroc )
   END_RUNG
   RUNG wire#w1
      Contact( "DB1_SalidasExterioresDeMesa".Mesa[#Mesa].Avanzar_E2E4 )
      Contact( #Avance_E2_Tx_Ok )
      Coil( #EstadoVI.Sa_Cad_Avance )
   END_RUNG
   RUNG wire#w1
      Contact( "DB1_SalidasExterioresDeMesa".Mesa[#Mesa].Retroceder_E2E4 )
      Contact( #Avance_E2_Tx_Ok )
      Coil( #EstadoVI.Sa_Cad_Retroc )
   END_RUNG
   // the same network as SCL:
   #EstadoVI.Sa_Rod_Avance := "ON" AND "DB1_SalidasExterioresDeMesa".Mesa[#Mesa].Avanzar_E1E3 AND #Avance_E1_Tx_Ok;
   #EstadoVI.Sa_Rod_Retroc := "ON" AND "DB1_SalidasExterioresDeMesa".Mesa[#Mesa].Retroceder_E1E3 AND #Avance_E1_Tx_Ok;
   #EstadoVI.Sa_Cad_Avance := "ON" AND "DB1_SalidasExterioresDeMesa".Mesa[#Mesa].Avanzar_E2E4 AND #Avance_E2_Tx_Ok;
   #EstadoVI.Sa_Cad_Retroc := "ON" AND "DB1_SalidasExterioresDeMesa".Mesa[#Mesa].Retroceder_E2E4 AND #Avance_E2_Tx_Ok;
END_REGION

REGION Network 134: ----
   RUNG wire#powerrail
      Contact( "ON" )
      wire#w1
      Contact( "DB1_SalidasExterioresDeMesa".Mesa[#Mesa].Ir_Pos_E2E4 )
      Contact( #EnMovimiento_TR )
      I_Contact( #Mx_UP_E1E3 )
      wire#w2
      Coil( #EstadoVI.Sa_Trans_Sub )
   END_RUNG
   RUNG wire#w1
      Contact( "DB1_SalidasExterioresDeMesa".Mesa[#Mesa].Ir_Pos_E1E3 )
      Contact( #EnMovimiento_TR )
      Contact( #Mx_UP_E1E3 )
   END_RUNG wire#w2
   RUNG wire#w1
      Contact( "DB1_SalidasExterioresDeMesa".Mesa[#Mesa].Ir_Pos_E1E3 )
      Contact( #EnMovimiento_TR )
      I_Contact( #Mx_UP_E1E3 )
      wire#w3
      Coil( #EstadoVI.Sa_Trans_Baj )
   END_RUNG
   RUNG wire#w1
      Contact( "DB1_SalidasExterioresDeMesa".Mesa[#Mesa].Ir_Pos_E2E4 )
      Contact( #EnMovimiento_TR )
      Contact( #Mx_UP_E1E3 )
   END_RUNG wire#w3
   // the same network as SCL:
   #EstadoVI.Sa_Trans_Sub := "ON" AND (("DB1_SalidasExterioresDeMesa".Mesa[#Mesa].Ir_Pos_E2E4 AND #EnMovimiento_TR AND NOT #Mx_UP_E1E3) OR ("DB1_SalidasExterioresDeMesa".Mesa[#Mesa].Ir_Pos_E1E3 AND #EnMovimiento_TR AND #Mx_UP_E1E3));
   #EstadoVI.Sa_Trans_Baj := "ON" AND (("DB1_SalidasExterioresDeMesa".Mesa[#Mesa].Ir_Pos_E1E3 AND #EnMovimiento_TR AND NOT #Mx_UP_E1E3) OR ("DB1_SalidasExterioresDeMesa".Mesa[#Mesa].Ir_Pos_E2E4 AND #EnMovimiento_TR AND #Mx_UP_E1E3));
END_REGION

REGION Network 135: ----
   RUNG wire#powerrail
      Contact( "ON" )
      wire#w1
      Contact( "DB1_SalidasExterioresDeMesa".Mesa[#Mesa].Subir_TP_E1E3 )
      Contact( #EnMovimiento_TP1 )
      Coil( #EstadoVI.Sa_Tope1_Sub )
   END_RUNG
   RUNG wire#w1
      Contact( "DB1_SalidasExterioresDeMesa".Mesa[#Mesa].Bajar_TP_E1E3 )
      Contact( #EnMovimiento_TP1 )
      Coil( #EstadoVI.Sa_Tope1_Baj )
   END_RUNG
   RUNG wire#w1
      Contact( "DB1_SalidasExterioresDeMesa".Mesa[#Mesa].Subir_TP_E2E4 )
      Contact( #EnMovimiento_TP2 )
      Coil( #EstadoVI.Sa_Tope2_Sub )
   END_RUNG
   RUNG wire#w1
      Contact( "DB1_SalidasExterioresDeMesa".Mesa[#Mesa].Bajar_TP_E2E4 )
      Contact( #EnMovimiento_TP2 )
      Coil( #EstadoVI.Sa_Tope2_Baj )
   END_RUNG
   // the same network as SCL:
   #EstadoVI.Sa_Tope1_Sub := "ON" AND "DB1_SalidasExterioresDeMesa".Mesa[#Mesa].Subir_TP_E1E3 AND #EnMovimiento_TP1;
   #EstadoVI.Sa_Tope1_Baj := "ON" AND "DB1_SalidasExterioresDeMesa".Mesa[#Mesa].Bajar_TP_E1E3 AND #EnMovimiento_TP1;
   #EstadoVI.Sa_Tope2_Sub := "ON" AND "DB1_SalidasExterioresDeMesa".Mesa[#Mesa].Subir_TP_E2E4 AND #EnMovimiento_TP2;
   #EstadoVI.Sa_Tope2_Baj := "ON" AND "DB1_SalidasExterioresDeMesa".Mesa[#Mesa].Bajar_TP_E2E4 AND #EnMovimiento_TP2;
END_REGION

REGION Network 136: FINALIZAR - Guardar las Variables de Trabajo de la Mesa
   RUNG wire#powerrail
      Move(in := #EstadoVI, out1 => "DB900_Estado_Mesas".EstadoVI[#Mesa])
   END_RUNG
   // the same network as SCL:
   "DB900_Estado_Mesas".EstadoVI[#Mesa] := #EstadoVI;
END_REGION
END_FUNCTION_BLOCK
